// TIA Portal V17 export
// export: Created 2025-03-05T07:59:31.0674442Z, ExportSetting WithDefaults, DisplayName Totally Integrated Automation Portal, DisplayVersion V17 Update 8, DisplayName TIA Portal Openness, DisplayVersion V17 Update 8, DisplayName TIA Portal Version Control Interface, DisplayVersion V17, DisplayName SINAMICS Startdrive Advanced, DisplayVersion V17 SP2, DisplayName SINAMICS Startdrive G110M, G120, G120C, G120D, G120P, G115D, DisplayVersion V17 SP2, DisplayName SINAMICS Startdrive G130, G150, S120, S150, SINAMICS MV, S210, DisplayVersion V17 SP2, DisplayName STEP 7 Professional, DisplayVersion V17 Update 8, DisplayName SINUMERIK ONE STEP 7 Toolbox, DisplayVersion V17 Update 12, DisplayName SINUMERIK 840D sl STEP 7 Toolbox, DisplayVersion V17 Update 12, DisplayName STEP 7 Safety, DisplayVersion V17 Update 6, DisplayName WinCC Advanced, DisplayVersion V17 Update 8
FUNCTION "FC341_NCK_M_CH1_UNIT_1_STA_0" : Void   // FC341, LAD
TITLE = Channel 1 data
{ S7_Optimized_Access := 'FALSE' }
AUTHOR : ETXETAR
VERSION : 1.0
// stored: AutoNumber false, IsIECCheckEnabled false, SetENOAutomatically false, UDAEnableTagReadback false
   VAR_TEMP
      auxm3 : Bool;
      auxm5 : Bool;
      M253_TORQUE_ACTUAL_AUX_1 : Real;
      M253_TORQUE_ACTUAL_AUX_2 : Real;
   END_VAR
   VAR_TEMP   // added for the SCL form of the ladder/FBD networks
      _w1 : Bool;
      _w2 : Bool;
   END_VAR
BEGIN

REGION Network 1: CALL FB331 M CODE EXTENDED CH1 / M CODE EXTENDED CHANNEL 1
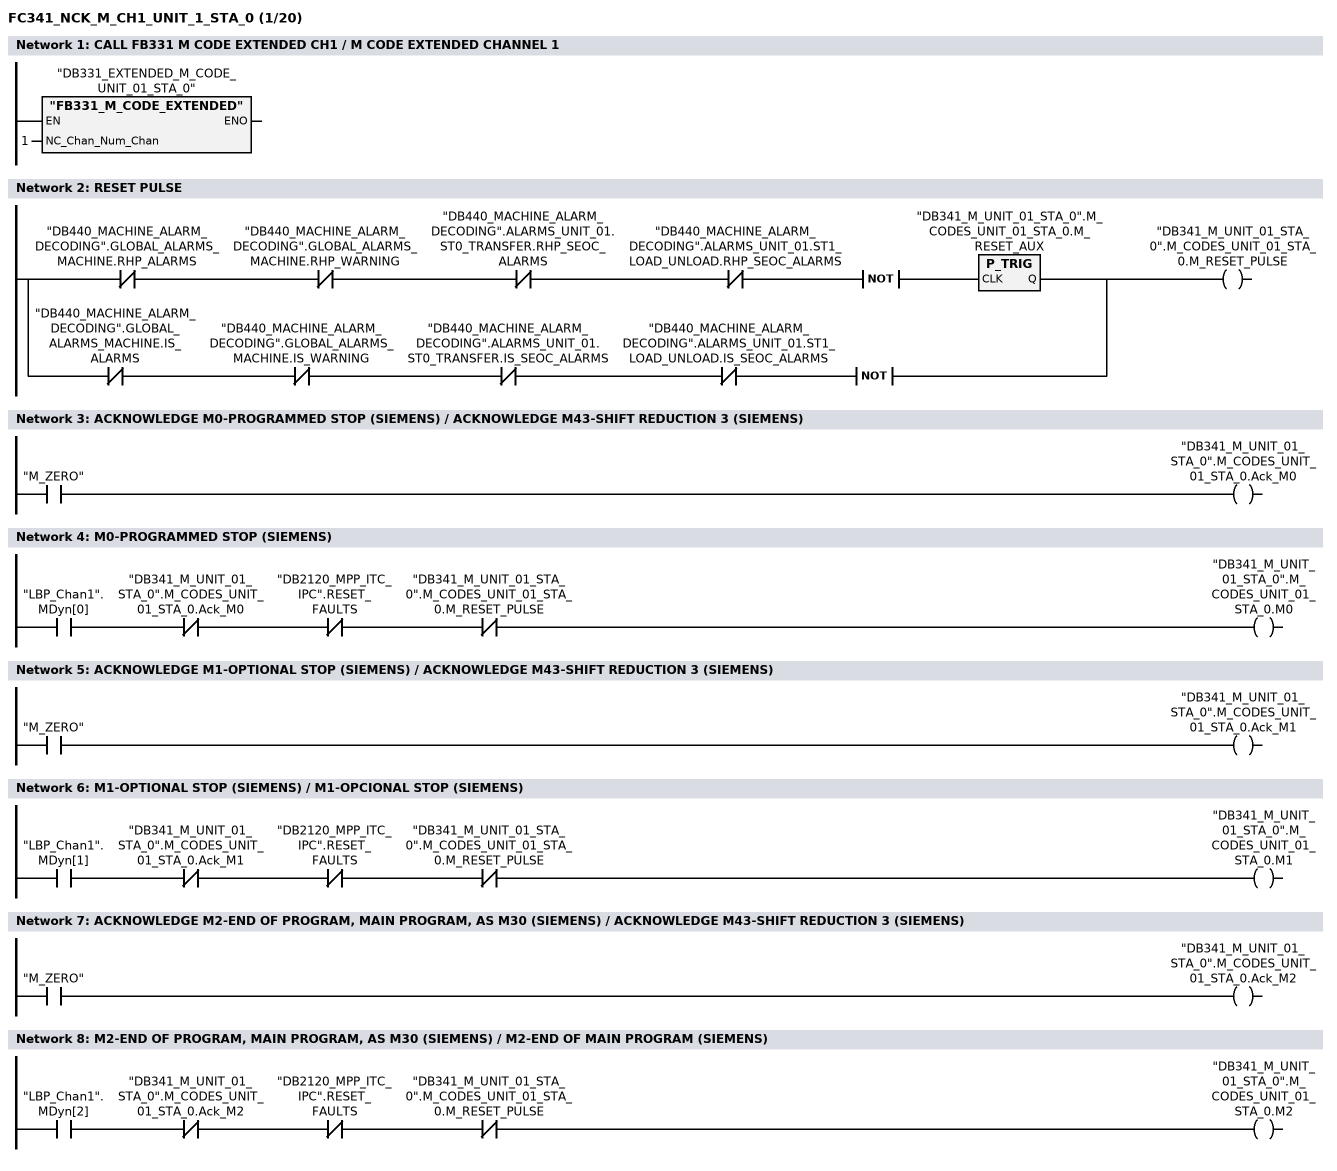
   RUNG wire#powerrail
      "DB331_EXTENDED_M_CODE_UNIT_01_STA_0"(NC_Chan_Num_Chan := 1)
   END_RUNG
   // the same network as SCL:
   "DB331_EXTENDED_M_CODE_UNIT_01_STA_0"(NC_Chan_Num_Chan := 1);   // "FB331_M_CODE_EXTENDED"
END_REGION

REGION Network 2: RESET PULSE
   RUNG wire#powerrail
      I_Contact( "DB440_MACHINE_ALARM_DECODING".GLOBAL_ALARMS_MACHINE.RHP_ALARMS )
      I_Contact( "DB440_MACHINE_ALARM_DECODING".GLOBAL_ALARMS_MACHINE.RHP_WARNING )
      I_Contact( "DB440_MACHINE_ALARM_DECODING".ALARMS_UNIT_01.ST0_TRANSFER.RHP_SEOC_ALARMS )
      I_Contact( "DB440_MACHINE_ALARM_DECODING".ALARMS_UNIT_01.ST1_LOAD_UNLOAD.RHP_SEOC_ALARMS )
      Not()
      P_Trig( "DB341_M_UNIT_01_STA_0".M_CODES_UNIT_01_STA_0.M_RESET_AUX )
      wire#w1
      Coil( "DB341_M_UNIT_01_STA_0".M_CODES_UNIT_01_STA_0.M_RESET_PULSE )
   END_RUNG
   RUNG wire#powerrail
      I_Contact( "DB440_MACHINE_ALARM_DECODING".GLOBAL_ALARMS_MACHINE.IS_ALARMS )
      I_Contact( "DB440_MACHINE_ALARM_DECODING".GLOBAL_ALARMS_MACHINE.IS_WARNING )
      I_Contact( "DB440_MACHINE_ALARM_DECODING".ALARMS_UNIT_01.ST0_TRANSFER.IS_SEOC_ALARMS )
      I_Contact( "DB440_MACHINE_ALARM_DECODING".ALARMS_UNIT_01.ST1_LOAD_UNLOAD.IS_SEOC_ALARMS )
      Not()
   END_RUNG wire#w1
   // the same network as SCL:
   #_w1 := NOT (NOT "DB440_MACHINE_ALARM_DECODING".GLOBAL_ALARMS_MACHINE.RHP_ALARMS AND NOT "DB440_MACHINE_ALARM_DECODING".GLOBAL_ALARMS_MACHINE.RHP_WARNING AND NOT "DB440_MACHINE_ALARM_DECODING".ALARMS_UNIT_01.ST0_TRANSFER.RHP_SEOC_ALARMS AND NOT "DB440_MACHINE_ALARM_DECODING".ALARMS_UNIT_01.ST1_LOAD_UNLOAD.RHP_SEOC_ALARMS);
   #_w2 := #_w1 AND NOT "DB341_M_UNIT_01_STA_0".M_CODES_UNIT_01_STA_0.M_RESET_AUX;   // rising edge
   "DB341_M_UNIT_01_STA_0".M_CODES_UNIT_01_STA_0.M_RESET_AUX := #_w1;
   "DB341_M_UNIT_01_STA_0".M_CODES_UNIT_01_STA_0.M_RESET_PULSE := #_w2 OR NOT (NOT "DB440_MACHINE_ALARM_DECODING".GLOBAL_ALARMS_MACHINE.IS_ALARMS AND NOT "DB440_MACHINE_ALARM_DECODING".GLOBAL_ALARMS_MACHINE.IS_WARNING AND NOT "DB440_MACHINE_ALARM_DECODING".ALARMS_UNIT_01.ST0_TRANSFER.IS_SEOC_ALARMS AND NOT "DB440_MACHINE_ALARM_DECODING".ALARMS_UNIT_01.ST1_LOAD_UNLOAD.IS_SEOC_ALARMS);
END_REGION

REGION Network 3: ACKNOWLEDGE M0-PROGRAMMED STOP (SIEMENS) / ACKNOWLEDGE M43-SHIFT REDUCTION 3 (SIEMENS)
   RUNG wire#powerrail
      Contact( "M_ZERO" )
      Coil( "DB341_M_UNIT_01_STA_0".M_CODES_UNIT_01_STA_0.Ack_M0 )
   END_RUNG
   // the same network as SCL:
   "DB341_M_UNIT_01_STA_0".M_CODES_UNIT_01_STA_0.Ack_M0 := "M_ZERO";
END_REGION

REGION Network 4: M0-PROGRAMMED STOP (SIEMENS)
   RUNG wire#powerrail
      Contact( "LBP_Chan1".MDyn[0] )
      I_Contact( "DB341_M_UNIT_01_STA_0".M_CODES_UNIT_01_STA_0.Ack_M0 )
      I_Contact( "DB2120_MPP_ITC_IPC".RESET_FAULTS )
      I_Contact( "DB341_M_UNIT_01_STA_0".M_CODES_UNIT_01_STA_0.M_RESET_PULSE )
      Coil( "DB341_M_UNIT_01_STA_0".M_CODES_UNIT_01_STA_0.M0 )
   END_RUNG
   // the same network as SCL:
   "DB341_M_UNIT_01_STA_0".M_CODES_UNIT_01_STA_0.M0 := "LBP_Chan1".MDyn[0] AND NOT "DB341_M_UNIT_01_STA_0".M_CODES_UNIT_01_STA_0.Ack_M0 AND NOT "DB2120_MPP_ITC_IPC".RESET_FAULTS AND NOT "DB341_M_UNIT_01_STA_0".M_CODES_UNIT_01_STA_0.M_RESET_PULSE;
END_REGION

REGION Network 5: ACKNOWLEDGE M1-OPTIONAL STOP (SIEMENS) / ACKNOWLEDGE M43-SHIFT REDUCTION 3 (SIEMENS)
   RUNG wire#powerrail
      Contact( "M_ZERO" )
      Coil( "DB341_M_UNIT_01_STA_0".M_CODES_UNIT_01_STA_0.Ack_M1 )
   END_RUNG
   // the same network as SCL:
   "DB341_M_UNIT_01_STA_0".M_CODES_UNIT_01_STA_0.Ack_M1 := "M_ZERO";
END_REGION

REGION Network 6: M1-OPTIONAL STOP (SIEMENS) / M1-OPCIONAL STOP (SIEMENS)
   RUNG wire#powerrail
      Contact( "LBP_Chan1".MDyn[1] )
      I_Contact( "DB341_M_UNIT_01_STA_0".M_CODES_UNIT_01_STA_0.Ack_M1 )
      I_Contact( "DB2120_MPP_ITC_IPC".RESET_FAULTS )
      I_Contact( "DB341_M_UNIT_01_STA_0".M_CODES_UNIT_01_STA_0.M_RESET_PULSE )
      Coil( "DB341_M_UNIT_01_STA_0".M_CODES_UNIT_01_STA_0.M1 )
   END_RUNG
   // the same network as SCL:
   "DB341_M_UNIT_01_STA_0".M_CODES_UNIT_01_STA_0.M1 := "LBP_Chan1".MDyn[1] AND NOT "DB341_M_UNIT_01_STA_0".M_CODES_UNIT_01_STA_0.Ack_M1 AND NOT "DB2120_MPP_ITC_IPC".RESET_FAULTS AND NOT "DB341_M_UNIT_01_STA_0".M_CODES_UNIT_01_STA_0.M_RESET_PULSE;
END_REGION

REGION Network 7: ACKNOWLEDGE M2-END OF PROGRAM, MAIN PROGRAM, AS M30 (SIEMENS) / ACKNOWLEDGE M43-SHIFT REDUCTION 3 (SIEMENS)
   RUNG wire#powerrail
      Contact( "M_ZERO" )
      Coil( "DB341_M_UNIT_01_STA_0".M_CODES_UNIT_01_STA_0.Ack_M2 )
   END_RUNG
   // the same network as SCL:
   "DB341_M_UNIT_01_STA_0".M_CODES_UNIT_01_STA_0.Ack_M2 := "M_ZERO";
END_REGION

REGION Network 8: M2-END OF PROGRAM, MAIN PROGRAM, AS M30 (SIEMENS) / M2-END OF MAIN PROGRAM (SIEMENS)
   RUNG wire#powerrail
      Contact( "LBP_Chan1".MDyn[2] )
      I_Contact( "DB341_M_UNIT_01_STA_0".M_CODES_UNIT_01_STA_0.Ack_M2 )
      I_Contact( "DB2120_MPP_ITC_IPC".RESET_FAULTS )
      I_Contact( "DB341_M_UNIT_01_STA_0".M_CODES_UNIT_01_STA_0.M_RESET_PULSE )
      Coil( "DB341_M_UNIT_01_STA_0".M_CODES_UNIT_01_STA_0.M2 )
   END_RUNG
   // the same network as SCL:
   "DB341_M_UNIT_01_STA_0".M_CODES_UNIT_01_STA_0.M2 := "LBP_Chan1".MDyn[2] AND NOT "DB341_M_UNIT_01_STA_0".M_CODES_UNIT_01_STA_0.Ack_M2 AND NOT "DB2120_MPP_ITC_IPC".RESET_FAULTS AND NOT "DB341_M_UNIT_01_STA_0".M_CODES_UNIT_01_STA_0.M_RESET_PULSE;
END_REGION

REGION Network 9: ACKNOWLEDGE M3-SPINDLE CLOCKWISE (SIEMENS) / ACKNOWLEDGE M3-START SPINDLE CLOCKWISE (SIEMENS)
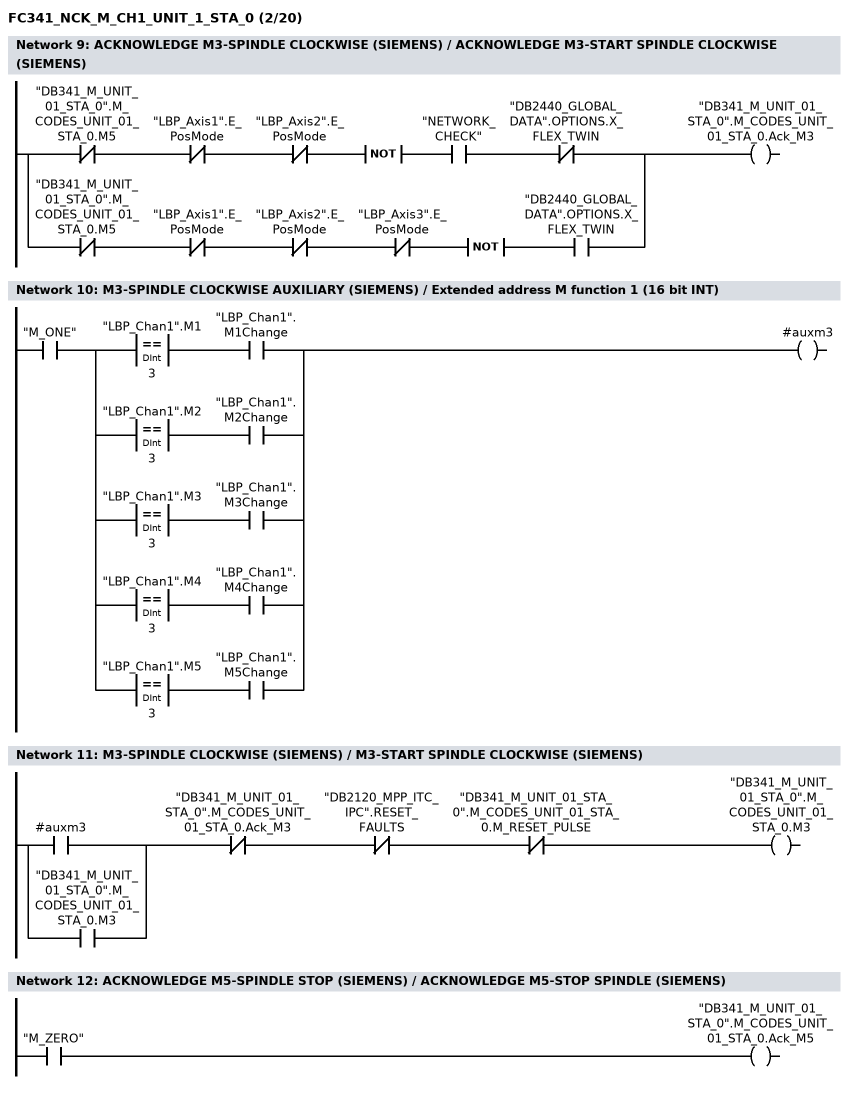
   RUNG wire#powerrail
      I_Contact( "DB341_M_UNIT_01_STA_0".M_CODES_UNIT_01_STA_0.M5 )
      I_Contact( "LBP_Axis1".E_PosMode )
      I_Contact( "LBP_Axis2".E_PosMode )
      Not()
      Contact( "NETWORK_CHECK" )
      I_Contact( "DB2440_GLOBAL_DATA".OPTIONS.X_FLEX_TWIN )
      wire#w1
      Coil( "DB341_M_UNIT_01_STA_0".M_CODES_UNIT_01_STA_0.Ack_M3 )
   END_RUNG
   RUNG wire#powerrail
      I_Contact( "DB341_M_UNIT_01_STA_0".M_CODES_UNIT_01_STA_0.M5 )
      I_Contact( "LBP_Axis1".E_PosMode )
      I_Contact( "LBP_Axis2".E_PosMode )
      I_Contact( "LBP_Axis3".E_PosMode )
      Not()
      Contact( "DB2440_GLOBAL_DATA".OPTIONS.X_FLEX_TWIN )
   END_RUNG wire#w1
   // the same network as SCL:
   "DB341_M_UNIT_01_STA_0".M_CODES_UNIT_01_STA_0.Ack_M3 := (NOT (NOT "DB341_M_UNIT_01_STA_0".M_CODES_UNIT_01_STA_0.M5 AND NOT "LBP_Axis1".E_PosMode AND NOT "LBP_Axis2".E_PosMode) AND "NETWORK_CHECK" AND NOT "DB2440_GLOBAL_DATA".OPTIONS.X_FLEX_TWIN) OR (NOT (NOT "DB341_M_UNIT_01_STA_0".M_CODES_UNIT_01_STA_0.M5 AND NOT "LBP_Axis1".E_PosMode AND NOT "LBP_Axis2".E_PosMode AND NOT "LBP_Axis3".E_PosMode) AND "DB2440_GLOBAL_DATA".OPTIONS.X_FLEX_TWIN);
END_REGION

REGION Network 10: M3-SPINDLE CLOCKWISE AUXILIARY (SIEMENS) / Extended address M function 1 (16 bit INT)
   RUNG wire#powerrail
      Contact( "M_ONE" )
      wire#w1
      { S7_Templates := "SrcType := DInt" } EQ_Contact(in1 := "LBP_Chan1".M1, in2 := 3)
      Contact( "LBP_Chan1".M1Change )
      wire#w2
      Coil( #auxm3 )
   END_RUNG
   RUNG wire#w1
      { S7_Templates := "SrcType := DInt" } EQ_Contact(in1 := "LBP_Chan1".M2, in2 := 3)
      Contact( "LBP_Chan1".M2Change )
   END_RUNG wire#w2
   RUNG wire#w1
      { S7_Templates := "SrcType := DInt" } EQ_Contact(in1 := "LBP_Chan1".M3, in2 := 3)
      Contact( "LBP_Chan1".M3Change )
   END_RUNG wire#w2
   RUNG wire#w1
      { S7_Templates := "SrcType := DInt" } EQ_Contact(in1 := "LBP_Chan1".M4, in2 := 3)
      Contact( "LBP_Chan1".M4Change )
   END_RUNG wire#w2
   RUNG wire#w1
      { S7_Templates := "SrcType := DInt" } EQ_Contact(in1 := "LBP_Chan1".M5, in2 := 3)
      Contact( "LBP_Chan1".M5Change )
   END_RUNG wire#w2
   // the same network as SCL:
   #auxm3 := "M_ONE" AND ((("LBP_Chan1".M1 = 3) AND "LBP_Chan1".M1Change) OR (("LBP_Chan1".M2 = 3) AND "LBP_Chan1".M2Change) OR (("LBP_Chan1".M3 = 3) AND "LBP_Chan1".M3Change) OR (("LBP_Chan1".M4 = 3) AND "LBP_Chan1".M4Change) OR (("LBP_Chan1".M5 = 3) AND "LBP_Chan1".M5Change));
END_REGION

REGION Network 11: M3-SPINDLE CLOCKWISE (SIEMENS) / M3-START SPINDLE CLOCKWISE (SIEMENS)
   RUNG wire#powerrail
      Contact( #auxm3 )
      wire#w1
      I_Contact( "DB341_M_UNIT_01_STA_0".M_CODES_UNIT_01_STA_0.Ack_M3 )
      I_Contact( "DB2120_MPP_ITC_IPC".RESET_FAULTS )
      I_Contact( "DB341_M_UNIT_01_STA_0".M_CODES_UNIT_01_STA_0.M_RESET_PULSE )
      Coil( "DB341_M_UNIT_01_STA_0".M_CODES_UNIT_01_STA_0.M3 )
   END_RUNG
   RUNG wire#powerrail
      Contact( "DB341_M_UNIT_01_STA_0".M_CODES_UNIT_01_STA_0.M3 )
   END_RUNG wire#w1
   // the same network as SCL:
   "DB341_M_UNIT_01_STA_0".M_CODES_UNIT_01_STA_0.M3 := (#auxm3 OR "DB341_M_UNIT_01_STA_0".M_CODES_UNIT_01_STA_0.M3) AND NOT "DB341_M_UNIT_01_STA_0".M_CODES_UNIT_01_STA_0.Ack_M3 AND NOT "DB2120_MPP_ITC_IPC".RESET_FAULTS AND NOT "DB341_M_UNIT_01_STA_0".M_CODES_UNIT_01_STA_0.M_RESET_PULSE;
END_REGION

REGION Network 12: ACKNOWLEDGE M5-SPINDLE STOP (SIEMENS) / ACKNOWLEDGE M5-STOP SPINDLE (SIEMENS)
   RUNG wire#powerrail
      Contact( "M_ZERO" )
      Coil( "DB341_M_UNIT_01_STA_0".M_CODES_UNIT_01_STA_0.Ack_M5 )
   END_RUNG
   // the same network as SCL:
   "DB341_M_UNIT_01_STA_0".M_CODES_UNIT_01_STA_0.Ack_M5 := "M_ZERO";
END_REGION

REGION Network 13: M5-SPINDLE STOP AUXILIARY (SIEMENS) / Auxilir M5
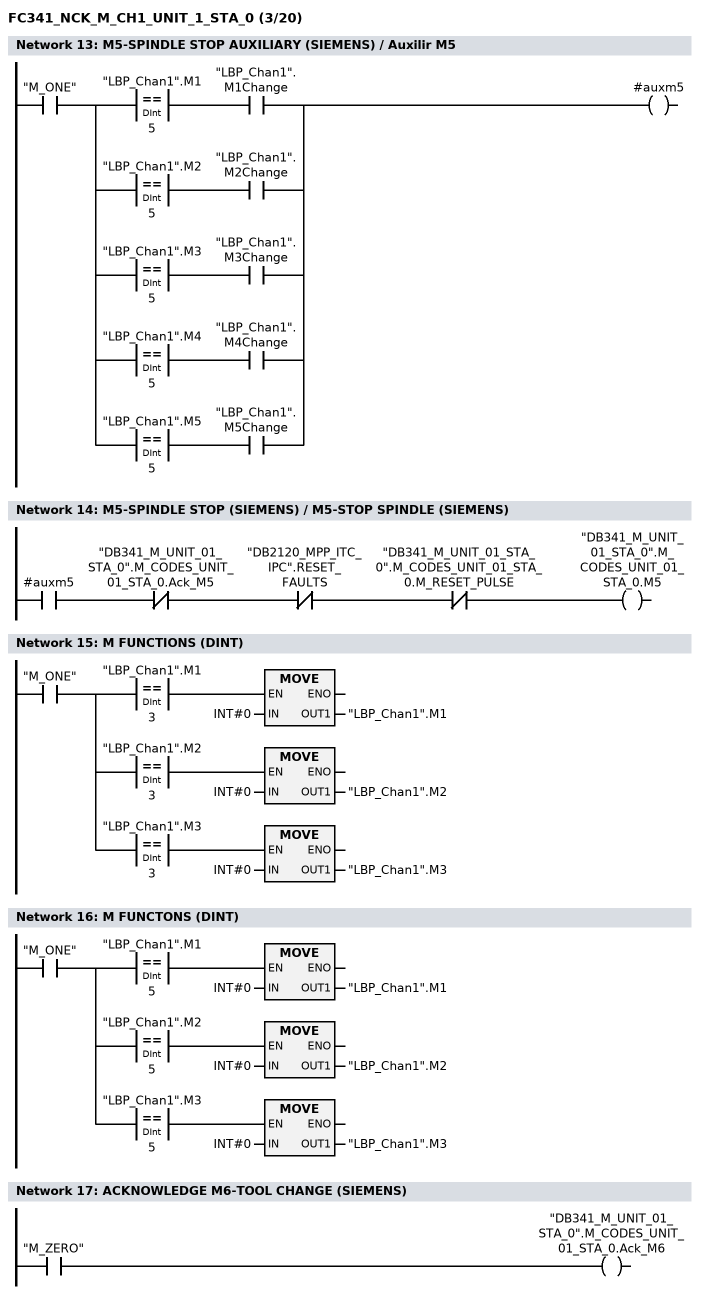
   RUNG wire#powerrail
      Contact( "M_ONE" )
      wire#w1
      { S7_Templates := "SrcType := DInt" } EQ_Contact(in1 := "LBP_Chan1".M1, in2 := 5)
      Contact( "LBP_Chan1".M1Change )
      wire#w2
      Coil( #auxm5 )
   END_RUNG
   RUNG wire#w1
      { S7_Templates := "SrcType := DInt" } EQ_Contact(in1 := "LBP_Chan1".M2, in2 := 5)
      Contact( "LBP_Chan1".M2Change )
   END_RUNG wire#w2
   RUNG wire#w1
      { S7_Templates := "SrcType := DInt" } EQ_Contact(in1 := "LBP_Chan1".M3, in2 := 5)
      Contact( "LBP_Chan1".M3Change )
   END_RUNG wire#w2
   RUNG wire#w1
      { S7_Templates := "SrcType := DInt" } EQ_Contact(in1 := "LBP_Chan1".M4, in2 := 5)
      Contact( "LBP_Chan1".M4Change )
   END_RUNG wire#w2
   RUNG wire#w1
      { S7_Templates := "SrcType := DInt" } EQ_Contact(in1 := "LBP_Chan1".M5, in2 := 5)
      Contact( "LBP_Chan1".M5Change )
   END_RUNG wire#w2
   // the same network as SCL:
   #auxm5 := "M_ONE" AND ((("LBP_Chan1".M1 = 5) AND "LBP_Chan1".M1Change) OR (("LBP_Chan1".M2 = 5) AND "LBP_Chan1".M2Change) OR (("LBP_Chan1".M3 = 5) AND "LBP_Chan1".M3Change) OR (("LBP_Chan1".M4 = 5) AND "LBP_Chan1".M4Change) OR (("LBP_Chan1".M5 = 5) AND "LBP_Chan1".M5Change));
END_REGION

REGION Network 14: M5-SPINDLE STOP (SIEMENS) / M5-STOP SPINDLE (SIEMENS)
   RUNG wire#powerrail
      Contact( #auxm5 )
      I_Contact( "DB341_M_UNIT_01_STA_0".M_CODES_UNIT_01_STA_0.Ack_M5 )
      I_Contact( "DB2120_MPP_ITC_IPC".RESET_FAULTS )
      I_Contact( "DB341_M_UNIT_01_STA_0".M_CODES_UNIT_01_STA_0.M_RESET_PULSE )
      Coil( "DB341_M_UNIT_01_STA_0".M_CODES_UNIT_01_STA_0.M5 )
   END_RUNG
   // the same network as SCL:
   "DB341_M_UNIT_01_STA_0".M_CODES_UNIT_01_STA_0.M5 := #auxm5 AND NOT "DB341_M_UNIT_01_STA_0".M_CODES_UNIT_01_STA_0.Ack_M5 AND NOT "DB2120_MPP_ITC_IPC".RESET_FAULTS AND NOT "DB341_M_UNIT_01_STA_0".M_CODES_UNIT_01_STA_0.M_RESET_PULSE;
END_REGION

REGION Network 15: M FUNCTIONS (DINT)
   RUNG wire#powerrail
      Contact( "M_ONE" )
      wire#w1
      { S7_Templates := "SrcType := DInt" } EQ_Contact(in1 := "LBP_Chan1".M1, in2 := 3)
      { S7_GenerateENO := "TRUE" } Move(in := INT#0, out1 => "LBP_Chan1".M1)
   END_RUNG
   RUNG wire#w1
      { S7_Templates := "SrcType := DInt" } EQ_Contact(in1 := "LBP_Chan1".M2, in2 := 3)
      { S7_GenerateENO := "TRUE" } Move(in := INT#0, out1 => "LBP_Chan1".M2)
   END_RUNG
   RUNG wire#w1
      { S7_Templates := "SrcType := DInt" } EQ_Contact(in1 := "LBP_Chan1".M3, in2 := 3)
      { S7_GenerateENO := "TRUE" } Move(in := INT#0, out1 => "LBP_Chan1".M3)
   END_RUNG
   // the same network as SCL:
   IF "M_ONE" AND ("LBP_Chan1".M1 = 3) THEN "LBP_Chan1".M1 := INT#0; END_IF;
   IF "M_ONE" AND ("LBP_Chan1".M2 = 3) THEN "LBP_Chan1".M2 := INT#0; END_IF;
   IF "M_ONE" AND ("LBP_Chan1".M3 = 3) THEN "LBP_Chan1".M3 := INT#0; END_IF;
END_REGION

REGION Network 16: M FUNCTONS (DINT)
   RUNG wire#powerrail
      Contact( "M_ONE" )
      wire#w1
      { S7_Templates := "SrcType := DInt" } EQ_Contact(in1 := "LBP_Chan1".M1, in2 := 5)
      { S7_GenerateENO := "TRUE" } Move(in := INT#0, out1 => "LBP_Chan1".M1)
   END_RUNG
   RUNG wire#w1
      { S7_Templates := "SrcType := DInt" } EQ_Contact(in1 := "LBP_Chan1".M2, in2 := 5)
      { S7_GenerateENO := "TRUE" } Move(in := INT#0, out1 => "LBP_Chan1".M2)
   END_RUNG
   RUNG wire#w1
      { S7_Templates := "SrcType := DInt" } EQ_Contact(in1 := "LBP_Chan1".M3, in2 := 5)
      { S7_GenerateENO := "TRUE" } Move(in := INT#0, out1 => "LBP_Chan1".M3)
   END_RUNG
   // the same network as SCL:
   IF "M_ONE" AND ("LBP_Chan1".M1 = 5) THEN "LBP_Chan1".M1 := INT#0; END_IF;
   IF "M_ONE" AND ("LBP_Chan1".M2 = 5) THEN "LBP_Chan1".M2 := INT#0; END_IF;
   IF "M_ONE" AND ("LBP_Chan1".M3 = 5) THEN "LBP_Chan1".M3 := INT#0; END_IF;
END_REGION

REGION Network 17: ACKNOWLEDGE M6-TOOL CHANGE (SIEMENS)
   RUNG wire#powerrail
      Contact( "M_ZERO" )
      Coil( "DB341_M_UNIT_01_STA_0".M_CODES_UNIT_01_STA_0.Ack_M6 )
   END_RUNG
   // the same network as SCL:
   "DB341_M_UNIT_01_STA_0".M_CODES_UNIT_01_STA_0.Ack_M6 := "M_ZERO";
END_REGION

REGION Network 18: M6-TOOL CHANGE (SIEMENS)
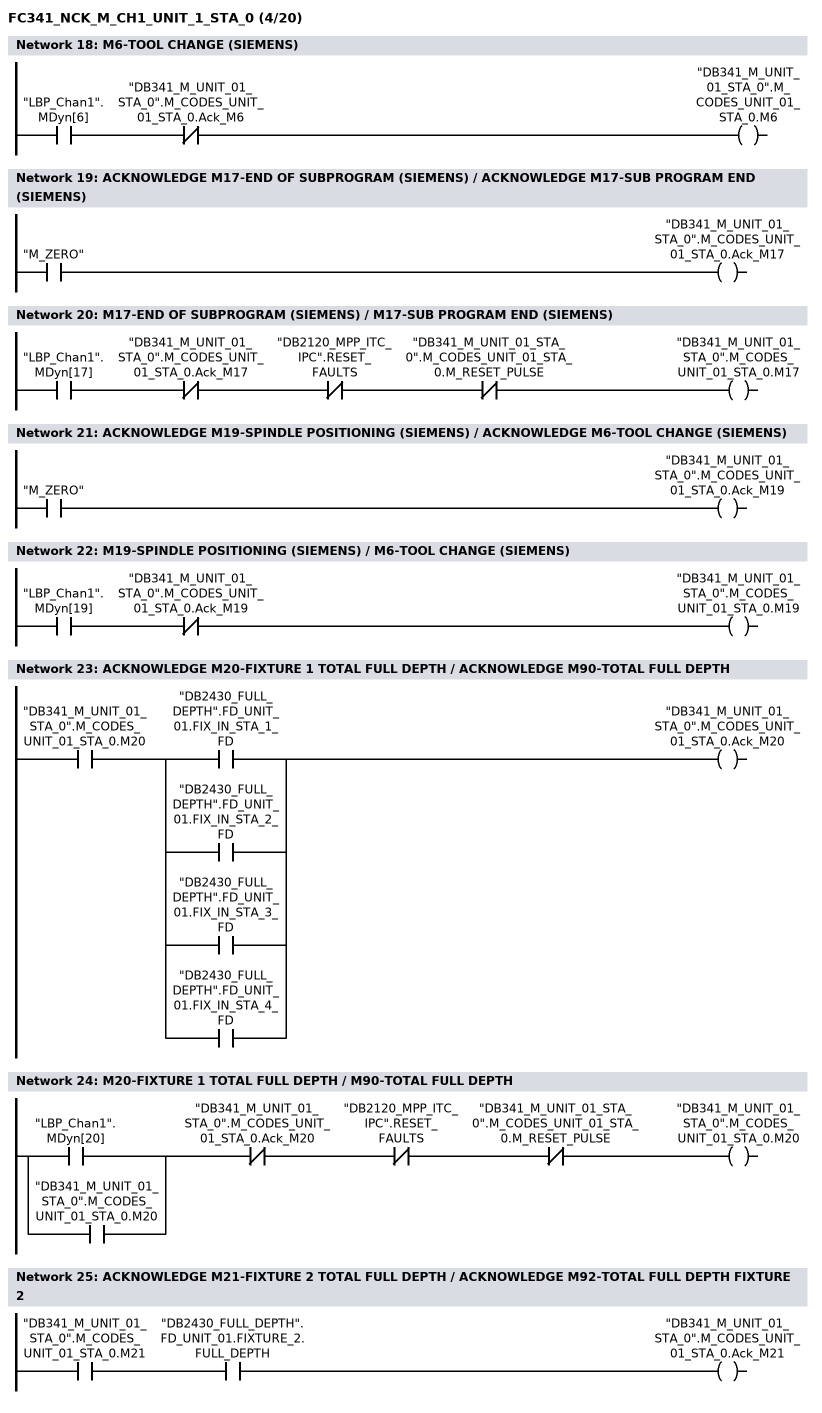
   RUNG wire#powerrail
      Contact( "LBP_Chan1".MDyn[6] )
      I_Contact( "DB341_M_UNIT_01_STA_0".M_CODES_UNIT_01_STA_0.Ack_M6 )
      Coil( "DB341_M_UNIT_01_STA_0".M_CODES_UNIT_01_STA_0.M6 )
   END_RUNG
   // the same network as SCL:
   "DB341_M_UNIT_01_STA_0".M_CODES_UNIT_01_STA_0.M6 := "LBP_Chan1".MDyn[6] AND NOT "DB341_M_UNIT_01_STA_0".M_CODES_UNIT_01_STA_0.Ack_M6;
END_REGION

REGION Network 19: ACKNOWLEDGE M17-END OF SUBPROGRAM (SIEMENS) / ACKNOWLEDGE M17-SUB PROGRAM END (SIEMENS)
   RUNG wire#powerrail
      Contact( "M_ZERO" )
      Coil( "DB341_M_UNIT_01_STA_0".M_CODES_UNIT_01_STA_0.Ack_M17 )
   END_RUNG
   // the same network as SCL:
   "DB341_M_UNIT_01_STA_0".M_CODES_UNIT_01_STA_0.Ack_M17 := "M_ZERO";
END_REGION

REGION Network 20: M17-END OF SUBPROGRAM (SIEMENS) / M17-SUB PROGRAM END (SIEMENS)
   RUNG wire#powerrail
      Contact( "LBP_Chan1".MDyn[17] )
      I_Contact( "DB341_M_UNIT_01_STA_0".M_CODES_UNIT_01_STA_0.Ack_M17 )
      I_Contact( "DB2120_MPP_ITC_IPC".RESET_FAULTS )
      I_Contact( "DB341_M_UNIT_01_STA_0".M_CODES_UNIT_01_STA_0.M_RESET_PULSE )
      Coil( "DB341_M_UNIT_01_STA_0".M_CODES_UNIT_01_STA_0.M17 )
   END_RUNG
   // the same network as SCL:
   "DB341_M_UNIT_01_STA_0".M_CODES_UNIT_01_STA_0.M17 := "LBP_Chan1".MDyn[17] AND NOT "DB341_M_UNIT_01_STA_0".M_CODES_UNIT_01_STA_0.Ack_M17 AND NOT "DB2120_MPP_ITC_IPC".RESET_FAULTS AND NOT "DB341_M_UNIT_01_STA_0".M_CODES_UNIT_01_STA_0.M_RESET_PULSE;
END_REGION

REGION Network 21: ACKNOWLEDGE M19-SPINDLE POSITIONING (SIEMENS) / ACKNOWLEDGE M6-TOOL CHANGE (SIEMENS)
   RUNG wire#powerrail
      Contact( "M_ZERO" )
      Coil( "DB341_M_UNIT_01_STA_0".M_CODES_UNIT_01_STA_0.Ack_M19 )
   END_RUNG
   // the same network as SCL:
   "DB341_M_UNIT_01_STA_0".M_CODES_UNIT_01_STA_0.Ack_M19 := "M_ZERO";
END_REGION

REGION Network 22: M19-SPINDLE POSITIONING (SIEMENS) / M6-TOOL CHANGE (SIEMENS)
   RUNG wire#powerrail
      Contact( "LBP_Chan1".MDyn[19] )
      I_Contact( "DB341_M_UNIT_01_STA_0".M_CODES_UNIT_01_STA_0.Ack_M19 )
      Coil( "DB341_M_UNIT_01_STA_0".M_CODES_UNIT_01_STA_0.M19 )
   END_RUNG
   // the same network as SCL:
   "DB341_M_UNIT_01_STA_0".M_CODES_UNIT_01_STA_0.M19 := "LBP_Chan1".MDyn[19] AND NOT "DB341_M_UNIT_01_STA_0".M_CODES_UNIT_01_STA_0.Ack_M19;
END_REGION

REGION Network 23: ACKNOWLEDGE M20-FIXTURE 1 TOTAL FULL DEPTH / ACKNOWLEDGE M90-TOTAL FULL DEPTH
   RUNG wire#powerrail
      Contact( "DB341_M_UNIT_01_STA_0".M_CODES_UNIT_01_STA_0.M20 )
      wire#w1
      Contact( "DB2430_FULL_DEPTH".FD_UNIT_01.FIX_IN_STA_1_FD )
      wire#w2
      Coil( "DB341_M_UNIT_01_STA_0".M_CODES_UNIT_01_STA_0.Ack_M20 )
   END_RUNG
   RUNG wire#w1
      Contact( "DB2430_FULL_DEPTH".FD_UNIT_01.FIX_IN_STA_2_FD )
   END_RUNG wire#w2
   RUNG wire#w1
      Contact( "DB2430_FULL_DEPTH".FD_UNIT_01.FIX_IN_STA_3_FD )
   END_RUNG wire#w2
   RUNG wire#w1
      Contact( "DB2430_FULL_DEPTH".FD_UNIT_01.FIX_IN_STA_4_FD )
   END_RUNG wire#w2
   // the same network as SCL:
   "DB341_M_UNIT_01_STA_0".M_CODES_UNIT_01_STA_0.Ack_M20 := "DB341_M_UNIT_01_STA_0".M_CODES_UNIT_01_STA_0.M20 AND ("DB2430_FULL_DEPTH".FD_UNIT_01.FIX_IN_STA_1_FD OR "DB2430_FULL_DEPTH".FD_UNIT_01.FIX_IN_STA_2_FD OR "DB2430_FULL_DEPTH".FD_UNIT_01.FIX_IN_STA_3_FD OR "DB2430_FULL_DEPTH".FD_UNIT_01.FIX_IN_STA_4_FD);
END_REGION

REGION Network 24: M20-FIXTURE 1 TOTAL FULL DEPTH / M90-TOTAL FULL DEPTH
   RUNG wire#powerrail
      Contact( "LBP_Chan1".MDyn[20] )
      wire#w1
      I_Contact( "DB341_M_UNIT_01_STA_0".M_CODES_UNIT_01_STA_0.Ack_M20 )
      I_Contact( "DB2120_MPP_ITC_IPC".RESET_FAULTS )
      I_Contact( "DB341_M_UNIT_01_STA_0".M_CODES_UNIT_01_STA_0.M_RESET_PULSE )
      Coil( "DB341_M_UNIT_01_STA_0".M_CODES_UNIT_01_STA_0.M20 )
   END_RUNG
   RUNG wire#powerrail
      Contact( "DB341_M_UNIT_01_STA_0".M_CODES_UNIT_01_STA_0.M20 )
   END_RUNG wire#w1
   // the same network as SCL:
   "DB341_M_UNIT_01_STA_0".M_CODES_UNIT_01_STA_0.M20 := ("LBP_Chan1".MDyn[20] OR "DB341_M_UNIT_01_STA_0".M_CODES_UNIT_01_STA_0.M20) AND NOT "DB341_M_UNIT_01_STA_0".M_CODES_UNIT_01_STA_0.Ack_M20 AND NOT "DB2120_MPP_ITC_IPC".RESET_FAULTS AND NOT "DB341_M_UNIT_01_STA_0".M_CODES_UNIT_01_STA_0.M_RESET_PULSE;
END_REGION

REGION Network 25: ACKNOWLEDGE M21-FIXTURE 2 TOTAL FULL DEPTH / ACKNOWLEDGE M92-TOTAL FULL DEPTH FIXTURE 2
   RUNG wire#powerrail
      Contact( "DB341_M_UNIT_01_STA_0".M_CODES_UNIT_01_STA_0.M21 )
      Contact( "DB2430_FULL_DEPTH".FD_UNIT_01.FIXTURE_2.FULL_DEPTH )
      Coil( "DB341_M_UNIT_01_STA_0".M_CODES_UNIT_01_STA_0.Ack_M21 )
   END_RUNG
   // the same network as SCL:
   "DB341_M_UNIT_01_STA_0".M_CODES_UNIT_01_STA_0.Ack_M21 := "DB341_M_UNIT_01_STA_0".M_CODES_UNIT_01_STA_0.M21 AND "DB2430_FULL_DEPTH".FD_UNIT_01.FIXTURE_2.FULL_DEPTH;
END_REGION

REGION Network 26: M21-FIXTURE 2 TOTAL FULL DEPTH / M92-TOTAL FULL DEPTH FIXTURE 2
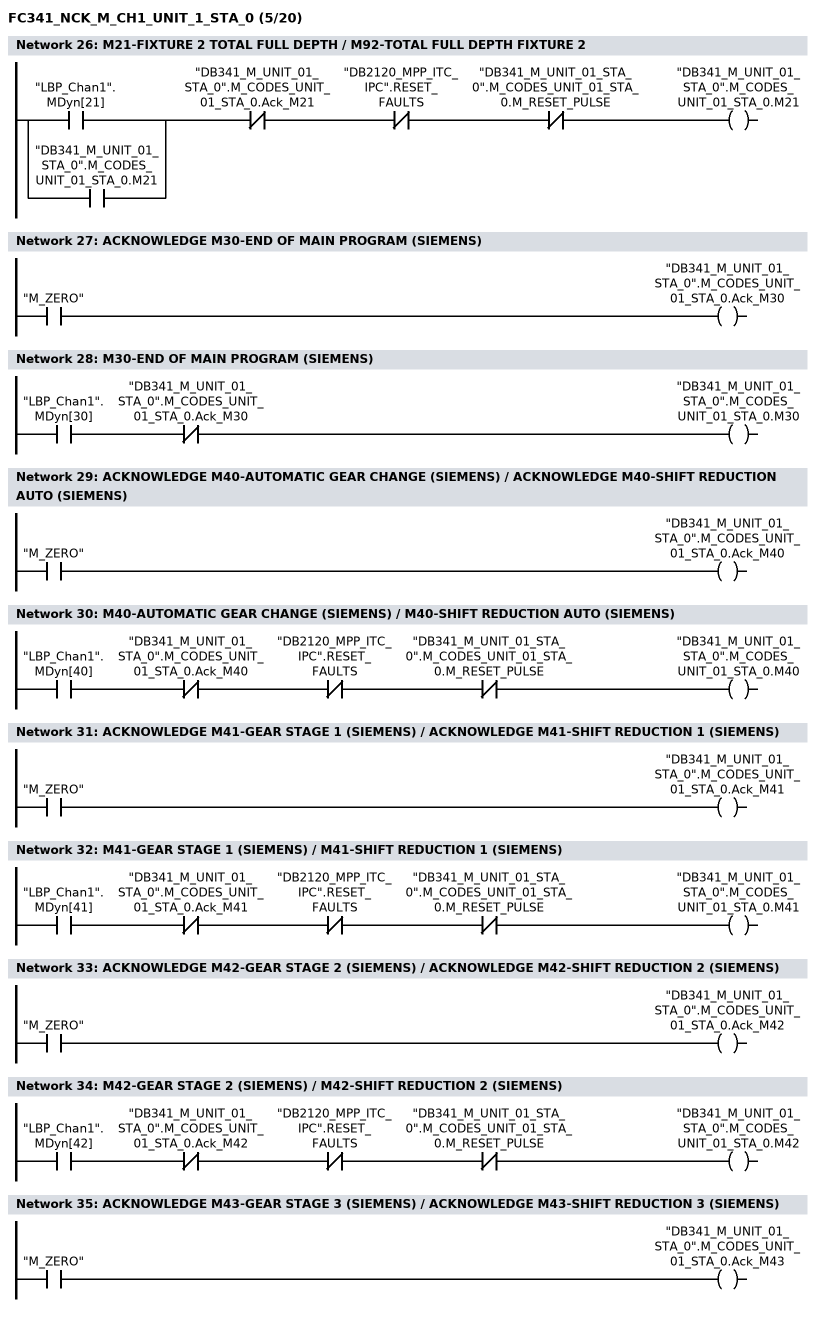
   RUNG wire#powerrail
      Contact( "LBP_Chan1".MDyn[21] )
      wire#w1
      I_Contact( "DB341_M_UNIT_01_STA_0".M_CODES_UNIT_01_STA_0.Ack_M21 )
      I_Contact( "DB2120_MPP_ITC_IPC".RESET_FAULTS )
      I_Contact( "DB341_M_UNIT_01_STA_0".M_CODES_UNIT_01_STA_0.M_RESET_PULSE )
      Coil( "DB341_M_UNIT_01_STA_0".M_CODES_UNIT_01_STA_0.M21 )
   END_RUNG
   RUNG wire#powerrail
      Contact( "DB341_M_UNIT_01_STA_0".M_CODES_UNIT_01_STA_0.M21 )
   END_RUNG wire#w1
   // the same network as SCL:
   "DB341_M_UNIT_01_STA_0".M_CODES_UNIT_01_STA_0.M21 := ("LBP_Chan1".MDyn[21] OR "DB341_M_UNIT_01_STA_0".M_CODES_UNIT_01_STA_0.M21) AND NOT "DB341_M_UNIT_01_STA_0".M_CODES_UNIT_01_STA_0.Ack_M21 AND NOT "DB2120_MPP_ITC_IPC".RESET_FAULTS AND NOT "DB341_M_UNIT_01_STA_0".M_CODES_UNIT_01_STA_0.M_RESET_PULSE;
END_REGION

REGION Network 27: ACKNOWLEDGE M30-END OF MAIN PROGRAM (SIEMENS)
   RUNG wire#powerrail
      Contact( "M_ZERO" )
      Coil( "DB341_M_UNIT_01_STA_0".M_CODES_UNIT_01_STA_0.Ack_M30 )
   END_RUNG
   // the same network as SCL:
   "DB341_M_UNIT_01_STA_0".M_CODES_UNIT_01_STA_0.Ack_M30 := "M_ZERO";
END_REGION

REGION Network 28: M30-END OF MAIN PROGRAM (SIEMENS)
   RUNG wire#powerrail
      Contact( "LBP_Chan1".MDyn[30] )
      I_Contact( "DB341_M_UNIT_01_STA_0".M_CODES_UNIT_01_STA_0.Ack_M30 )
      Coil( "DB341_M_UNIT_01_STA_0".M_CODES_UNIT_01_STA_0.M30 )
   END_RUNG
   // the same network as SCL:
   "DB341_M_UNIT_01_STA_0".M_CODES_UNIT_01_STA_0.M30 := "LBP_Chan1".MDyn[30] AND NOT "DB341_M_UNIT_01_STA_0".M_CODES_UNIT_01_STA_0.Ack_M30;
END_REGION

REGION Network 29: ACKNOWLEDGE M40-AUTOMATIC GEAR CHANGE (SIEMENS) / ACKNOWLEDGE M40-SHIFT REDUCTION AUTO (SIEMENS)
   RUNG wire#powerrail
      Contact( "M_ZERO" )
      Coil( "DB341_M_UNIT_01_STA_0".M_CODES_UNIT_01_STA_0.Ack_M40 )
   END_RUNG
   // the same network as SCL:
   "DB341_M_UNIT_01_STA_0".M_CODES_UNIT_01_STA_0.Ack_M40 := "M_ZERO";
END_REGION

REGION Network 30: M40-AUTOMATIC GEAR CHANGE (SIEMENS) / M40-SHIFT REDUCTION AUTO (SIEMENS)
   RUNG wire#powerrail
      Contact( "LBP_Chan1".MDyn[40] )
      I_Contact( "DB341_M_UNIT_01_STA_0".M_CODES_UNIT_01_STA_0.Ack_M40 )
      I_Contact( "DB2120_MPP_ITC_IPC".RESET_FAULTS )
      I_Contact( "DB341_M_UNIT_01_STA_0".M_CODES_UNIT_01_STA_0.M_RESET_PULSE )
      Coil( "DB341_M_UNIT_01_STA_0".M_CODES_UNIT_01_STA_0.M40 )
   END_RUNG
   // the same network as SCL:
   "DB341_M_UNIT_01_STA_0".M_CODES_UNIT_01_STA_0.M40 := "LBP_Chan1".MDyn[40] AND NOT "DB341_M_UNIT_01_STA_0".M_CODES_UNIT_01_STA_0.Ack_M40 AND NOT "DB2120_MPP_ITC_IPC".RESET_FAULTS AND NOT "DB341_M_UNIT_01_STA_0".M_CODES_UNIT_01_STA_0.M_RESET_PULSE;
END_REGION

REGION Network 31: ACKNOWLEDGE M41-GEAR STAGE 1 (SIEMENS) / ACKNOWLEDGE M41-SHIFT REDUCTION 1 (SIEMENS)
   RUNG wire#powerrail
      Contact( "M_ZERO" )
      Coil( "DB341_M_UNIT_01_STA_0".M_CODES_UNIT_01_STA_0.Ack_M41 )
   END_RUNG
   // the same network as SCL:
   "DB341_M_UNIT_01_STA_0".M_CODES_UNIT_01_STA_0.Ack_M41 := "M_ZERO";
END_REGION

REGION Network 32: M41-GEAR STAGE 1 (SIEMENS) / M41-SHIFT REDUCTION 1 (SIEMENS)
   RUNG wire#powerrail
      Contact( "LBP_Chan1".MDyn[41] )
      I_Contact( "DB341_M_UNIT_01_STA_0".M_CODES_UNIT_01_STA_0.Ack_M41 )
      I_Contact( "DB2120_MPP_ITC_IPC".RESET_FAULTS )
      I_Contact( "DB341_M_UNIT_01_STA_0".M_CODES_UNIT_01_STA_0.M_RESET_PULSE )
      Coil( "DB341_M_UNIT_01_STA_0".M_CODES_UNIT_01_STA_0.M41 )
   END_RUNG
   // the same network as SCL:
   "DB341_M_UNIT_01_STA_0".M_CODES_UNIT_01_STA_0.M41 := "LBP_Chan1".MDyn[41] AND NOT "DB341_M_UNIT_01_STA_0".M_CODES_UNIT_01_STA_0.Ack_M41 AND NOT "DB2120_MPP_ITC_IPC".RESET_FAULTS AND NOT "DB341_M_UNIT_01_STA_0".M_CODES_UNIT_01_STA_0.M_RESET_PULSE;
END_REGION

REGION Network 33: ACKNOWLEDGE M42-GEAR STAGE 2 (SIEMENS) / ACKNOWLEDGE M42-SHIFT REDUCTION 2 (SIEMENS)
   RUNG wire#powerrail
      Contact( "M_ZERO" )
      Coil( "DB341_M_UNIT_01_STA_0".M_CODES_UNIT_01_STA_0.Ack_M42 )
   END_RUNG
   // the same network as SCL:
   "DB341_M_UNIT_01_STA_0".M_CODES_UNIT_01_STA_0.Ack_M42 := "M_ZERO";
END_REGION

REGION Network 34: M42-GEAR STAGE 2 (SIEMENS) / M42-SHIFT REDUCTION 2 (SIEMENS)
   RUNG wire#powerrail
      Contact( "LBP_Chan1".MDyn[42] )
      I_Contact( "DB341_M_UNIT_01_STA_0".M_CODES_UNIT_01_STA_0.Ack_M42 )
      I_Contact( "DB2120_MPP_ITC_IPC".RESET_FAULTS )
      I_Contact( "DB341_M_UNIT_01_STA_0".M_CODES_UNIT_01_STA_0.M_RESET_PULSE )
      Coil( "DB341_M_UNIT_01_STA_0".M_CODES_UNIT_01_STA_0.M42 )
   END_RUNG
   // the same network as SCL:
   "DB341_M_UNIT_01_STA_0".M_CODES_UNIT_01_STA_0.M42 := "LBP_Chan1".MDyn[42] AND NOT "DB341_M_UNIT_01_STA_0".M_CODES_UNIT_01_STA_0.Ack_M42 AND NOT "DB2120_MPP_ITC_IPC".RESET_FAULTS AND NOT "DB341_M_UNIT_01_STA_0".M_CODES_UNIT_01_STA_0.M_RESET_PULSE;
END_REGION

REGION Network 35: ACKNOWLEDGE M43-GEAR STAGE 3 (SIEMENS) / ACKNOWLEDGE M43-SHIFT REDUCTION 3 (SIEMENS)
   RUNG wire#powerrail
      Contact( "M_ZERO" )
      Coil( "DB341_M_UNIT_01_STA_0".M_CODES_UNIT_01_STA_0.Ack_M43 )
   END_RUNG
   // the same network as SCL:
   "DB341_M_UNIT_01_STA_0".M_CODES_UNIT_01_STA_0.Ack_M43 := "M_ZERO";
END_REGION

REGION Network 36: M43-GEAR STAGE 3 (SIEMENS) / M43-SHIFT REDUCTION 3 (SIEMENS)
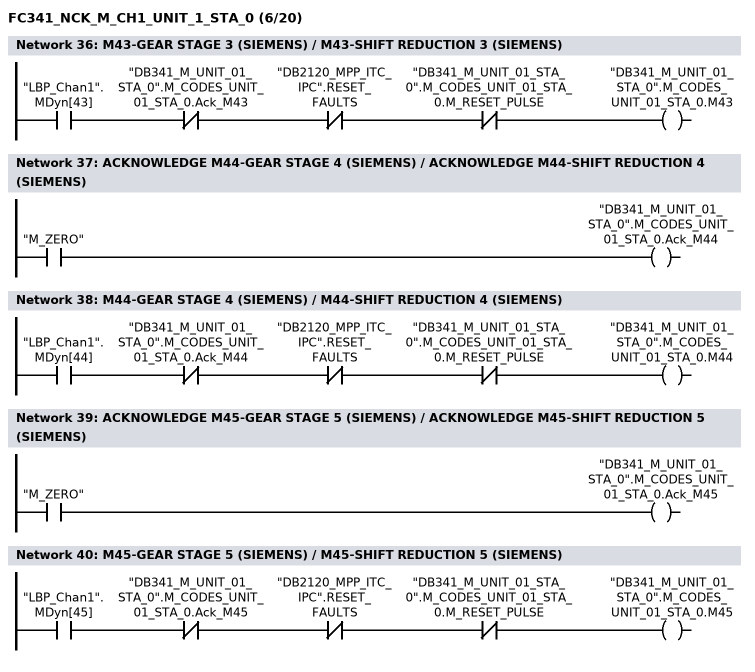
   RUNG wire#powerrail
      Contact( "LBP_Chan1".MDyn[43] )
      I_Contact( "DB341_M_UNIT_01_STA_0".M_CODES_UNIT_01_STA_0.Ack_M43 )
      I_Contact( "DB2120_MPP_ITC_IPC".RESET_FAULTS )
      I_Contact( "DB341_M_UNIT_01_STA_0".M_CODES_UNIT_01_STA_0.M_RESET_PULSE )
      Coil( "DB341_M_UNIT_01_STA_0".M_CODES_UNIT_01_STA_0.M43 )
   END_RUNG
   // the same network as SCL:
   "DB341_M_UNIT_01_STA_0".M_CODES_UNIT_01_STA_0.M43 := "LBP_Chan1".MDyn[43] AND NOT "DB341_M_UNIT_01_STA_0".M_CODES_UNIT_01_STA_0.Ack_M43 AND NOT "DB2120_MPP_ITC_IPC".RESET_FAULTS AND NOT "DB341_M_UNIT_01_STA_0".M_CODES_UNIT_01_STA_0.M_RESET_PULSE;
END_REGION

REGION Network 37: ACKNOWLEDGE M44-GEAR STAGE 4 (SIEMENS) / ACKNOWLEDGE M44-SHIFT REDUCTION 4 (SIEMENS)
   RUNG wire#powerrail
      Contact( "M_ZERO" )
      Coil( "DB341_M_UNIT_01_STA_0".M_CODES_UNIT_01_STA_0.Ack_M44 )
   END_RUNG
   // the same network as SCL:
   "DB341_M_UNIT_01_STA_0".M_CODES_UNIT_01_STA_0.Ack_M44 := "M_ZERO";
END_REGION

REGION Network 38: M44-GEAR STAGE 4 (SIEMENS) / M44-SHIFT REDUCTION 4 (SIEMENS)
   RUNG wire#powerrail
      Contact( "LBP_Chan1".MDyn[44] )
      I_Contact( "DB341_M_UNIT_01_STA_0".M_CODES_UNIT_01_STA_0.Ack_M44 )
      I_Contact( "DB2120_MPP_ITC_IPC".RESET_FAULTS )
      I_Contact( "DB341_M_UNIT_01_STA_0".M_CODES_UNIT_01_STA_0.M_RESET_PULSE )
      Coil( "DB341_M_UNIT_01_STA_0".M_CODES_UNIT_01_STA_0.M44 )
   END_RUNG
   // the same network as SCL:
   "DB341_M_UNIT_01_STA_0".M_CODES_UNIT_01_STA_0.M44 := "LBP_Chan1".MDyn[44] AND NOT "DB341_M_UNIT_01_STA_0".M_CODES_UNIT_01_STA_0.Ack_M44 AND NOT "DB2120_MPP_ITC_IPC".RESET_FAULTS AND NOT "DB341_M_UNIT_01_STA_0".M_CODES_UNIT_01_STA_0.M_RESET_PULSE;
END_REGION

REGION Network 39: ACKNOWLEDGE M45-GEAR STAGE 5 (SIEMENS) / ACKNOWLEDGE M45-SHIFT REDUCTION 5 (SIEMENS)
   RUNG wire#powerrail
      Contact( "M_ZERO" )
      Coil( "DB341_M_UNIT_01_STA_0".M_CODES_UNIT_01_STA_0.Ack_M45 )
   END_RUNG
   // the same network as SCL:
   "DB341_M_UNIT_01_STA_0".M_CODES_UNIT_01_STA_0.Ack_M45 := "M_ZERO";
END_REGION

REGION Network 40: M45-GEAR STAGE 5 (SIEMENS) / M45-SHIFT REDUCTION 5 (SIEMENS)
   RUNG wire#powerrail
      Contact( "LBP_Chan1".MDyn[45] )
      I_Contact( "DB341_M_UNIT_01_STA_0".M_CODES_UNIT_01_STA_0.Ack_M45 )
      I_Contact( "DB2120_MPP_ITC_IPC".RESET_FAULTS )
      I_Contact( "DB341_M_UNIT_01_STA_0".M_CODES_UNIT_01_STA_0.M_RESET_PULSE )
      Coil( "DB341_M_UNIT_01_STA_0".M_CODES_UNIT_01_STA_0.M45 )
   END_RUNG
   // the same network as SCL:
   "DB341_M_UNIT_01_STA_0".M_CODES_UNIT_01_STA_0.M45 := "LBP_Chan1".MDyn[45] AND NOT "DB341_M_UNIT_01_STA_0".M_CODES_UNIT_01_STA_0.Ack_M45 AND NOT "DB2120_MPP_ITC_IPC".RESET_FAULTS AND NOT "DB341_M_UNIT_01_STA_0".M_CODES_UNIT_01_STA_0.M_RESET_PULSE;
END_REGION

REGION Network 41: ACKNOWLEDGE M50-LOAD PART FROM ROBOT (READ IN DISABLE)
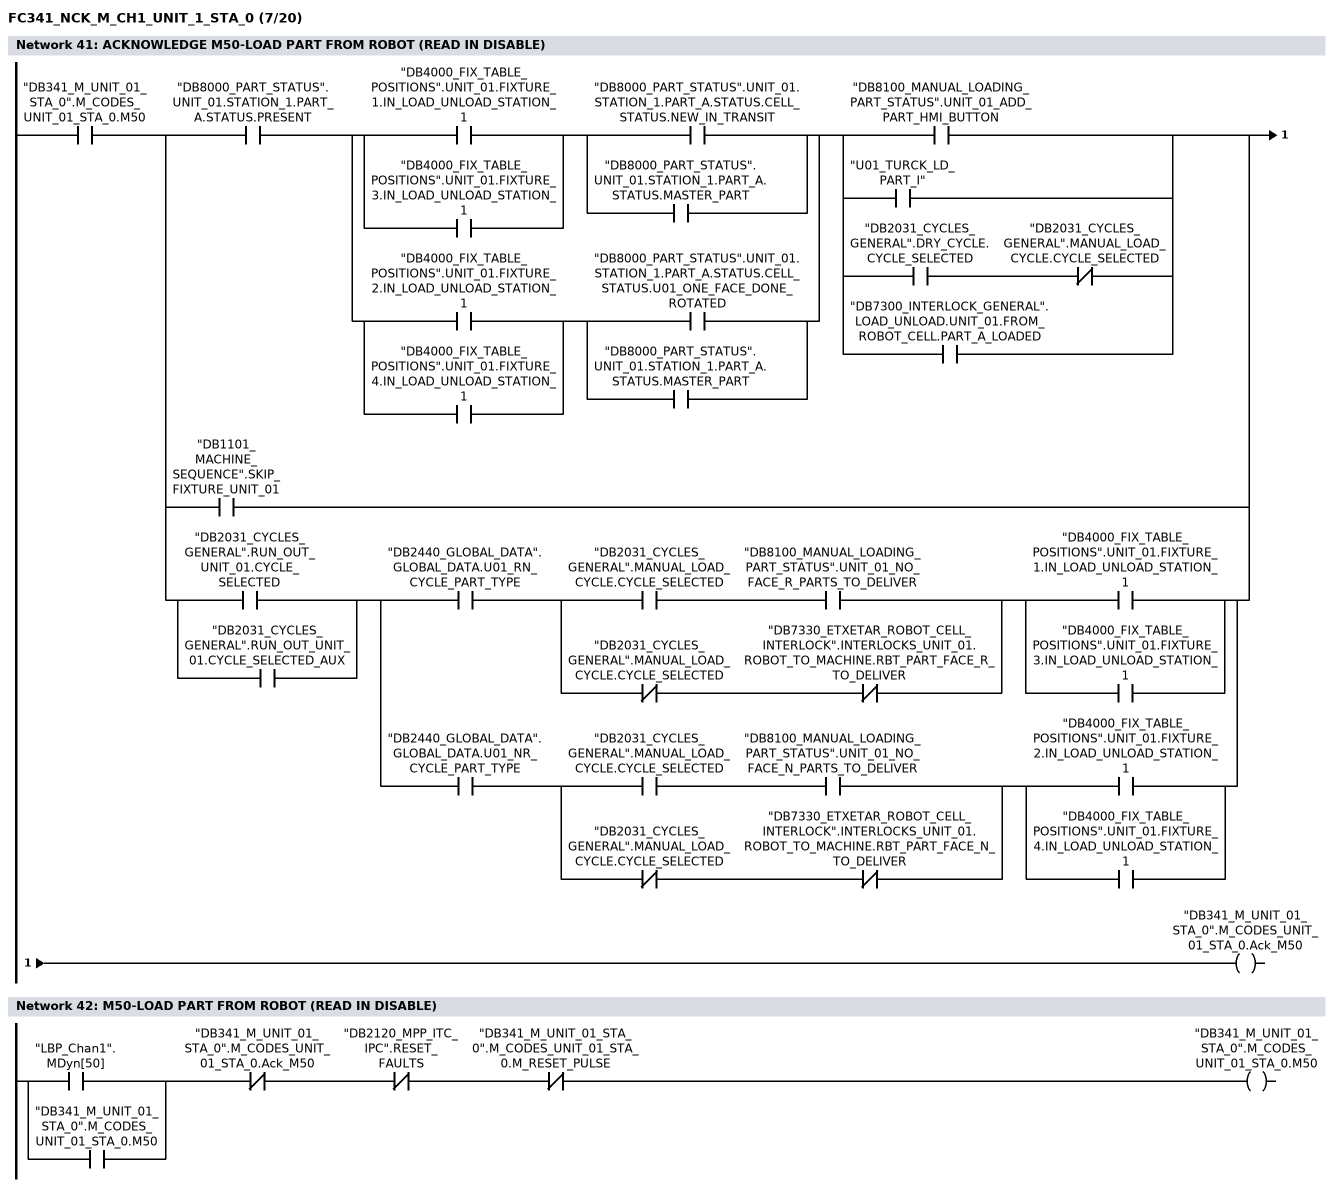
   RUNG wire#powerrail
      Contact( "DB341_M_UNIT_01_STA_0".M_CODES_UNIT_01_STA_0.M50 )
      wire#w1
      Contact( "DB8000_PART_STATUS".UNIT_01.STATION_1.PART_A.STATUS.PRESENT )
      wire#w2
      Contact( "DB4000_FIX_TABLE_POSITIONS".UNIT_01.FIXTURE_1.IN_LOAD_UNLOAD_STATION_1 )
      wire#w3
      Contact( "DB8000_PART_STATUS".UNIT_01.STATION_1.PART_A.STATUS.CELL_STATUS.NEW_IN_TRANSIT )
      wire#w4
      Contact( "DB8100_MANUAL_LOADING_PART_STATUS".UNIT_01_ADD_PART_HMI_BUTTON )
      wire#w6
      Coil( "DB341_M_UNIT_01_STA_0".M_CODES_UNIT_01_STA_0.Ack_M50 )
   END_RUNG
   RUNG wire#w2
      Contact( "DB4000_FIX_TABLE_POSITIONS".UNIT_01.FIXTURE_3.IN_LOAD_UNLOAD_STATION_1 )
   END_RUNG wire#w3
   RUNG wire#w3
      Contact( "DB8000_PART_STATUS".UNIT_01.STATION_1.PART_A.STATUS.MASTER_PART )
   END_RUNG wire#w4
   RUNG wire#w2
      Contact( "DB4000_FIX_TABLE_POSITIONS".UNIT_01.FIXTURE_2.IN_LOAD_UNLOAD_STATION_1 )
      wire#w5
      Contact( "DB8000_PART_STATUS".UNIT_01.STATION_1.PART_A.STATUS.CELL_STATUS.U01_ONE_FACE_DONE_ROTATED )
   END_RUNG wire#w4
   RUNG wire#w2
      Contact( "DB4000_FIX_TABLE_POSITIONS".UNIT_01.FIXTURE_4.IN_LOAD_UNLOAD_STATION_1 )
   END_RUNG wire#w5
   RUNG wire#w5
      Contact( "DB8000_PART_STATUS".UNIT_01.STATION_1.PART_A.STATUS.MASTER_PART )
   END_RUNG wire#w4
   RUNG wire#w4
      Contact( "U01_TURCK_LD_PART_I" )
   END_RUNG wire#w6
   RUNG wire#w4
      Contact( "DB2031_CYCLES_GENERAL".DRY_CYCLE.CYCLE_SELECTED )
      I_Contact( "DB2031_CYCLES_GENERAL".MANUAL_LOAD_CYCLE.CYCLE_SELECTED )
   END_RUNG wire#w6
   RUNG wire#w4
      Contact( "DB7300_INTERLOCK_GENERAL".LOAD_UNLOAD.UNIT_01.FROM_ROBOT_CELL.PART_A_LOADED )
   END_RUNG wire#w6
   RUNG wire#w1
      Contact( "DB1101_MACHINE_SEQUENCE".SKIP_FIXTURE_UNIT_01 )
   END_RUNG wire#w6
   RUNG wire#w1
      Contact( "DB2031_CYCLES_GENERAL".RUN_OUT_UNIT_01.CYCLE_SELECTED )
      wire#w7
      Contact( "DB2440_GLOBAL_DATA".GLOBAL_DATA.U01_RN_CYCLE_PART_TYPE )
      wire#w8
      Contact( "DB2031_CYCLES_GENERAL".MANUAL_LOAD_CYCLE.CYCLE_SELECTED )
      Contact( "DB8100_MANUAL_LOADING_PART_STATUS".UNIT_01_NO_FACE_R_PARTS_TO_DELIVER )
      wire#w9
      Contact( "DB4000_FIX_TABLE_POSITIONS".UNIT_01.FIXTURE_1.IN_LOAD_UNLOAD_STATION_1 )
   END_RUNG wire#w6
   RUNG wire#w1
      Contact( "DB2031_CYCLES_GENERAL".RUN_OUT_UNIT_01.CYCLE_SELECTED_AUX )
   END_RUNG wire#w7
   RUNG wire#w8
      I_Contact( "DB2031_CYCLES_GENERAL".MANUAL_LOAD_CYCLE.CYCLE_SELECTED )
      I_Contact( "DB7330_ETXETAR_ROBOT_CELL_INTERLOCK".INTERLOCKS_UNIT_01.ROBOT_TO_MACHINE.RBT_PART_FACE_R_TO_DELIVER )
   END_RUNG wire#w9
   RUNG wire#w9
      Contact( "DB4000_FIX_TABLE_POSITIONS".UNIT_01.FIXTURE_3.IN_LOAD_UNLOAD_STATION_1 )
   END_RUNG wire#w6
   RUNG wire#w7
      Contact( "DB2440_GLOBAL_DATA".GLOBAL_DATA.U01_NR_CYCLE_PART_TYPE )
      wire#w10
      Contact( "DB2031_CYCLES_GENERAL".MANUAL_LOAD_CYCLE.CYCLE_SELECTED )
      Contact( "DB8100_MANUAL_LOADING_PART_STATUS".UNIT_01_NO_FACE_N_PARTS_TO_DELIVER )
      wire#w11
      Contact( "DB4000_FIX_TABLE_POSITIONS".UNIT_01.FIXTURE_2.IN_LOAD_UNLOAD_STATION_1 )
   END_RUNG wire#w6
   RUNG wire#w10
      I_Contact( "DB2031_CYCLES_GENERAL".MANUAL_LOAD_CYCLE.CYCLE_SELECTED )
      I_Contact( "DB7330_ETXETAR_ROBOT_CELL_INTERLOCK".INTERLOCKS_UNIT_01.ROBOT_TO_MACHINE.RBT_PART_FACE_N_TO_DELIVER )
   END_RUNG wire#w11
   RUNG wire#w11
      Contact( "DB4000_FIX_TABLE_POSITIONS".UNIT_01.FIXTURE_4.IN_LOAD_UNLOAD_STATION_1 )
   END_RUNG wire#w6
   // the same network as SCL:
   "DB341_M_UNIT_01_STA_0".M_CODES_UNIT_01_STA_0.Ack_M50 := "DB341_M_UNIT_01_STA_0".M_CODES_UNIT_01_STA_0.M50 AND (("DB8000_PART_STATUS".UNIT_01.STATION_1.PART_A.STATUS.PRESENT AND ((("DB4000_FIX_TABLE_POSITIONS".UNIT_01.FIXTURE_1.IN_LOAD_UNLOAD_STATION_1 OR "DB4000_FIX_TABLE_POSITIONS".UNIT_01.FIXTURE_3.IN_LOAD_UNLOAD_STATION_1) AND ("DB8000_PART_STATUS".UNIT_01.STATION_1.PART_A.STATUS.CELL_STATUS.NEW_IN_TRANSIT OR "DB8000_PART_STATUS".UNIT_01.STATION_1.PART_A.STATUS.MASTER_PART)) OR (("DB4000_FIX_TABLE_POSITIONS".UNIT_01.FIXTURE_2.IN_LOAD_UNLOAD_STATION_1 OR "DB4000_FIX_TABLE_POSITIONS".UNIT_01.FIXTURE_4.IN_LOAD_UNLOAD_STATION_1) AND ("DB8000_PART_STATUS".UNIT_01.STATION_1.PART_A.STATUS.CELL_STATUS.U01_ONE_FACE_DONE_ROTATED OR "DB8000_PART_STATUS".UNIT_01.STATION_1.PART_A.STATUS.MASTER_PART))) AND ("DB8100_MANUAL_LOADING_PART_STATUS".UNIT_01_ADD_PART_HMI_BUTTON OR "U01_TURCK_LD_PART_I" OR ("DB2031_CYCLES_GENERAL".DRY_CYCLE.CYCLE_SELECTED AND NOT "DB2031_CYCLES_GENERAL".MANUAL_LOAD_CYCLE.CYCLE_SELECTED) OR "DB7300_INTERLOCK_GENERAL".LOAD_UNLOAD.UNIT_01.FROM_ROBOT_CELL.PART_A_LOADED)) OR "DB1101_MACHINE_SEQUENCE".SKIP_FIXTURE_UNIT_01 OR (("DB2031_CYCLES_GENERAL".RUN_OUT_UNIT_01.CYCLE_SELECTED OR "DB2031_CYCLES_GENERAL".RUN_OUT_UNIT_01.CYCLE_SELECTED_AUX) AND (("DB2440_GLOBAL_DATA".GLOBAL_DATA.U01_RN_CYCLE_PART_TYPE AND (("DB2031_CYCLES_GENERAL".MANUAL_LOAD_CYCLE.CYCLE_SELECTED AND "DB8100_MANUAL_LOADING_PART_STATUS".UNIT_01_NO_FACE_R_PARTS_TO_DELIVER) OR (NOT "DB2031_CYCLES_GENERAL".MANUAL_LOAD_CYCLE.CYCLE_SELECTED AND NOT "DB7330_ETXETAR_ROBOT_CELL_INTERLOCK".INTERLOCKS_UNIT_01.ROBOT_TO_MACHINE.RBT_PART_FACE_R_TO_DELIVER)) AND ("DB4000_FIX_TABLE_POSITIONS".UNIT_01.FIXTURE_1.IN_LOAD_UNLOAD_STATION_1 OR "DB4000_FIX_TABLE_POSITIONS".UNIT_01.FIXTURE_3.IN_LOAD_UNLOAD_STATION_1)) OR ("DB2440_GLOBAL_DATA".GLOBAL_DATA.U01_NR_CYCLE_PART_TYPE AND (("DB2031_CYCLES_GENERAL".MANUAL_LOAD_CYCLE.CYCLE_SELECTED AND "DB8100_MANUAL_LOADING_PART_STATUS".UNIT_01_NO_FACE_N_PARTS_TO_DELIVER) OR (NOT "DB2031_CYCLES_GENERAL".MANUAL_LOAD_CYCLE.CYCLE_SELECTED AND NOT "DB7330_ETXETAR_ROBOT_CELL_INTERLOCK".INTERLOCKS_UNIT_01.ROBOT_TO_MACHINE.RBT_PART_FACE_N_TO_DELIVER)) AND ("DB4000_FIX_TABLE_POSITIONS".UNIT_01.FIXTURE_2.IN_LOAD_UNLOAD_STATION_1 OR "DB4000_FIX_TABLE_POSITIONS".UNIT_01.FIXTURE_4.IN_LOAD_UNLOAD_STATION_1)))));
END_REGION

REGION Network 42: M50-LOAD PART FROM ROBOT (READ IN DISABLE)
   RUNG wire#powerrail
      Contact( "LBP_Chan1".MDyn[50] )
      wire#w1
      I_Contact( "DB341_M_UNIT_01_STA_0".M_CODES_UNIT_01_STA_0.Ack_M50 )
      I_Contact( "DB2120_MPP_ITC_IPC".RESET_FAULTS )
      I_Contact( "DB341_M_UNIT_01_STA_0".M_CODES_UNIT_01_STA_0.M_RESET_PULSE )
      Coil( "DB341_M_UNIT_01_STA_0".M_CODES_UNIT_01_STA_0.M50 )
   END_RUNG
   RUNG wire#powerrail
      Contact( "DB341_M_UNIT_01_STA_0".M_CODES_UNIT_01_STA_0.M50 )
   END_RUNG wire#w1
   // the same network as SCL:
   "DB341_M_UNIT_01_STA_0".M_CODES_UNIT_01_STA_0.M50 := ("LBP_Chan1".MDyn[50] OR "DB341_M_UNIT_01_STA_0".M_CODES_UNIT_01_STA_0.M50) AND NOT "DB341_M_UNIT_01_STA_0".M_CODES_UNIT_01_STA_0.Ack_M50 AND NOT "DB2120_MPP_ITC_IPC".RESET_FAULTS AND NOT "DB341_M_UNIT_01_STA_0".M_CODES_UNIT_01_STA_0.M_RESET_PULSE;
END_REGION

REGION Network 43: ACKNOWLEDGE M51-UNLOAD PART FROM ROBOT (READ IN DISABLE)
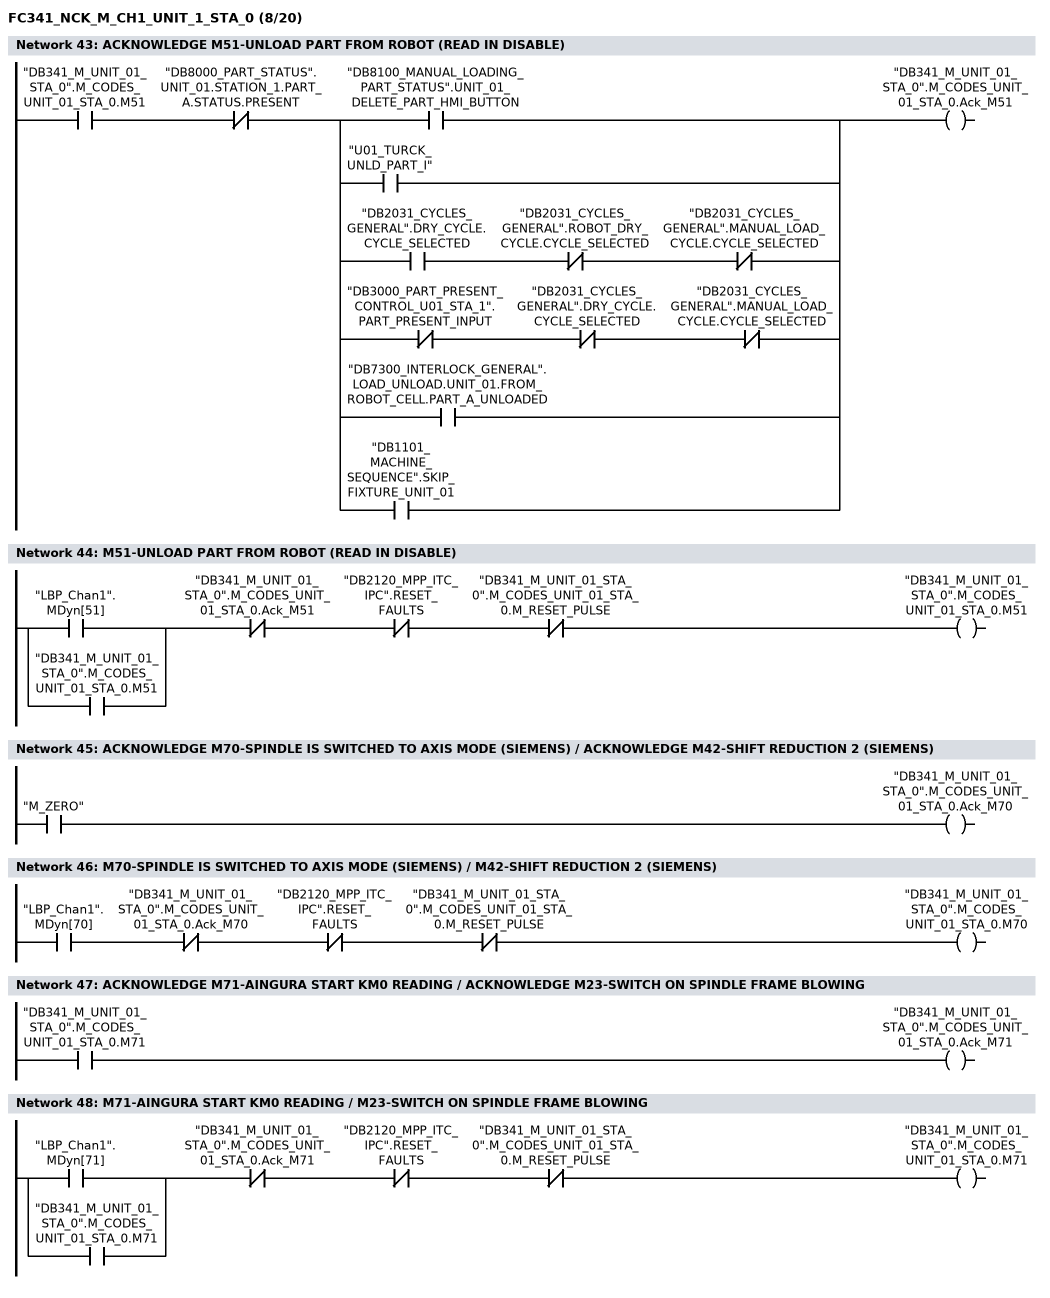
   RUNG wire#powerrail
      Contact( "DB341_M_UNIT_01_STA_0".M_CODES_UNIT_01_STA_0.M51 )
      I_Contact( "DB8000_PART_STATUS".UNIT_01.STATION_1.PART_A.STATUS.PRESENT )
      wire#w1
      Contact( "DB8100_MANUAL_LOADING_PART_STATUS".UNIT_01_DELETE_PART_HMI_BUTTON )
      wire#w2
      Coil( "DB341_M_UNIT_01_STA_0".M_CODES_UNIT_01_STA_0.Ack_M51 )
   END_RUNG
   RUNG wire#w1
      Contact( "U01_TURCK_UNLD_PART_I" )
   END_RUNG wire#w2
   RUNG wire#w1
      Contact( "DB2031_CYCLES_GENERAL".DRY_CYCLE.CYCLE_SELECTED )
      I_Contact( "DB2031_CYCLES_GENERAL".ROBOT_DRY_CYCLE.CYCLE_SELECTED )
      I_Contact( "DB2031_CYCLES_GENERAL".MANUAL_LOAD_CYCLE.CYCLE_SELECTED )
   END_RUNG wire#w2
   RUNG wire#w1
      I_Contact( "DB3000_PART_PRESENT_CONTROL_U01_STA_1".PART_PRESENT_INPUT )
      I_Contact( "DB2031_CYCLES_GENERAL".DRY_CYCLE.CYCLE_SELECTED )
      I_Contact( "DB2031_CYCLES_GENERAL".MANUAL_LOAD_CYCLE.CYCLE_SELECTED )
   END_RUNG wire#w2
   RUNG wire#w1
      Contact( "DB7300_INTERLOCK_GENERAL".LOAD_UNLOAD.UNIT_01.FROM_ROBOT_CELL.PART_A_UNLOADED )
   END_RUNG wire#w2
   RUNG wire#w1
      Contact( "DB1101_MACHINE_SEQUENCE".SKIP_FIXTURE_UNIT_01 )
   END_RUNG wire#w2
   // the same network as SCL:
   "DB341_M_UNIT_01_STA_0".M_CODES_UNIT_01_STA_0.Ack_M51 := "DB341_M_UNIT_01_STA_0".M_CODES_UNIT_01_STA_0.M51 AND NOT "DB8000_PART_STATUS".UNIT_01.STATION_1.PART_A.STATUS.PRESENT AND ("DB8100_MANUAL_LOADING_PART_STATUS".UNIT_01_DELETE_PART_HMI_BUTTON OR "U01_TURCK_UNLD_PART_I" OR ("DB2031_CYCLES_GENERAL".DRY_CYCLE.CYCLE_SELECTED AND NOT "DB2031_CYCLES_GENERAL".ROBOT_DRY_CYCLE.CYCLE_SELECTED AND NOT "DB2031_CYCLES_GENERAL".MANUAL_LOAD_CYCLE.CYCLE_SELECTED) OR (NOT "DB3000_PART_PRESENT_CONTROL_U01_STA_1".PART_PRESENT_INPUT AND NOT "DB2031_CYCLES_GENERAL".DRY_CYCLE.CYCLE_SELECTED AND NOT "DB2031_CYCLES_GENERAL".MANUAL_LOAD_CYCLE.CYCLE_SELECTED) OR "DB7300_INTERLOCK_GENERAL".LOAD_UNLOAD.UNIT_01.FROM_ROBOT_CELL.PART_A_UNLOADED OR "DB1101_MACHINE_SEQUENCE".SKIP_FIXTURE_UNIT_01);
END_REGION

REGION Network 44: M51-UNLOAD PART FROM ROBOT (READ IN DISABLE)
   RUNG wire#powerrail
      Contact( "LBP_Chan1".MDyn[51] )
      wire#w1
      I_Contact( "DB341_M_UNIT_01_STA_0".M_CODES_UNIT_01_STA_0.Ack_M51 )
      I_Contact( "DB2120_MPP_ITC_IPC".RESET_FAULTS )
      I_Contact( "DB341_M_UNIT_01_STA_0".M_CODES_UNIT_01_STA_0.M_RESET_PULSE )
      Coil( "DB341_M_UNIT_01_STA_0".M_CODES_UNIT_01_STA_0.M51 )
   END_RUNG
   RUNG wire#powerrail
      Contact( "DB341_M_UNIT_01_STA_0".M_CODES_UNIT_01_STA_0.M51 )
   END_RUNG wire#w1
   // the same network as SCL:
   "DB341_M_UNIT_01_STA_0".M_CODES_UNIT_01_STA_0.M51 := ("LBP_Chan1".MDyn[51] OR "DB341_M_UNIT_01_STA_0".M_CODES_UNIT_01_STA_0.M51) AND NOT "DB341_M_UNIT_01_STA_0".M_CODES_UNIT_01_STA_0.Ack_M51 AND NOT "DB2120_MPP_ITC_IPC".RESET_FAULTS AND NOT "DB341_M_UNIT_01_STA_0".M_CODES_UNIT_01_STA_0.M_RESET_PULSE;
END_REGION

REGION Network 45: ACKNOWLEDGE M70-SPINDLE IS SWITCHED TO AXIS MODE (SIEMENS) / ACKNOWLEDGE M42-SHIFT REDUCTION 2 (SIEMENS)
   RUNG wire#powerrail
      Contact( "M_ZERO" )
      Coil( "DB341_M_UNIT_01_STA_0".M_CODES_UNIT_01_STA_0.Ack_M70 )
   END_RUNG
   // the same network as SCL:
   "DB341_M_UNIT_01_STA_0".M_CODES_UNIT_01_STA_0.Ack_M70 := "M_ZERO";
END_REGION

REGION Network 46: M70-SPINDLE IS SWITCHED TO AXIS MODE (SIEMENS) / M42-SHIFT REDUCTION 2 (SIEMENS)
   RUNG wire#powerrail
      Contact( "LBP_Chan1".MDyn[70] )
      I_Contact( "DB341_M_UNIT_01_STA_0".M_CODES_UNIT_01_STA_0.Ack_M70 )
      I_Contact( "DB2120_MPP_ITC_IPC".RESET_FAULTS )
      I_Contact( "DB341_M_UNIT_01_STA_0".M_CODES_UNIT_01_STA_0.M_RESET_PULSE )
      Coil( "DB341_M_UNIT_01_STA_0".M_CODES_UNIT_01_STA_0.M70 )
   END_RUNG
   // the same network as SCL:
   "DB341_M_UNIT_01_STA_0".M_CODES_UNIT_01_STA_0.M70 := "LBP_Chan1".MDyn[70] AND NOT "DB341_M_UNIT_01_STA_0".M_CODES_UNIT_01_STA_0.Ack_M70 AND NOT "DB2120_MPP_ITC_IPC".RESET_FAULTS AND NOT "DB341_M_UNIT_01_STA_0".M_CODES_UNIT_01_STA_0.M_RESET_PULSE;
END_REGION

REGION Network 47: ACKNOWLEDGE M71-AINGURA START KM0 READING / ACKNOWLEDGE M23-SWITCH ON SPINDLE FRAME BLOWING
   RUNG wire#powerrail
      Contact( "DB341_M_UNIT_01_STA_0".M_CODES_UNIT_01_STA_0.M71 )
      Coil( "DB341_M_UNIT_01_STA_0".M_CODES_UNIT_01_STA_0.Ack_M71 )
   END_RUNG
   // the same network as SCL:
   "DB341_M_UNIT_01_STA_0".M_CODES_UNIT_01_STA_0.Ack_M71 := "DB341_M_UNIT_01_STA_0".M_CODES_UNIT_01_STA_0.M71;
END_REGION

REGION Network 48: M71-AINGURA START KM0 READING / M23-SWITCH ON SPINDLE FRAME BLOWING
   RUNG wire#powerrail
      Contact( "LBP_Chan1".MDyn[71] )
      wire#w1
      I_Contact( "DB341_M_UNIT_01_STA_0".M_CODES_UNIT_01_STA_0.Ack_M71 )
      I_Contact( "DB2120_MPP_ITC_IPC".RESET_FAULTS )
      I_Contact( "DB341_M_UNIT_01_STA_0".M_CODES_UNIT_01_STA_0.M_RESET_PULSE )
      Coil( "DB341_M_UNIT_01_STA_0".M_CODES_UNIT_01_STA_0.M71 )
   END_RUNG
   RUNG wire#powerrail
      Contact( "DB341_M_UNIT_01_STA_0".M_CODES_UNIT_01_STA_0.M71 )
   END_RUNG wire#w1
   // the same network as SCL:
   "DB341_M_UNIT_01_STA_0".M_CODES_UNIT_01_STA_0.M71 := ("LBP_Chan1".MDyn[71] OR "DB341_M_UNIT_01_STA_0".M_CODES_UNIT_01_STA_0.M71) AND NOT "DB341_M_UNIT_01_STA_0".M_CODES_UNIT_01_STA_0.Ack_M71 AND NOT "DB2120_MPP_ITC_IPC".RESET_FAULTS AND NOT "DB341_M_UNIT_01_STA_0".M_CODES_UNIT_01_STA_0.M_RESET_PULSE;
END_REGION

REGION Network 49: ACKNOWLEDGE M72-AINGURA STOP KM0 READING / ACKNOWLEDGE M23-SWITCH ON SPINDLE FRAME BLOWING
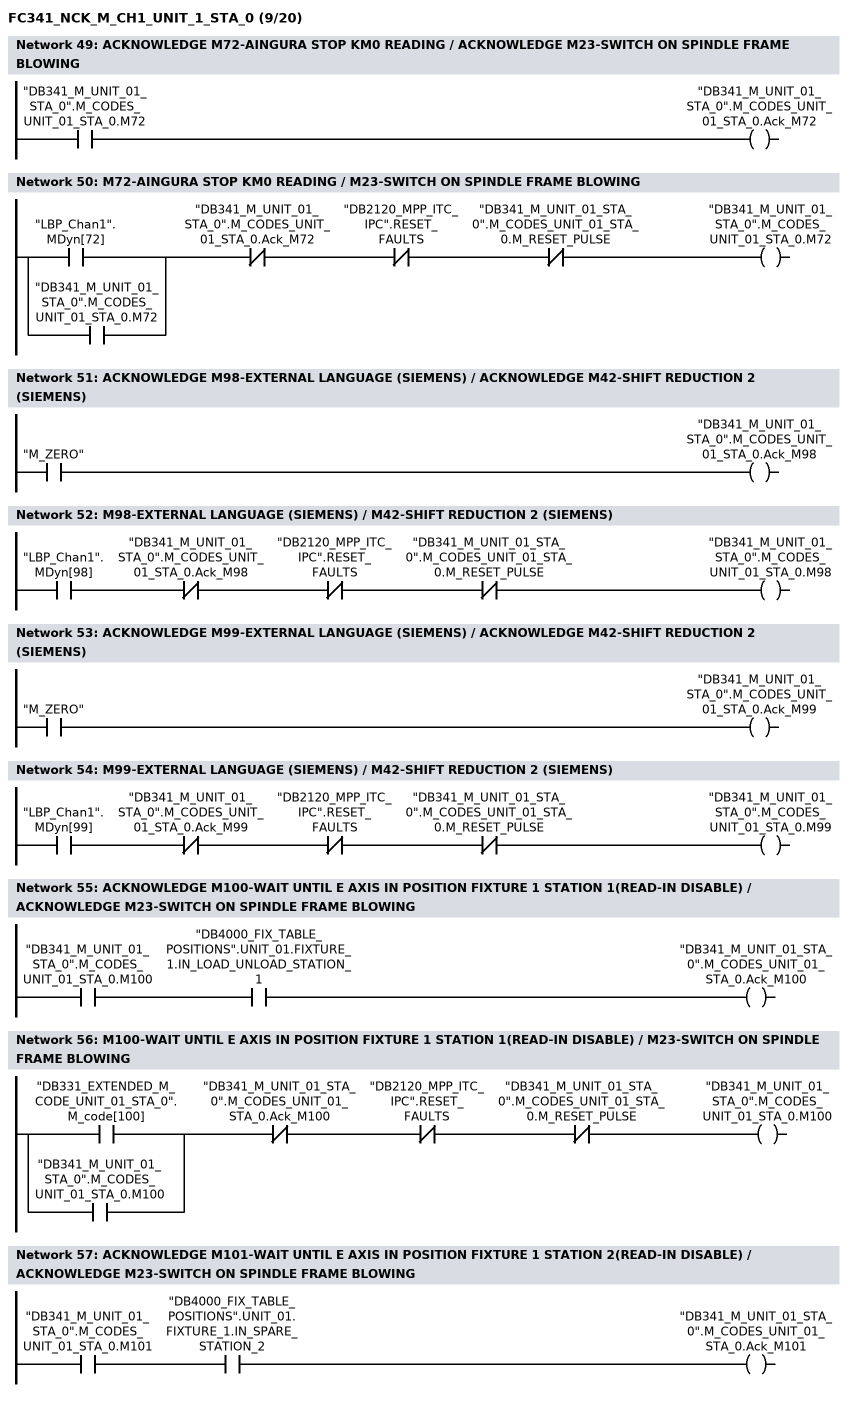
   RUNG wire#powerrail
      Contact( "DB341_M_UNIT_01_STA_0".M_CODES_UNIT_01_STA_0.M72 )
      Coil( "DB341_M_UNIT_01_STA_0".M_CODES_UNIT_01_STA_0.Ack_M72 )
   END_RUNG
   // the same network as SCL:
   "DB341_M_UNIT_01_STA_0".M_CODES_UNIT_01_STA_0.Ack_M72 := "DB341_M_UNIT_01_STA_0".M_CODES_UNIT_01_STA_0.M72;
END_REGION

REGION Network 50: M72-AINGURA STOP KM0 READING / M23-SWITCH ON SPINDLE FRAME BLOWING
   RUNG wire#powerrail
      Contact( "LBP_Chan1".MDyn[72] )
      wire#w1
      I_Contact( "DB341_M_UNIT_01_STA_0".M_CODES_UNIT_01_STA_0.Ack_M72 )
      I_Contact( "DB2120_MPP_ITC_IPC".RESET_FAULTS )
      I_Contact( "DB341_M_UNIT_01_STA_0".M_CODES_UNIT_01_STA_0.M_RESET_PULSE )
      Coil( "DB341_M_UNIT_01_STA_0".M_CODES_UNIT_01_STA_0.M72 )
   END_RUNG
   RUNG wire#powerrail
      Contact( "DB341_M_UNIT_01_STA_0".M_CODES_UNIT_01_STA_0.M72 )
   END_RUNG wire#w1
   // the same network as SCL:
   "DB341_M_UNIT_01_STA_0".M_CODES_UNIT_01_STA_0.M72 := ("LBP_Chan1".MDyn[72] OR "DB341_M_UNIT_01_STA_0".M_CODES_UNIT_01_STA_0.M72) AND NOT "DB341_M_UNIT_01_STA_0".M_CODES_UNIT_01_STA_0.Ack_M72 AND NOT "DB2120_MPP_ITC_IPC".RESET_FAULTS AND NOT "DB341_M_UNIT_01_STA_0".M_CODES_UNIT_01_STA_0.M_RESET_PULSE;
END_REGION

REGION Network 51: ACKNOWLEDGE M98-EXTERNAL LANGUAGE (SIEMENS) / ACKNOWLEDGE M42-SHIFT REDUCTION 2 (SIEMENS)
   RUNG wire#powerrail
      Contact( "M_ZERO" )
      Coil( "DB341_M_UNIT_01_STA_0".M_CODES_UNIT_01_STA_0.Ack_M98 )
   END_RUNG
   // the same network as SCL:
   "DB341_M_UNIT_01_STA_0".M_CODES_UNIT_01_STA_0.Ack_M98 := "M_ZERO";
END_REGION

REGION Network 52: M98-EXTERNAL LANGUAGE (SIEMENS) / M42-SHIFT REDUCTION 2 (SIEMENS)
   RUNG wire#powerrail
      Contact( "LBP_Chan1".MDyn[98] )
      I_Contact( "DB341_M_UNIT_01_STA_0".M_CODES_UNIT_01_STA_0.Ack_M98 )
      I_Contact( "DB2120_MPP_ITC_IPC".RESET_FAULTS )
      I_Contact( "DB341_M_UNIT_01_STA_0".M_CODES_UNIT_01_STA_0.M_RESET_PULSE )
      Coil( "DB341_M_UNIT_01_STA_0".M_CODES_UNIT_01_STA_0.M98 )
   END_RUNG
   // the same network as SCL:
   "DB341_M_UNIT_01_STA_0".M_CODES_UNIT_01_STA_0.M98 := "LBP_Chan1".MDyn[98] AND NOT "DB341_M_UNIT_01_STA_0".M_CODES_UNIT_01_STA_0.Ack_M98 AND NOT "DB2120_MPP_ITC_IPC".RESET_FAULTS AND NOT "DB341_M_UNIT_01_STA_0".M_CODES_UNIT_01_STA_0.M_RESET_PULSE;
END_REGION

REGION Network 53: ACKNOWLEDGE M99-EXTERNAL LANGUAGE (SIEMENS) / ACKNOWLEDGE M42-SHIFT REDUCTION 2 (SIEMENS)
   RUNG wire#powerrail
      Contact( "M_ZERO" )
      Coil( "DB341_M_UNIT_01_STA_0".M_CODES_UNIT_01_STA_0.Ack_M99 )
   END_RUNG
   // the same network as SCL:
   "DB341_M_UNIT_01_STA_0".M_CODES_UNIT_01_STA_0.Ack_M99 := "M_ZERO";
END_REGION

REGION Network 54: M99-EXTERNAL LANGUAGE (SIEMENS) / M42-SHIFT REDUCTION 2 (SIEMENS)
   RUNG wire#powerrail
      Contact( "LBP_Chan1".MDyn[99] )
      I_Contact( "DB341_M_UNIT_01_STA_0".M_CODES_UNIT_01_STA_0.Ack_M99 )
      I_Contact( "DB2120_MPP_ITC_IPC".RESET_FAULTS )
      I_Contact( "DB341_M_UNIT_01_STA_0".M_CODES_UNIT_01_STA_0.M_RESET_PULSE )
      Coil( "DB341_M_UNIT_01_STA_0".M_CODES_UNIT_01_STA_0.M99 )
   END_RUNG
   // the same network as SCL:
   "DB341_M_UNIT_01_STA_0".M_CODES_UNIT_01_STA_0.M99 := "LBP_Chan1".MDyn[99] AND NOT "DB341_M_UNIT_01_STA_0".M_CODES_UNIT_01_STA_0.Ack_M99 AND NOT "DB2120_MPP_ITC_IPC".RESET_FAULTS AND NOT "DB341_M_UNIT_01_STA_0".M_CODES_UNIT_01_STA_0.M_RESET_PULSE;
END_REGION

REGION Network 55: ACKNOWLEDGE M100-WAIT UNTIL E AXIS IN POSITION FIXTURE 1 STATION 1(READ-IN DISABLE) / ACKNOWLEDGE M23-SWITCH ON SPINDLE FRAME BLOWING
   RUNG wire#powerrail
      Contact( "DB341_M_UNIT_01_STA_0".M_CODES_UNIT_01_STA_0.M100 )
      Contact( "DB4000_FIX_TABLE_POSITIONS".UNIT_01.FIXTURE_1.IN_LOAD_UNLOAD_STATION_1 )
      Coil( "DB341_M_UNIT_01_STA_0".M_CODES_UNIT_01_STA_0.Ack_M100 )
   END_RUNG
   // the same network as SCL:
   "DB341_M_UNIT_01_STA_0".M_CODES_UNIT_01_STA_0.Ack_M100 := "DB341_M_UNIT_01_STA_0".M_CODES_UNIT_01_STA_0.M100 AND "DB4000_FIX_TABLE_POSITIONS".UNIT_01.FIXTURE_1.IN_LOAD_UNLOAD_STATION_1;
END_REGION

REGION Network 56: M100-WAIT UNTIL E AXIS IN POSITION FIXTURE 1 STATION 1(READ-IN DISABLE) / M23-SWITCH ON SPINDLE FRAME BLOWING
   RUNG wire#powerrail
      Contact( "DB331_EXTENDED_M_CODE_UNIT_01_STA_0".M_code[100] )
      wire#w1
      I_Contact( "DB341_M_UNIT_01_STA_0".M_CODES_UNIT_01_STA_0.Ack_M100 )
      I_Contact( "DB2120_MPP_ITC_IPC".RESET_FAULTS )
      I_Contact( "DB341_M_UNIT_01_STA_0".M_CODES_UNIT_01_STA_0.M_RESET_PULSE )
      Coil( "DB341_M_UNIT_01_STA_0".M_CODES_UNIT_01_STA_0.M100 )
   END_RUNG
   RUNG wire#powerrail
      Contact( "DB341_M_UNIT_01_STA_0".M_CODES_UNIT_01_STA_0.M100 )
   END_RUNG wire#w1
   // the same network as SCL:
   "DB341_M_UNIT_01_STA_0".M_CODES_UNIT_01_STA_0.M100 := ("DB331_EXTENDED_M_CODE_UNIT_01_STA_0".M_code[100] OR "DB341_M_UNIT_01_STA_0".M_CODES_UNIT_01_STA_0.M100) AND NOT "DB341_M_UNIT_01_STA_0".M_CODES_UNIT_01_STA_0.Ack_M100 AND NOT "DB2120_MPP_ITC_IPC".RESET_FAULTS AND NOT "DB341_M_UNIT_01_STA_0".M_CODES_UNIT_01_STA_0.M_RESET_PULSE;
END_REGION

REGION Network 57: ACKNOWLEDGE M101-WAIT UNTIL E AXIS IN POSITION FIXTURE 1 STATION 2(READ-IN DISABLE) / ACKNOWLEDGE M23-SWITCH ON SPINDLE FRAME BLOWING
   RUNG wire#powerrail
      Contact( "DB341_M_UNIT_01_STA_0".M_CODES_UNIT_01_STA_0.M101 )
      Contact( "DB4000_FIX_TABLE_POSITIONS".UNIT_01.FIXTURE_1.IN_SPARE_STATION_2 )
      Coil( "DB341_M_UNIT_01_STA_0".M_CODES_UNIT_01_STA_0.Ack_M101 )
   END_RUNG
   // the same network as SCL:
   "DB341_M_UNIT_01_STA_0".M_CODES_UNIT_01_STA_0.Ack_M101 := "DB341_M_UNIT_01_STA_0".M_CODES_UNIT_01_STA_0.M101 AND "DB4000_FIX_TABLE_POSITIONS".UNIT_01.FIXTURE_1.IN_SPARE_STATION_2;
END_REGION

REGION Network 58: M101-WAIT UNTIL E AXIS IN POSITION FIXTURE 1 STATION 2(READ-IN DISABLE) / M23-SWITCH ON SPINDLE FRAME BLOWING
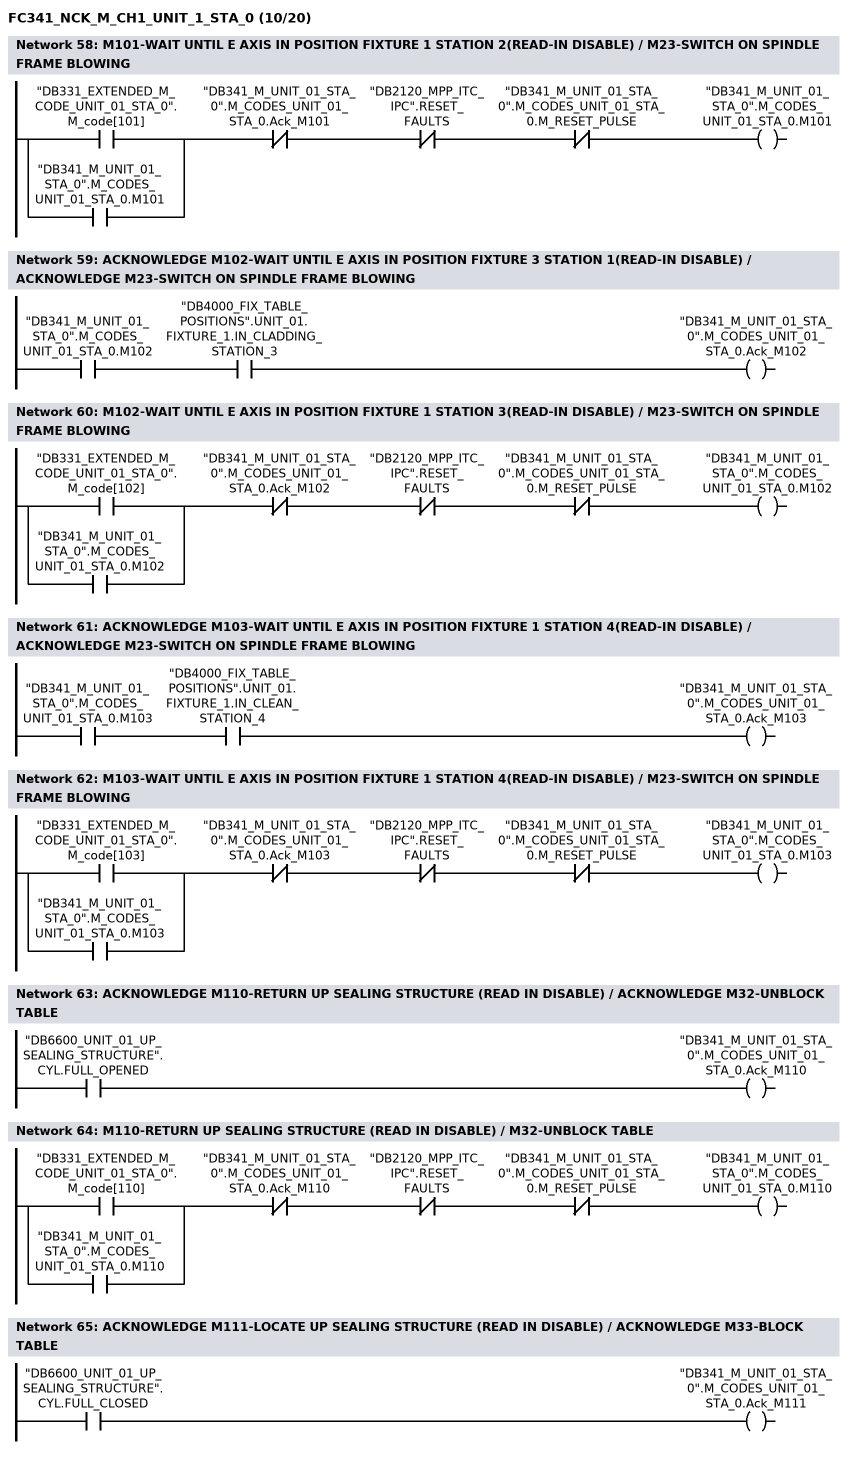
   RUNG wire#powerrail
      Contact( "DB331_EXTENDED_M_CODE_UNIT_01_STA_0".M_code[101] )
      wire#w1
      I_Contact( "DB341_M_UNIT_01_STA_0".M_CODES_UNIT_01_STA_0.Ack_M101 )
      I_Contact( "DB2120_MPP_ITC_IPC".RESET_FAULTS )
      I_Contact( "DB341_M_UNIT_01_STA_0".M_CODES_UNIT_01_STA_0.M_RESET_PULSE )
      Coil( "DB341_M_UNIT_01_STA_0".M_CODES_UNIT_01_STA_0.M101 )
   END_RUNG
   RUNG wire#powerrail
      Contact( "DB341_M_UNIT_01_STA_0".M_CODES_UNIT_01_STA_0.M101 )
   END_RUNG wire#w1
   // the same network as SCL:
   "DB341_M_UNIT_01_STA_0".M_CODES_UNIT_01_STA_0.M101 := ("DB331_EXTENDED_M_CODE_UNIT_01_STA_0".M_code[101] OR "DB341_M_UNIT_01_STA_0".M_CODES_UNIT_01_STA_0.M101) AND NOT "DB341_M_UNIT_01_STA_0".M_CODES_UNIT_01_STA_0.Ack_M101 AND NOT "DB2120_MPP_ITC_IPC".RESET_FAULTS AND NOT "DB341_M_UNIT_01_STA_0".M_CODES_UNIT_01_STA_0.M_RESET_PULSE;
END_REGION

REGION Network 59: ACKNOWLEDGE M102-WAIT UNTIL E AXIS IN POSITION FIXTURE 3 STATION 1(READ-IN DISABLE) / ACKNOWLEDGE M23-SWITCH ON SPINDLE FRAME BLOWING
   RUNG wire#powerrail
      Contact( "DB341_M_UNIT_01_STA_0".M_CODES_UNIT_01_STA_0.M102 )
      Contact( "DB4000_FIX_TABLE_POSITIONS".UNIT_01.FIXTURE_1.IN_CLADDING_STATION_3 )
      Coil( "DB341_M_UNIT_01_STA_0".M_CODES_UNIT_01_STA_0.Ack_M102 )
   END_RUNG
   // the same network as SCL:
   "DB341_M_UNIT_01_STA_0".M_CODES_UNIT_01_STA_0.Ack_M102 := "DB341_M_UNIT_01_STA_0".M_CODES_UNIT_01_STA_0.M102 AND "DB4000_FIX_TABLE_POSITIONS".UNIT_01.FIXTURE_1.IN_CLADDING_STATION_3;
END_REGION

REGION Network 60: M102-WAIT UNTIL E AXIS IN POSITION FIXTURE 1 STATION 3(READ-IN DISABLE) / M23-SWITCH ON SPINDLE FRAME BLOWING
   RUNG wire#powerrail
      Contact( "DB331_EXTENDED_M_CODE_UNIT_01_STA_0".M_code[102] )
      wire#w1
      I_Contact( "DB341_M_UNIT_01_STA_0".M_CODES_UNIT_01_STA_0.Ack_M102 )
      I_Contact( "DB2120_MPP_ITC_IPC".RESET_FAULTS )
      I_Contact( "DB341_M_UNIT_01_STA_0".M_CODES_UNIT_01_STA_0.M_RESET_PULSE )
      Coil( "DB341_M_UNIT_01_STA_0".M_CODES_UNIT_01_STA_0.M102 )
   END_RUNG
   RUNG wire#powerrail
      Contact( "DB341_M_UNIT_01_STA_0".M_CODES_UNIT_01_STA_0.M102 )
   END_RUNG wire#w1
   // the same network as SCL:
   "DB341_M_UNIT_01_STA_0".M_CODES_UNIT_01_STA_0.M102 := ("DB331_EXTENDED_M_CODE_UNIT_01_STA_0".M_code[102] OR "DB341_M_UNIT_01_STA_0".M_CODES_UNIT_01_STA_0.M102) AND NOT "DB341_M_UNIT_01_STA_0".M_CODES_UNIT_01_STA_0.Ack_M102 AND NOT "DB2120_MPP_ITC_IPC".RESET_FAULTS AND NOT "DB341_M_UNIT_01_STA_0".M_CODES_UNIT_01_STA_0.M_RESET_PULSE;
END_REGION

REGION Network 61: ACKNOWLEDGE M103-WAIT UNTIL E AXIS IN POSITION FIXTURE 1 STATION 4(READ-IN DISABLE) / ACKNOWLEDGE M23-SWITCH ON SPINDLE FRAME BLOWING
   RUNG wire#powerrail
      Contact( "DB341_M_UNIT_01_STA_0".M_CODES_UNIT_01_STA_0.M103 )
      Contact( "DB4000_FIX_TABLE_POSITIONS".UNIT_01.FIXTURE_1.IN_CLEAN_STATION_4 )
      Coil( "DB341_M_UNIT_01_STA_0".M_CODES_UNIT_01_STA_0.Ack_M103 )
   END_RUNG
   // the same network as SCL:
   "DB341_M_UNIT_01_STA_0".M_CODES_UNIT_01_STA_0.Ack_M103 := "DB341_M_UNIT_01_STA_0".M_CODES_UNIT_01_STA_0.M103 AND "DB4000_FIX_TABLE_POSITIONS".UNIT_01.FIXTURE_1.IN_CLEAN_STATION_4;
END_REGION

REGION Network 62: M103-WAIT UNTIL E AXIS IN POSITION FIXTURE 1 STATION 4(READ-IN DISABLE) / M23-SWITCH ON SPINDLE FRAME BLOWING
   RUNG wire#powerrail
      Contact( "DB331_EXTENDED_M_CODE_UNIT_01_STA_0".M_code[103] )
      wire#w1
      I_Contact( "DB341_M_UNIT_01_STA_0".M_CODES_UNIT_01_STA_0.Ack_M103 )
      I_Contact( "DB2120_MPP_ITC_IPC".RESET_FAULTS )
      I_Contact( "DB341_M_UNIT_01_STA_0".M_CODES_UNIT_01_STA_0.M_RESET_PULSE )
      Coil( "DB341_M_UNIT_01_STA_0".M_CODES_UNIT_01_STA_0.M103 )
   END_RUNG
   RUNG wire#powerrail
      Contact( "DB341_M_UNIT_01_STA_0".M_CODES_UNIT_01_STA_0.M103 )
   END_RUNG wire#w1
   // the same network as SCL:
   "DB341_M_UNIT_01_STA_0".M_CODES_UNIT_01_STA_0.M103 := ("DB331_EXTENDED_M_CODE_UNIT_01_STA_0".M_code[103] OR "DB341_M_UNIT_01_STA_0".M_CODES_UNIT_01_STA_0.M103) AND NOT "DB341_M_UNIT_01_STA_0".M_CODES_UNIT_01_STA_0.Ack_M103 AND NOT "DB2120_MPP_ITC_IPC".RESET_FAULTS AND NOT "DB341_M_UNIT_01_STA_0".M_CODES_UNIT_01_STA_0.M_RESET_PULSE;
END_REGION

REGION Network 63: ACKNOWLEDGE M110-RETURN UP SEALING STRUCTURE (READ IN DISABLE) / ACKNOWLEDGE M32-UNBLOCK TABLE
   RUNG wire#powerrail
      Contact( "DB6600_UNIT_01_UP_SEALING_STRUCTURE".CYL.FULL_OPENED )
      Coil( "DB341_M_UNIT_01_STA_0".M_CODES_UNIT_01_STA_0.Ack_M110 )
   END_RUNG
   // the same network as SCL:
   "DB341_M_UNIT_01_STA_0".M_CODES_UNIT_01_STA_0.Ack_M110 := "DB6600_UNIT_01_UP_SEALING_STRUCTURE".CYL.FULL_OPENED;
END_REGION

REGION Network 64: M110-RETURN UP SEALING STRUCTURE (READ IN DISABLE) / M32-UNBLOCK TABLE
   RUNG wire#powerrail
      Contact( "DB331_EXTENDED_M_CODE_UNIT_01_STA_0".M_code[110] )
      wire#w1
      I_Contact( "DB341_M_UNIT_01_STA_0".M_CODES_UNIT_01_STA_0.Ack_M110 )
      I_Contact( "DB2120_MPP_ITC_IPC".RESET_FAULTS )
      I_Contact( "DB341_M_UNIT_01_STA_0".M_CODES_UNIT_01_STA_0.M_RESET_PULSE )
      Coil( "DB341_M_UNIT_01_STA_0".M_CODES_UNIT_01_STA_0.M110 )
   END_RUNG
   RUNG wire#powerrail
      Contact( "DB341_M_UNIT_01_STA_0".M_CODES_UNIT_01_STA_0.M110 )
   END_RUNG wire#w1
   // the same network as SCL:
   "DB341_M_UNIT_01_STA_0".M_CODES_UNIT_01_STA_0.M110 := ("DB331_EXTENDED_M_CODE_UNIT_01_STA_0".M_code[110] OR "DB341_M_UNIT_01_STA_0".M_CODES_UNIT_01_STA_0.M110) AND NOT "DB341_M_UNIT_01_STA_0".M_CODES_UNIT_01_STA_0.Ack_M110 AND NOT "DB2120_MPP_ITC_IPC".RESET_FAULTS AND NOT "DB341_M_UNIT_01_STA_0".M_CODES_UNIT_01_STA_0.M_RESET_PULSE;
END_REGION

REGION Network 65: ACKNOWLEDGE M111-LOCATE UP SEALING STRUCTURE (READ IN DISABLE) / ACKNOWLEDGE M33-BLOCK TABLE
   RUNG wire#powerrail
      Contact( "DB6600_UNIT_01_UP_SEALING_STRUCTURE".CYL.FULL_CLOSED )
      Coil( "DB341_M_UNIT_01_STA_0".M_CODES_UNIT_01_STA_0.Ack_M111 )
   END_RUNG
   // the same network as SCL:
   "DB341_M_UNIT_01_STA_0".M_CODES_UNIT_01_STA_0.Ack_M111 := "DB6600_UNIT_01_UP_SEALING_STRUCTURE".CYL.FULL_CLOSED;
END_REGION

REGION Network 66: M111-LOCATE UP SEALING STRUCTURE (READ IN DISABLE) / M33-BLOCK TABLE
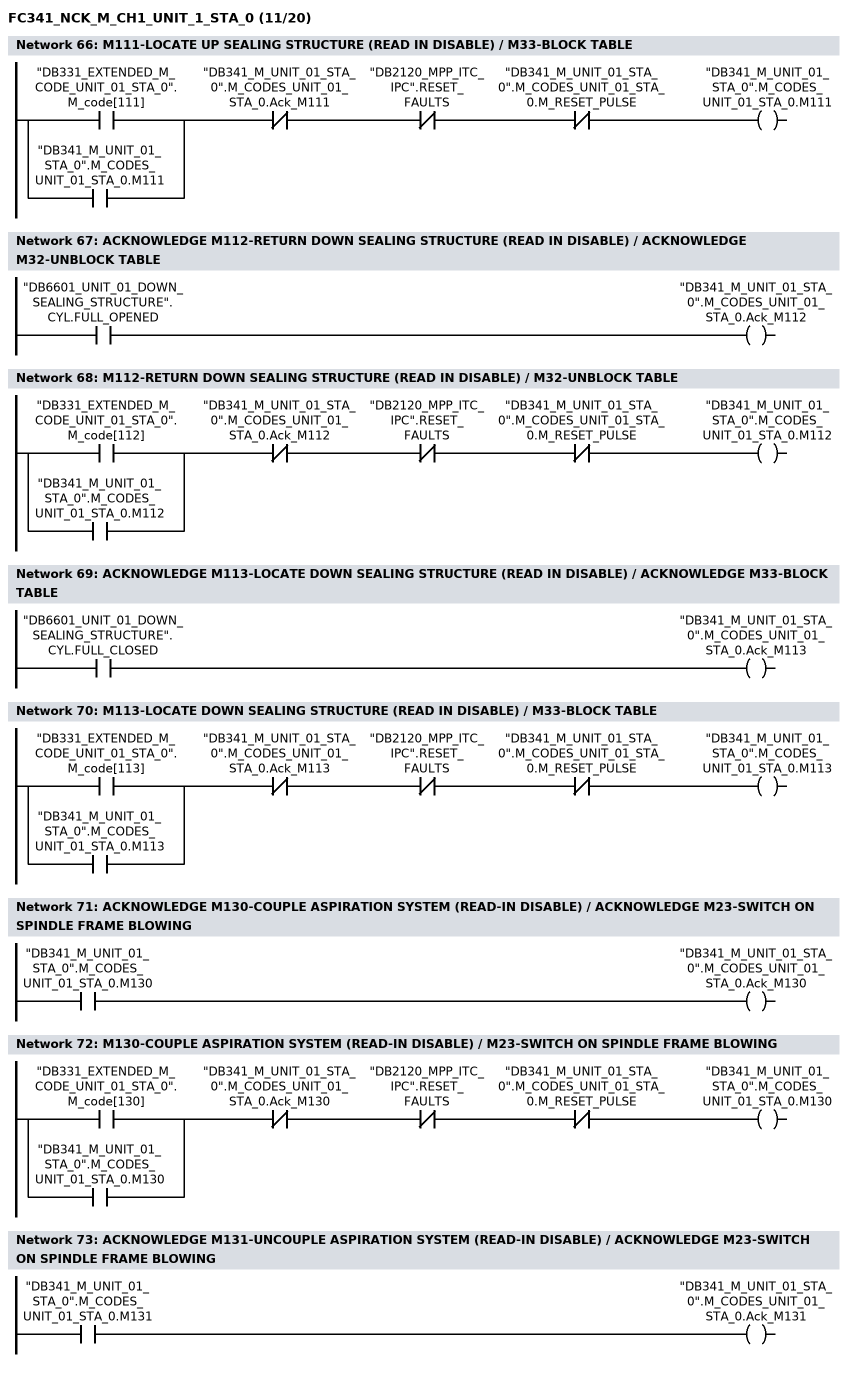
   RUNG wire#powerrail
      Contact( "DB331_EXTENDED_M_CODE_UNIT_01_STA_0".M_code[111] )
      wire#w1
      I_Contact( "DB341_M_UNIT_01_STA_0".M_CODES_UNIT_01_STA_0.Ack_M111 )
      I_Contact( "DB2120_MPP_ITC_IPC".RESET_FAULTS )
      I_Contact( "DB341_M_UNIT_01_STA_0".M_CODES_UNIT_01_STA_0.M_RESET_PULSE )
      Coil( "DB341_M_UNIT_01_STA_0".M_CODES_UNIT_01_STA_0.M111 )
   END_RUNG
   RUNG wire#powerrail
      Contact( "DB341_M_UNIT_01_STA_0".M_CODES_UNIT_01_STA_0.M111 )
   END_RUNG wire#w1
   // the same network as SCL:
   "DB341_M_UNIT_01_STA_0".M_CODES_UNIT_01_STA_0.M111 := ("DB331_EXTENDED_M_CODE_UNIT_01_STA_0".M_code[111] OR "DB341_M_UNIT_01_STA_0".M_CODES_UNIT_01_STA_0.M111) AND NOT "DB341_M_UNIT_01_STA_0".M_CODES_UNIT_01_STA_0.Ack_M111 AND NOT "DB2120_MPP_ITC_IPC".RESET_FAULTS AND NOT "DB341_M_UNIT_01_STA_0".M_CODES_UNIT_01_STA_0.M_RESET_PULSE;
END_REGION

REGION Network 67: ACKNOWLEDGE M112-RETURN DOWN SEALING STRUCTURE (READ IN DISABLE) / ACKNOWLEDGE M32-UNBLOCK TABLE
   RUNG wire#powerrail
      Contact( "DB6601_UNIT_01_DOWN_SEALING_STRUCTURE".CYL.FULL_OPENED )
      Coil( "DB341_M_UNIT_01_STA_0".M_CODES_UNIT_01_STA_0.Ack_M112 )
   END_RUNG
   // the same network as SCL:
   "DB341_M_UNIT_01_STA_0".M_CODES_UNIT_01_STA_0.Ack_M112 := "DB6601_UNIT_01_DOWN_SEALING_STRUCTURE".CYL.FULL_OPENED;
END_REGION

REGION Network 68: M112-RETURN DOWN SEALING STRUCTURE (READ IN DISABLE) / M32-UNBLOCK TABLE
   RUNG wire#powerrail
      Contact( "DB331_EXTENDED_M_CODE_UNIT_01_STA_0".M_code[112] )
      wire#w1
      I_Contact( "DB341_M_UNIT_01_STA_0".M_CODES_UNIT_01_STA_0.Ack_M112 )
      I_Contact( "DB2120_MPP_ITC_IPC".RESET_FAULTS )
      I_Contact( "DB341_M_UNIT_01_STA_0".M_CODES_UNIT_01_STA_0.M_RESET_PULSE )
      Coil( "DB341_M_UNIT_01_STA_0".M_CODES_UNIT_01_STA_0.M112 )
   END_RUNG
   RUNG wire#powerrail
      Contact( "DB341_M_UNIT_01_STA_0".M_CODES_UNIT_01_STA_0.M112 )
   END_RUNG wire#w1
   // the same network as SCL:
   "DB341_M_UNIT_01_STA_0".M_CODES_UNIT_01_STA_0.M112 := ("DB331_EXTENDED_M_CODE_UNIT_01_STA_0".M_code[112] OR "DB341_M_UNIT_01_STA_0".M_CODES_UNIT_01_STA_0.M112) AND NOT "DB341_M_UNIT_01_STA_0".M_CODES_UNIT_01_STA_0.Ack_M112 AND NOT "DB2120_MPP_ITC_IPC".RESET_FAULTS AND NOT "DB341_M_UNIT_01_STA_0".M_CODES_UNIT_01_STA_0.M_RESET_PULSE;
END_REGION

REGION Network 69: ACKNOWLEDGE M113-LOCATE DOWN SEALING STRUCTURE (READ IN DISABLE) / ACKNOWLEDGE M33-BLOCK TABLE
   RUNG wire#powerrail
      Contact( "DB6601_UNIT_01_DOWN_SEALING_STRUCTURE".CYL.FULL_CLOSED )
      Coil( "DB341_M_UNIT_01_STA_0".M_CODES_UNIT_01_STA_0.Ack_M113 )
   END_RUNG
   // the same network as SCL:
   "DB341_M_UNIT_01_STA_0".M_CODES_UNIT_01_STA_0.Ack_M113 := "DB6601_UNIT_01_DOWN_SEALING_STRUCTURE".CYL.FULL_CLOSED;
END_REGION

REGION Network 70: M113-LOCATE DOWN SEALING STRUCTURE (READ IN DISABLE) / M33-BLOCK TABLE
   RUNG wire#powerrail
      Contact( "DB331_EXTENDED_M_CODE_UNIT_01_STA_0".M_code[113] )
      wire#w1
      I_Contact( "DB341_M_UNIT_01_STA_0".M_CODES_UNIT_01_STA_0.Ack_M113 )
      I_Contact( "DB2120_MPP_ITC_IPC".RESET_FAULTS )
      I_Contact( "DB341_M_UNIT_01_STA_0".M_CODES_UNIT_01_STA_0.M_RESET_PULSE )
      Coil( "DB341_M_UNIT_01_STA_0".M_CODES_UNIT_01_STA_0.M113 )
   END_RUNG
   RUNG wire#powerrail
      Contact( "DB341_M_UNIT_01_STA_0".M_CODES_UNIT_01_STA_0.M113 )
   END_RUNG wire#w1
   // the same network as SCL:
   "DB341_M_UNIT_01_STA_0".M_CODES_UNIT_01_STA_0.M113 := ("DB331_EXTENDED_M_CODE_UNIT_01_STA_0".M_code[113] OR "DB341_M_UNIT_01_STA_0".M_CODES_UNIT_01_STA_0.M113) AND NOT "DB341_M_UNIT_01_STA_0".M_CODES_UNIT_01_STA_0.Ack_M113 AND NOT "DB2120_MPP_ITC_IPC".RESET_FAULTS AND NOT "DB341_M_UNIT_01_STA_0".M_CODES_UNIT_01_STA_0.M_RESET_PULSE;
END_REGION

REGION Network 71: ACKNOWLEDGE M130-COUPLE ASPIRATION SYSTEM (READ-IN DISABLE) / ACKNOWLEDGE M23-SWITCH ON SPINDLE FRAME BLOWING
   RUNG wire#powerrail
      Contact( "DB341_M_UNIT_01_STA_0".M_CODES_UNIT_01_STA_0.M130 )
      Coil( "DB341_M_UNIT_01_STA_0".M_CODES_UNIT_01_STA_0.Ack_M130 )
   END_RUNG
   // the same network as SCL:
   "DB341_M_UNIT_01_STA_0".M_CODES_UNIT_01_STA_0.Ack_M130 := "DB341_M_UNIT_01_STA_0".M_CODES_UNIT_01_STA_0.M130;
END_REGION

REGION Network 72: M130-COUPLE ASPIRATION SYSTEM (READ-IN DISABLE) / M23-SWITCH ON SPINDLE FRAME BLOWING
   RUNG wire#powerrail
      Contact( "DB331_EXTENDED_M_CODE_UNIT_01_STA_0".M_code[130] )
      wire#w1
      I_Contact( "DB341_M_UNIT_01_STA_0".M_CODES_UNIT_01_STA_0.Ack_M130 )
      I_Contact( "DB2120_MPP_ITC_IPC".RESET_FAULTS )
      I_Contact( "DB341_M_UNIT_01_STA_0".M_CODES_UNIT_01_STA_0.M_RESET_PULSE )
      Coil( "DB341_M_UNIT_01_STA_0".M_CODES_UNIT_01_STA_0.M130 )
   END_RUNG
   RUNG wire#powerrail
      Contact( "DB341_M_UNIT_01_STA_0".M_CODES_UNIT_01_STA_0.M130 )
   END_RUNG wire#w1
   // the same network as SCL:
   "DB341_M_UNIT_01_STA_0".M_CODES_UNIT_01_STA_0.M130 := ("DB331_EXTENDED_M_CODE_UNIT_01_STA_0".M_code[130] OR "DB341_M_UNIT_01_STA_0".M_CODES_UNIT_01_STA_0.M130) AND NOT "DB341_M_UNIT_01_STA_0".M_CODES_UNIT_01_STA_0.Ack_M130 AND NOT "DB2120_MPP_ITC_IPC".RESET_FAULTS AND NOT "DB341_M_UNIT_01_STA_0".M_CODES_UNIT_01_STA_0.M_RESET_PULSE;
END_REGION

REGION Network 73: ACKNOWLEDGE M131-UNCOUPLE ASPIRATION SYSTEM (READ-IN DISABLE) / ACKNOWLEDGE M23-SWITCH ON SPINDLE FRAME BLOWING
   RUNG wire#powerrail
      Contact( "DB341_M_UNIT_01_STA_0".M_CODES_UNIT_01_STA_0.M131 )
      Coil( "DB341_M_UNIT_01_STA_0".M_CODES_UNIT_01_STA_0.Ack_M131 )
   END_RUNG
   // the same network as SCL:
   "DB341_M_UNIT_01_STA_0".M_CODES_UNIT_01_STA_0.Ack_M131 := "DB341_M_UNIT_01_STA_0".M_CODES_UNIT_01_STA_0.M131;
END_REGION

REGION Network 74: M131-UNCOUPLE ASPIRATION SYSTEM (READ-IN DISABLE) / M23-SWITCH ON SPINDLE FRAME BLOWING
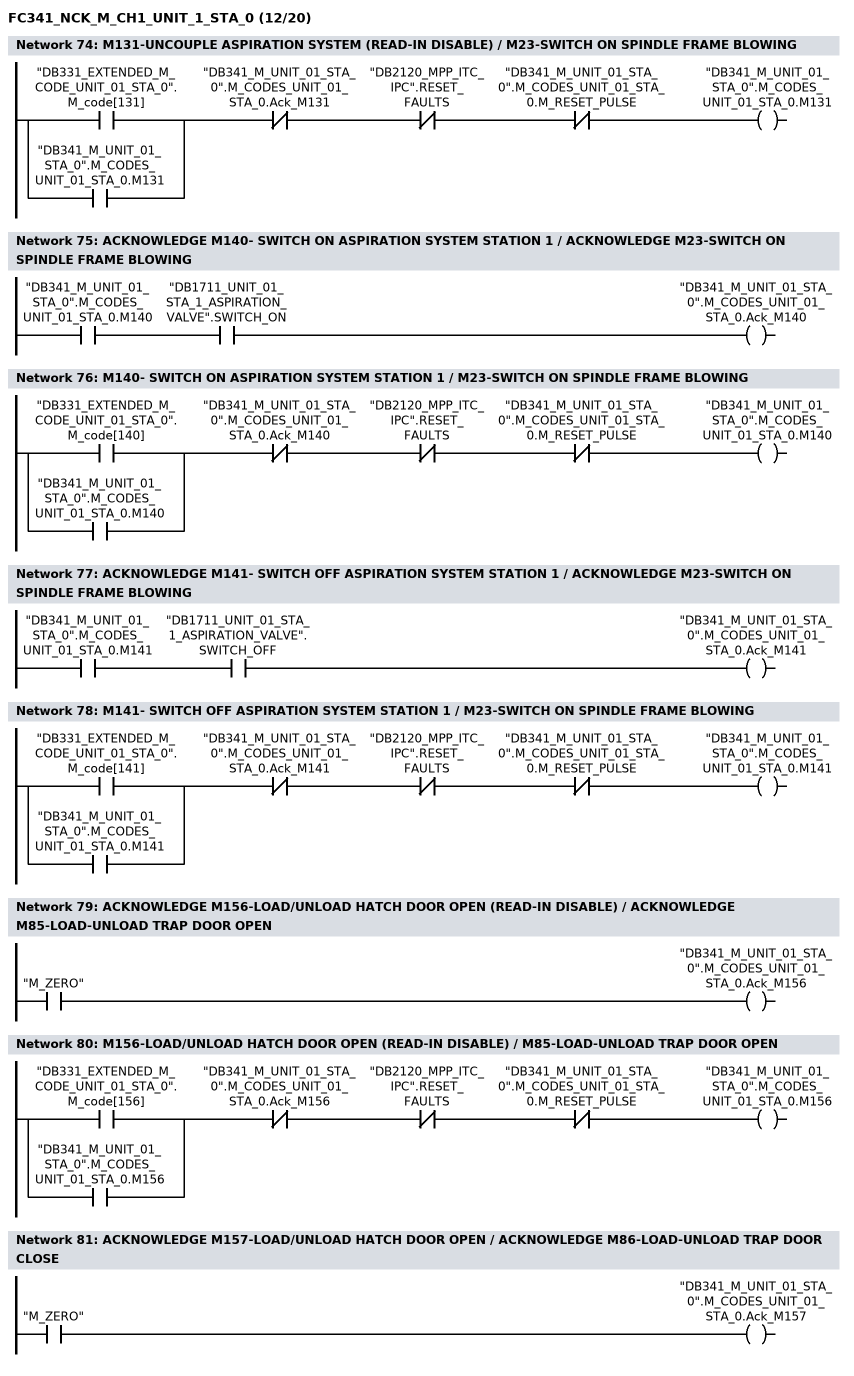
   RUNG wire#powerrail
      Contact( "DB331_EXTENDED_M_CODE_UNIT_01_STA_0".M_code[131] )
      wire#w1
      I_Contact( "DB341_M_UNIT_01_STA_0".M_CODES_UNIT_01_STA_0.Ack_M131 )
      I_Contact( "DB2120_MPP_ITC_IPC".RESET_FAULTS )
      I_Contact( "DB341_M_UNIT_01_STA_0".M_CODES_UNIT_01_STA_0.M_RESET_PULSE )
      Coil( "DB341_M_UNIT_01_STA_0".M_CODES_UNIT_01_STA_0.M131 )
   END_RUNG
   RUNG wire#powerrail
      Contact( "DB341_M_UNIT_01_STA_0".M_CODES_UNIT_01_STA_0.M131 )
   END_RUNG wire#w1
   // the same network as SCL:
   "DB341_M_UNIT_01_STA_0".M_CODES_UNIT_01_STA_0.M131 := ("DB331_EXTENDED_M_CODE_UNIT_01_STA_0".M_code[131] OR "DB341_M_UNIT_01_STA_0".M_CODES_UNIT_01_STA_0.M131) AND NOT "DB341_M_UNIT_01_STA_0".M_CODES_UNIT_01_STA_0.Ack_M131 AND NOT "DB2120_MPP_ITC_IPC".RESET_FAULTS AND NOT "DB341_M_UNIT_01_STA_0".M_CODES_UNIT_01_STA_0.M_RESET_PULSE;
END_REGION

REGION Network 75: ACKNOWLEDGE M140- SWITCH ON ASPIRATION SYSTEM STATION 1 / ACKNOWLEDGE M23-SWITCH ON SPINDLE FRAME BLOWING
   RUNG wire#powerrail
      Contact( "DB341_M_UNIT_01_STA_0".M_CODES_UNIT_01_STA_0.M140 )
      Contact( "DB1711_UNIT_01_STA_1_ASPIRATION_VALVE".SWITCH_ON )
      Coil( "DB341_M_UNIT_01_STA_0".M_CODES_UNIT_01_STA_0.Ack_M140 )
   END_RUNG
   // the same network as SCL:
   "DB341_M_UNIT_01_STA_0".M_CODES_UNIT_01_STA_0.Ack_M140 := "DB341_M_UNIT_01_STA_0".M_CODES_UNIT_01_STA_0.M140 AND "DB1711_UNIT_01_STA_1_ASPIRATION_VALVE".SWITCH_ON;
END_REGION

REGION Network 76: M140- SWITCH ON ASPIRATION SYSTEM STATION 1 / M23-SWITCH ON SPINDLE FRAME BLOWING
   RUNG wire#powerrail
      Contact( "DB331_EXTENDED_M_CODE_UNIT_01_STA_0".M_code[140] )
      wire#w1
      I_Contact( "DB341_M_UNIT_01_STA_0".M_CODES_UNIT_01_STA_0.Ack_M140 )
      I_Contact( "DB2120_MPP_ITC_IPC".RESET_FAULTS )
      I_Contact( "DB341_M_UNIT_01_STA_0".M_CODES_UNIT_01_STA_0.M_RESET_PULSE )
      Coil( "DB341_M_UNIT_01_STA_0".M_CODES_UNIT_01_STA_0.M140 )
   END_RUNG
   RUNG wire#powerrail
      Contact( "DB341_M_UNIT_01_STA_0".M_CODES_UNIT_01_STA_0.M140 )
   END_RUNG wire#w1
   // the same network as SCL:
   "DB341_M_UNIT_01_STA_0".M_CODES_UNIT_01_STA_0.M140 := ("DB331_EXTENDED_M_CODE_UNIT_01_STA_0".M_code[140] OR "DB341_M_UNIT_01_STA_0".M_CODES_UNIT_01_STA_0.M140) AND NOT "DB341_M_UNIT_01_STA_0".M_CODES_UNIT_01_STA_0.Ack_M140 AND NOT "DB2120_MPP_ITC_IPC".RESET_FAULTS AND NOT "DB341_M_UNIT_01_STA_0".M_CODES_UNIT_01_STA_0.M_RESET_PULSE;
END_REGION

REGION Network 77: ACKNOWLEDGE M141- SWITCH OFF ASPIRATION SYSTEM STATION 1 / ACKNOWLEDGE M23-SWITCH ON SPINDLE FRAME BLOWING
   RUNG wire#powerrail
      Contact( "DB341_M_UNIT_01_STA_0".M_CODES_UNIT_01_STA_0.M141 )
      Contact( "DB1711_UNIT_01_STA_1_ASPIRATION_VALVE".SWITCH_OFF )
      Coil( "DB341_M_UNIT_01_STA_0".M_CODES_UNIT_01_STA_0.Ack_M141 )
   END_RUNG
   // the same network as SCL:
   "DB341_M_UNIT_01_STA_0".M_CODES_UNIT_01_STA_0.Ack_M141 := "DB341_M_UNIT_01_STA_0".M_CODES_UNIT_01_STA_0.M141 AND "DB1711_UNIT_01_STA_1_ASPIRATION_VALVE".SWITCH_OFF;
END_REGION

REGION Network 78: M141- SWITCH OFF ASPIRATION SYSTEM STATION 1 / M23-SWITCH ON SPINDLE FRAME BLOWING
   RUNG wire#powerrail
      Contact( "DB331_EXTENDED_M_CODE_UNIT_01_STA_0".M_code[141] )
      wire#w1
      I_Contact( "DB341_M_UNIT_01_STA_0".M_CODES_UNIT_01_STA_0.Ack_M141 )
      I_Contact( "DB2120_MPP_ITC_IPC".RESET_FAULTS )
      I_Contact( "DB341_M_UNIT_01_STA_0".M_CODES_UNIT_01_STA_0.M_RESET_PULSE )
      Coil( "DB341_M_UNIT_01_STA_0".M_CODES_UNIT_01_STA_0.M141 )
   END_RUNG
   RUNG wire#powerrail
      Contact( "DB341_M_UNIT_01_STA_0".M_CODES_UNIT_01_STA_0.M141 )
   END_RUNG wire#w1
   // the same network as SCL:
   "DB341_M_UNIT_01_STA_0".M_CODES_UNIT_01_STA_0.M141 := ("DB331_EXTENDED_M_CODE_UNIT_01_STA_0".M_code[141] OR "DB341_M_UNIT_01_STA_0".M_CODES_UNIT_01_STA_0.M141) AND NOT "DB341_M_UNIT_01_STA_0".M_CODES_UNIT_01_STA_0.Ack_M141 AND NOT "DB2120_MPP_ITC_IPC".RESET_FAULTS AND NOT "DB341_M_UNIT_01_STA_0".M_CODES_UNIT_01_STA_0.M_RESET_PULSE;
END_REGION

REGION Network 79: ACKNOWLEDGE M156-LOAD/UNLOAD HATCH DOOR OPEN (READ-IN DISABLE) / ACKNOWLEDGE M85-LOAD-UNLOAD TRAP DOOR OPEN
   RUNG wire#powerrail
      Contact( "M_ZERO" )
      Coil( "DB341_M_UNIT_01_STA_0".M_CODES_UNIT_01_STA_0.Ack_M156 )
   END_RUNG
   // the same network as SCL:
   "DB341_M_UNIT_01_STA_0".M_CODES_UNIT_01_STA_0.Ack_M156 := "M_ZERO";
END_REGION

REGION Network 80: M156-LOAD/UNLOAD HATCH DOOR OPEN (READ-IN DISABLE) / M85-LOAD-UNLOAD TRAP DOOR OPEN
   RUNG wire#powerrail
      Contact( "DB331_EXTENDED_M_CODE_UNIT_01_STA_0".M_code[156] )
      wire#w1
      I_Contact( "DB341_M_UNIT_01_STA_0".M_CODES_UNIT_01_STA_0.Ack_M156 )
      I_Contact( "DB2120_MPP_ITC_IPC".RESET_FAULTS )
      I_Contact( "DB341_M_UNIT_01_STA_0".M_CODES_UNIT_01_STA_0.M_RESET_PULSE )
      Coil( "DB341_M_UNIT_01_STA_0".M_CODES_UNIT_01_STA_0.M156 )
   END_RUNG
   RUNG wire#powerrail
      Contact( "DB341_M_UNIT_01_STA_0".M_CODES_UNIT_01_STA_0.M156 )
   END_RUNG wire#w1
   // the same network as SCL:
   "DB341_M_UNIT_01_STA_0".M_CODES_UNIT_01_STA_0.M156 := ("DB331_EXTENDED_M_CODE_UNIT_01_STA_0".M_code[156] OR "DB341_M_UNIT_01_STA_0".M_CODES_UNIT_01_STA_0.M156) AND NOT "DB341_M_UNIT_01_STA_0".M_CODES_UNIT_01_STA_0.Ack_M156 AND NOT "DB2120_MPP_ITC_IPC".RESET_FAULTS AND NOT "DB341_M_UNIT_01_STA_0".M_CODES_UNIT_01_STA_0.M_RESET_PULSE;
END_REGION

REGION Network 81: ACKNOWLEDGE M157-LOAD/UNLOAD HATCH DOOR OPEN / ACKNOWLEDGE M86-LOAD-UNLOAD TRAP DOOR CLOSE
   RUNG wire#powerrail
      Contact( "M_ZERO" )
      Coil( "DB341_M_UNIT_01_STA_0".M_CODES_UNIT_01_STA_0.Ack_M157 )
   END_RUNG
   // the same network as SCL:
   "DB341_M_UNIT_01_STA_0".M_CODES_UNIT_01_STA_0.Ack_M157 := "M_ZERO";
END_REGION

REGION Network 82: M157-LOAD/UNLOAD HATCH DOOR OPEN / M86-LOAD-UNLOAD TRAP DOOR CLOSE
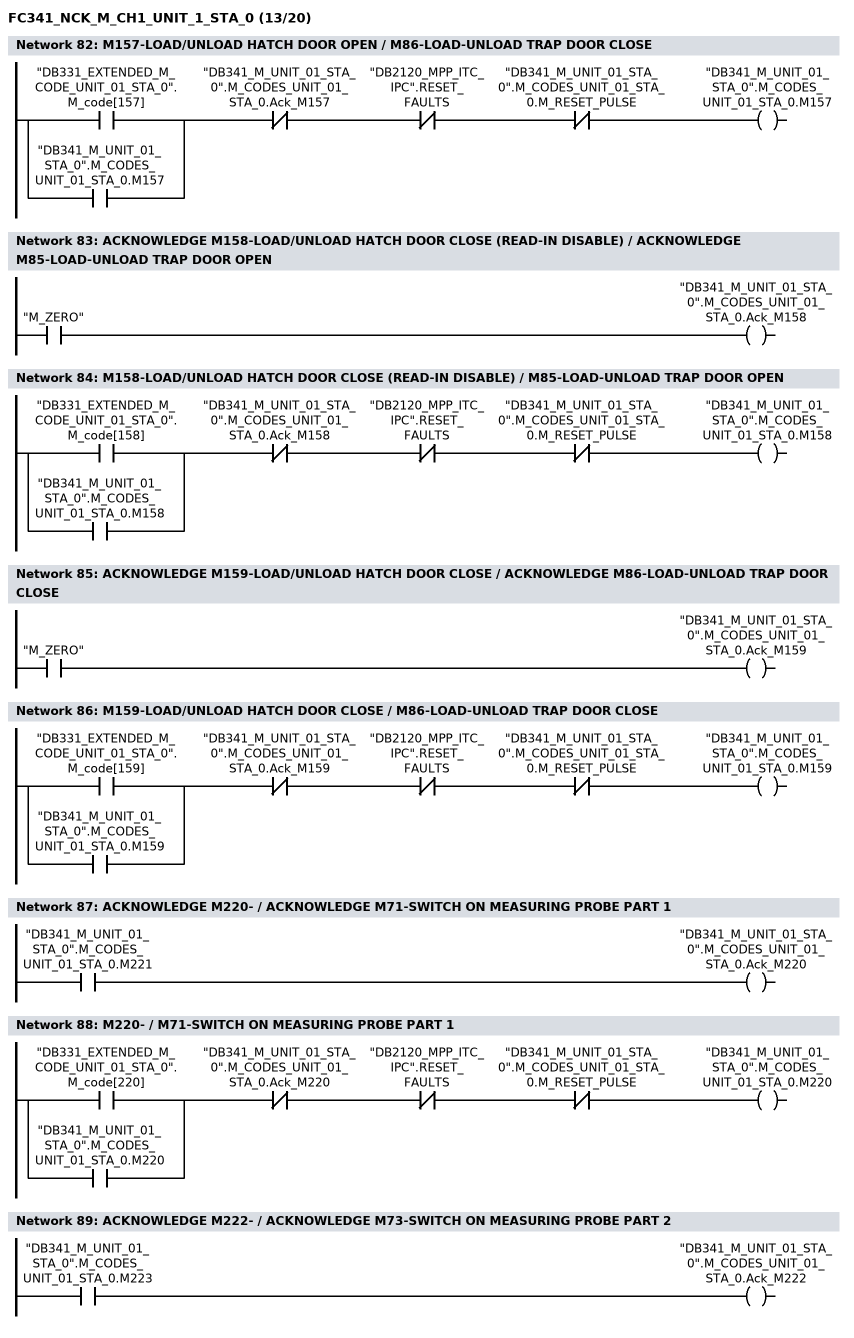
   RUNG wire#powerrail
      Contact( "DB331_EXTENDED_M_CODE_UNIT_01_STA_0".M_code[157] )
      wire#w1
      I_Contact( "DB341_M_UNIT_01_STA_0".M_CODES_UNIT_01_STA_0.Ack_M157 )
      I_Contact( "DB2120_MPP_ITC_IPC".RESET_FAULTS )
      I_Contact( "DB341_M_UNIT_01_STA_0".M_CODES_UNIT_01_STA_0.M_RESET_PULSE )
      Coil( "DB341_M_UNIT_01_STA_0".M_CODES_UNIT_01_STA_0.M157 )
   END_RUNG
   RUNG wire#powerrail
      Contact( "DB341_M_UNIT_01_STA_0".M_CODES_UNIT_01_STA_0.M157 )
   END_RUNG wire#w1
   // the same network as SCL:
   "DB341_M_UNIT_01_STA_0".M_CODES_UNIT_01_STA_0.M157 := ("DB331_EXTENDED_M_CODE_UNIT_01_STA_0".M_code[157] OR "DB341_M_UNIT_01_STA_0".M_CODES_UNIT_01_STA_0.M157) AND NOT "DB341_M_UNIT_01_STA_0".M_CODES_UNIT_01_STA_0.Ack_M157 AND NOT "DB2120_MPP_ITC_IPC".RESET_FAULTS AND NOT "DB341_M_UNIT_01_STA_0".M_CODES_UNIT_01_STA_0.M_RESET_PULSE;
END_REGION

REGION Network 83: ACKNOWLEDGE M158-LOAD/UNLOAD HATCH DOOR CLOSE (READ-IN DISABLE) / ACKNOWLEDGE M85-LOAD-UNLOAD TRAP DOOR OPEN
   RUNG wire#powerrail
      Contact( "M_ZERO" )
      Coil( "DB341_M_UNIT_01_STA_0".M_CODES_UNIT_01_STA_0.Ack_M158 )
   END_RUNG
   // the same network as SCL:
   "DB341_M_UNIT_01_STA_0".M_CODES_UNIT_01_STA_0.Ack_M158 := "M_ZERO";
END_REGION

REGION Network 84: M158-LOAD/UNLOAD HATCH DOOR CLOSE (READ-IN DISABLE) / M85-LOAD-UNLOAD TRAP DOOR OPEN
   RUNG wire#powerrail
      Contact( "DB331_EXTENDED_M_CODE_UNIT_01_STA_0".M_code[158] )
      wire#w1
      I_Contact( "DB341_M_UNIT_01_STA_0".M_CODES_UNIT_01_STA_0.Ack_M158 )
      I_Contact( "DB2120_MPP_ITC_IPC".RESET_FAULTS )
      I_Contact( "DB341_M_UNIT_01_STA_0".M_CODES_UNIT_01_STA_0.M_RESET_PULSE )
      Coil( "DB341_M_UNIT_01_STA_0".M_CODES_UNIT_01_STA_0.M158 )
   END_RUNG
   RUNG wire#powerrail
      Contact( "DB341_M_UNIT_01_STA_0".M_CODES_UNIT_01_STA_0.M158 )
   END_RUNG wire#w1
   // the same network as SCL:
   "DB341_M_UNIT_01_STA_0".M_CODES_UNIT_01_STA_0.M158 := ("DB331_EXTENDED_M_CODE_UNIT_01_STA_0".M_code[158] OR "DB341_M_UNIT_01_STA_0".M_CODES_UNIT_01_STA_0.M158) AND NOT "DB341_M_UNIT_01_STA_0".M_CODES_UNIT_01_STA_0.Ack_M158 AND NOT "DB2120_MPP_ITC_IPC".RESET_FAULTS AND NOT "DB341_M_UNIT_01_STA_0".M_CODES_UNIT_01_STA_0.M_RESET_PULSE;
END_REGION

REGION Network 85: ACKNOWLEDGE M159-LOAD/UNLOAD HATCH DOOR CLOSE / ACKNOWLEDGE M86-LOAD-UNLOAD TRAP DOOR CLOSE
   RUNG wire#powerrail
      Contact( "M_ZERO" )
      Coil( "DB341_M_UNIT_01_STA_0".M_CODES_UNIT_01_STA_0.Ack_M159 )
   END_RUNG
   // the same network as SCL:
   "DB341_M_UNIT_01_STA_0".M_CODES_UNIT_01_STA_0.Ack_M159 := "M_ZERO";
END_REGION

REGION Network 86: M159-LOAD/UNLOAD HATCH DOOR CLOSE / M86-LOAD-UNLOAD TRAP DOOR CLOSE
   RUNG wire#powerrail
      Contact( "DB331_EXTENDED_M_CODE_UNIT_01_STA_0".M_code[159] )
      wire#w1
      I_Contact( "DB341_M_UNIT_01_STA_0".M_CODES_UNIT_01_STA_0.Ack_M159 )
      I_Contact( "DB2120_MPP_ITC_IPC".RESET_FAULTS )
      I_Contact( "DB341_M_UNIT_01_STA_0".M_CODES_UNIT_01_STA_0.M_RESET_PULSE )
      Coil( "DB341_M_UNIT_01_STA_0".M_CODES_UNIT_01_STA_0.M159 )
   END_RUNG
   RUNG wire#powerrail
      Contact( "DB341_M_UNIT_01_STA_0".M_CODES_UNIT_01_STA_0.M159 )
   END_RUNG wire#w1
   // the same network as SCL:
   "DB341_M_UNIT_01_STA_0".M_CODES_UNIT_01_STA_0.M159 := ("DB331_EXTENDED_M_CODE_UNIT_01_STA_0".M_code[159] OR "DB341_M_UNIT_01_STA_0".M_CODES_UNIT_01_STA_0.M159) AND NOT "DB341_M_UNIT_01_STA_0".M_CODES_UNIT_01_STA_0.Ack_M159 AND NOT "DB2120_MPP_ITC_IPC".RESET_FAULTS AND NOT "DB341_M_UNIT_01_STA_0".M_CODES_UNIT_01_STA_0.M_RESET_PULSE;
END_REGION

REGION Network 87: ACKNOWLEDGE M220- / ACKNOWLEDGE M71-SWITCH ON MEASURING PROBE PART 1
   RUNG wire#powerrail
      Contact( "DB341_M_UNIT_01_STA_0".M_CODES_UNIT_01_STA_0.M221 )
      Coil( "DB341_M_UNIT_01_STA_0".M_CODES_UNIT_01_STA_0.Ack_M220 )
   END_RUNG
   // the same network as SCL:
   "DB341_M_UNIT_01_STA_0".M_CODES_UNIT_01_STA_0.Ack_M220 := "DB341_M_UNIT_01_STA_0".M_CODES_UNIT_01_STA_0.M221;
END_REGION

REGION Network 88: M220- / M71-SWITCH ON MEASURING PROBE PART 1
   RUNG wire#powerrail
      Contact( "DB331_EXTENDED_M_CODE_UNIT_01_STA_0".M_code[220] )
      wire#w1
      I_Contact( "DB341_M_UNIT_01_STA_0".M_CODES_UNIT_01_STA_0.Ack_M220 )
      I_Contact( "DB2120_MPP_ITC_IPC".RESET_FAULTS )
      I_Contact( "DB341_M_UNIT_01_STA_0".M_CODES_UNIT_01_STA_0.M_RESET_PULSE )
      Coil( "DB341_M_UNIT_01_STA_0".M_CODES_UNIT_01_STA_0.M220 )
   END_RUNG
   RUNG wire#powerrail
      Contact( "DB341_M_UNIT_01_STA_0".M_CODES_UNIT_01_STA_0.M220 )
   END_RUNG wire#w1
   // the same network as SCL:
   "DB341_M_UNIT_01_STA_0".M_CODES_UNIT_01_STA_0.M220 := ("DB331_EXTENDED_M_CODE_UNIT_01_STA_0".M_code[220] OR "DB341_M_UNIT_01_STA_0".M_CODES_UNIT_01_STA_0.M220) AND NOT "DB341_M_UNIT_01_STA_0".M_CODES_UNIT_01_STA_0.Ack_M220 AND NOT "DB2120_MPP_ITC_IPC".RESET_FAULTS AND NOT "DB341_M_UNIT_01_STA_0".M_CODES_UNIT_01_STA_0.M_RESET_PULSE;
END_REGION

REGION Network 89: ACKNOWLEDGE M222- / ACKNOWLEDGE M73-SWITCH ON MEASURING PROBE PART 2
   RUNG wire#powerrail
      Contact( "DB341_M_UNIT_01_STA_0".M_CODES_UNIT_01_STA_0.M223 )
      Coil( "DB341_M_UNIT_01_STA_0".M_CODES_UNIT_01_STA_0.Ack_M222 )
   END_RUNG
   // the same network as SCL:
   "DB341_M_UNIT_01_STA_0".M_CODES_UNIT_01_STA_0.Ack_M222 := "DB341_M_UNIT_01_STA_0".M_CODES_UNIT_01_STA_0.M223;
END_REGION

REGION Network 90: M222- / M73-SWITCH ON MEASURING PROBE PART 2
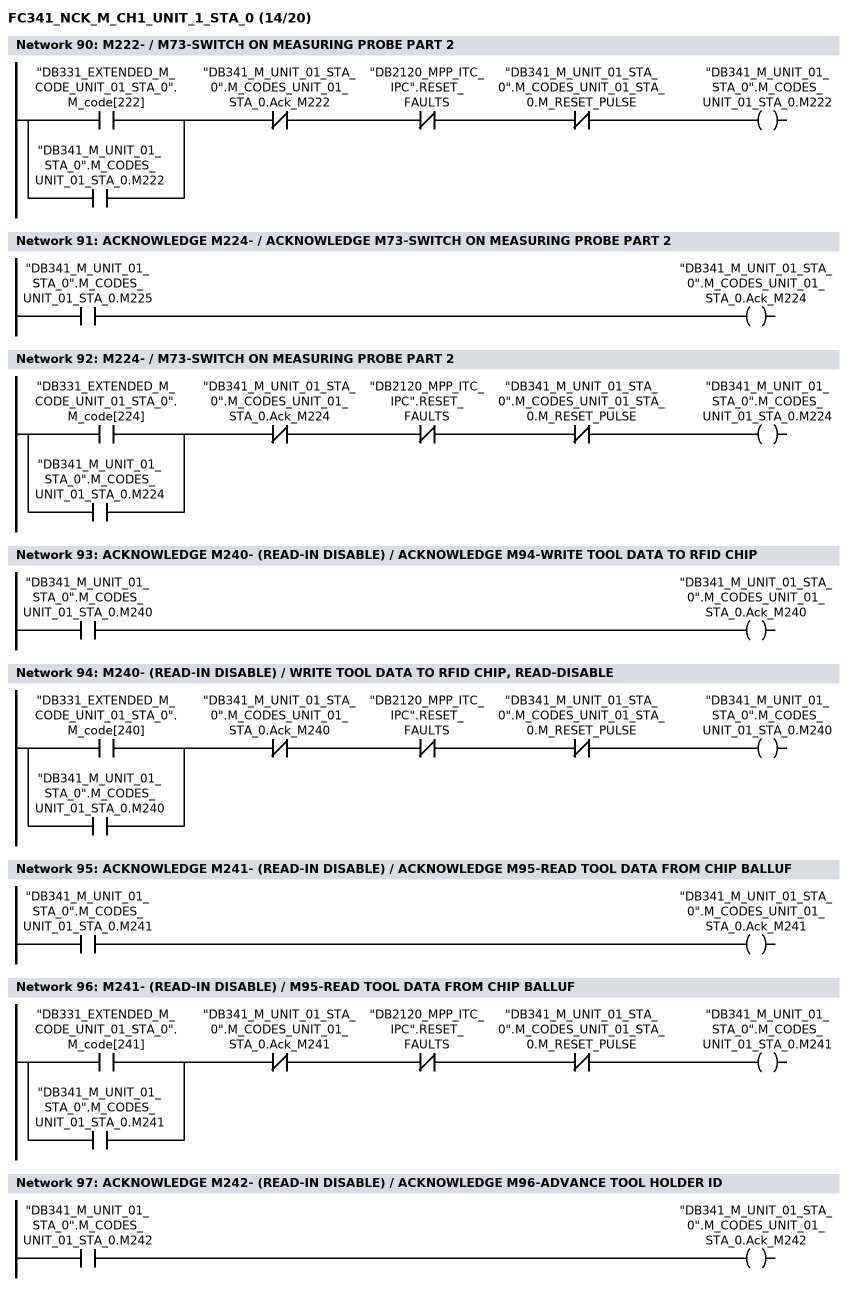
   RUNG wire#powerrail
      Contact( "DB331_EXTENDED_M_CODE_UNIT_01_STA_0".M_code[222] )
      wire#w1
      I_Contact( "DB341_M_UNIT_01_STA_0".M_CODES_UNIT_01_STA_0.Ack_M222 )
      I_Contact( "DB2120_MPP_ITC_IPC".RESET_FAULTS )
      I_Contact( "DB341_M_UNIT_01_STA_0".M_CODES_UNIT_01_STA_0.M_RESET_PULSE )
      Coil( "DB341_M_UNIT_01_STA_0".M_CODES_UNIT_01_STA_0.M222 )
   END_RUNG
   RUNG wire#powerrail
      Contact( "DB341_M_UNIT_01_STA_0".M_CODES_UNIT_01_STA_0.M222 )
   END_RUNG wire#w1
   // the same network as SCL:
   "DB341_M_UNIT_01_STA_0".M_CODES_UNIT_01_STA_0.M222 := ("DB331_EXTENDED_M_CODE_UNIT_01_STA_0".M_code[222] OR "DB341_M_UNIT_01_STA_0".M_CODES_UNIT_01_STA_0.M222) AND NOT "DB341_M_UNIT_01_STA_0".M_CODES_UNIT_01_STA_0.Ack_M222 AND NOT "DB2120_MPP_ITC_IPC".RESET_FAULTS AND NOT "DB341_M_UNIT_01_STA_0".M_CODES_UNIT_01_STA_0.M_RESET_PULSE;
END_REGION

REGION Network 91: ACKNOWLEDGE M224- / ACKNOWLEDGE M73-SWITCH ON MEASURING PROBE PART 2
   RUNG wire#powerrail
      Contact( "DB341_M_UNIT_01_STA_0".M_CODES_UNIT_01_STA_0.M225 )
      Coil( "DB341_M_UNIT_01_STA_0".M_CODES_UNIT_01_STA_0.Ack_M224 )
   END_RUNG
   // the same network as SCL:
   "DB341_M_UNIT_01_STA_0".M_CODES_UNIT_01_STA_0.Ack_M224 := "DB341_M_UNIT_01_STA_0".M_CODES_UNIT_01_STA_0.M225;
END_REGION

REGION Network 92: M224- / M73-SWITCH ON MEASURING PROBE PART 2
   RUNG wire#powerrail
      Contact( "DB331_EXTENDED_M_CODE_UNIT_01_STA_0".M_code[224] )
      wire#w1
      I_Contact( "DB341_M_UNIT_01_STA_0".M_CODES_UNIT_01_STA_0.Ack_M224 )
      I_Contact( "DB2120_MPP_ITC_IPC".RESET_FAULTS )
      I_Contact( "DB341_M_UNIT_01_STA_0".M_CODES_UNIT_01_STA_0.M_RESET_PULSE )
      Coil( "DB341_M_UNIT_01_STA_0".M_CODES_UNIT_01_STA_0.M224 )
   END_RUNG
   RUNG wire#powerrail
      Contact( "DB341_M_UNIT_01_STA_0".M_CODES_UNIT_01_STA_0.M224 )
   END_RUNG wire#w1
   // the same network as SCL:
   "DB341_M_UNIT_01_STA_0".M_CODES_UNIT_01_STA_0.M224 := ("DB331_EXTENDED_M_CODE_UNIT_01_STA_0".M_code[224] OR "DB341_M_UNIT_01_STA_0".M_CODES_UNIT_01_STA_0.M224) AND NOT "DB341_M_UNIT_01_STA_0".M_CODES_UNIT_01_STA_0.Ack_M224 AND NOT "DB2120_MPP_ITC_IPC".RESET_FAULTS AND NOT "DB341_M_UNIT_01_STA_0".M_CODES_UNIT_01_STA_0.M_RESET_PULSE;
END_REGION

REGION Network 93: ACKNOWLEDGE M240- (READ-IN DISABLE) / ACKNOWLEDGE M94-WRITE TOOL DATA TO RFID CHIP
   RUNG wire#powerrail
      Contact( "DB341_M_UNIT_01_STA_0".M_CODES_UNIT_01_STA_0.M240 )
      Coil( "DB341_M_UNIT_01_STA_0".M_CODES_UNIT_01_STA_0.Ack_M240 )
   END_RUNG
   // the same network as SCL:
   "DB341_M_UNIT_01_STA_0".M_CODES_UNIT_01_STA_0.Ack_M240 := "DB341_M_UNIT_01_STA_0".M_CODES_UNIT_01_STA_0.M240;
END_REGION

REGION Network 94: M240- (READ-IN DISABLE) / WRITE TOOL DATA TO RFID CHIP, READ-DISABLE
   RUNG wire#powerrail
      Contact( "DB331_EXTENDED_M_CODE_UNIT_01_STA_0".M_code[240] )
      wire#w1
      I_Contact( "DB341_M_UNIT_01_STA_0".M_CODES_UNIT_01_STA_0.Ack_M240 )
      I_Contact( "DB2120_MPP_ITC_IPC".RESET_FAULTS )
      I_Contact( "DB341_M_UNIT_01_STA_0".M_CODES_UNIT_01_STA_0.M_RESET_PULSE )
      Coil( "DB341_M_UNIT_01_STA_0".M_CODES_UNIT_01_STA_0.M240 )
   END_RUNG
   RUNG wire#powerrail
      Contact( "DB341_M_UNIT_01_STA_0".M_CODES_UNIT_01_STA_0.M240 )
   END_RUNG wire#w1
   // the same network as SCL:
   "DB341_M_UNIT_01_STA_0".M_CODES_UNIT_01_STA_0.M240 := ("DB331_EXTENDED_M_CODE_UNIT_01_STA_0".M_code[240] OR "DB341_M_UNIT_01_STA_0".M_CODES_UNIT_01_STA_0.M240) AND NOT "DB341_M_UNIT_01_STA_0".M_CODES_UNIT_01_STA_0.Ack_M240 AND NOT "DB2120_MPP_ITC_IPC".RESET_FAULTS AND NOT "DB341_M_UNIT_01_STA_0".M_CODES_UNIT_01_STA_0.M_RESET_PULSE;
END_REGION

REGION Network 95: ACKNOWLEDGE M241- (READ-IN DISABLE) / ACKNOWLEDGE M95-READ TOOL DATA FROM CHIP BALLUF
   RUNG wire#powerrail
      Contact( "DB341_M_UNIT_01_STA_0".M_CODES_UNIT_01_STA_0.M241 )
      Coil( "DB341_M_UNIT_01_STA_0".M_CODES_UNIT_01_STA_0.Ack_M241 )
   END_RUNG
   // the same network as SCL:
   "DB341_M_UNIT_01_STA_0".M_CODES_UNIT_01_STA_0.Ack_M241 := "DB341_M_UNIT_01_STA_0".M_CODES_UNIT_01_STA_0.M241;
END_REGION

REGION Network 96: M241- (READ-IN DISABLE) / M95-READ TOOL DATA FROM CHIP BALLUF
   RUNG wire#powerrail
      Contact( "DB331_EXTENDED_M_CODE_UNIT_01_STA_0".M_code[241] )
      wire#w1
      I_Contact( "DB341_M_UNIT_01_STA_0".M_CODES_UNIT_01_STA_0.Ack_M241 )
      I_Contact( "DB2120_MPP_ITC_IPC".RESET_FAULTS )
      I_Contact( "DB341_M_UNIT_01_STA_0".M_CODES_UNIT_01_STA_0.M_RESET_PULSE )
      Coil( "DB341_M_UNIT_01_STA_0".M_CODES_UNIT_01_STA_0.M241 )
   END_RUNG
   RUNG wire#powerrail
      Contact( "DB341_M_UNIT_01_STA_0".M_CODES_UNIT_01_STA_0.M241 )
   END_RUNG wire#w1
   // the same network as SCL:
   "DB341_M_UNIT_01_STA_0".M_CODES_UNIT_01_STA_0.M241 := ("DB331_EXTENDED_M_CODE_UNIT_01_STA_0".M_code[241] OR "DB341_M_UNIT_01_STA_0".M_CODES_UNIT_01_STA_0.M241) AND NOT "DB341_M_UNIT_01_STA_0".M_CODES_UNIT_01_STA_0.Ack_M241 AND NOT "DB2120_MPP_ITC_IPC".RESET_FAULTS AND NOT "DB341_M_UNIT_01_STA_0".M_CODES_UNIT_01_STA_0.M_RESET_PULSE;
END_REGION

REGION Network 97: ACKNOWLEDGE M242- (READ-IN DISABLE) / ACKNOWLEDGE M96-ADVANCE TOOL HOLDER ID
   RUNG wire#powerrail
      Contact( "DB341_M_UNIT_01_STA_0".M_CODES_UNIT_01_STA_0.M242 )
      Coil( "DB341_M_UNIT_01_STA_0".M_CODES_UNIT_01_STA_0.Ack_M242 )
   END_RUNG
   // the same network as SCL:
   "DB341_M_UNIT_01_STA_0".M_CODES_UNIT_01_STA_0.Ack_M242 := "DB341_M_UNIT_01_STA_0".M_CODES_UNIT_01_STA_0.M242;
END_REGION

REGION Network 98: M242- (READ-IN DISABLE) / M96-ADVANCE TOOL HOLDER ID
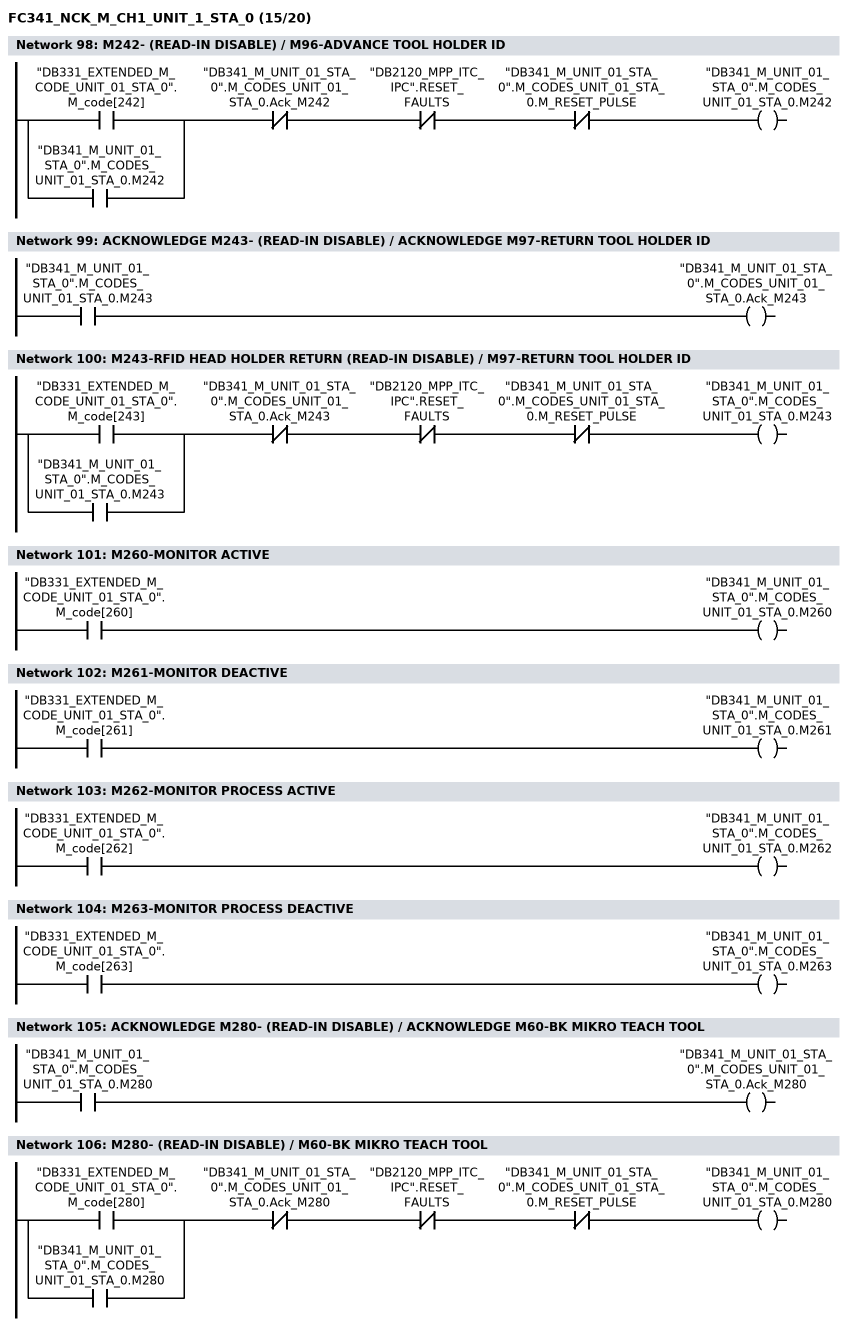
   RUNG wire#powerrail
      Contact( "DB331_EXTENDED_M_CODE_UNIT_01_STA_0".M_code[242] )
      wire#w1
      I_Contact( "DB341_M_UNIT_01_STA_0".M_CODES_UNIT_01_STA_0.Ack_M242 )
      I_Contact( "DB2120_MPP_ITC_IPC".RESET_FAULTS )
      I_Contact( "DB341_M_UNIT_01_STA_0".M_CODES_UNIT_01_STA_0.M_RESET_PULSE )
      Coil( "DB341_M_UNIT_01_STA_0".M_CODES_UNIT_01_STA_0.M242 )
   END_RUNG
   RUNG wire#powerrail
      Contact( "DB341_M_UNIT_01_STA_0".M_CODES_UNIT_01_STA_0.M242 )
   END_RUNG wire#w1
   // the same network as SCL:
   "DB341_M_UNIT_01_STA_0".M_CODES_UNIT_01_STA_0.M242 := ("DB331_EXTENDED_M_CODE_UNIT_01_STA_0".M_code[242] OR "DB341_M_UNIT_01_STA_0".M_CODES_UNIT_01_STA_0.M242) AND NOT "DB341_M_UNIT_01_STA_0".M_CODES_UNIT_01_STA_0.Ack_M242 AND NOT "DB2120_MPP_ITC_IPC".RESET_FAULTS AND NOT "DB341_M_UNIT_01_STA_0".M_CODES_UNIT_01_STA_0.M_RESET_PULSE;
END_REGION

REGION Network 99: ACKNOWLEDGE M243- (READ-IN DISABLE) / ACKNOWLEDGE M97-RETURN TOOL HOLDER ID
   RUNG wire#powerrail
      Contact( "DB341_M_UNIT_01_STA_0".M_CODES_UNIT_01_STA_0.M243 )
      Coil( "DB341_M_UNIT_01_STA_0".M_CODES_UNIT_01_STA_0.Ack_M243 )
   END_RUNG
   // the same network as SCL:
   "DB341_M_UNIT_01_STA_0".M_CODES_UNIT_01_STA_0.Ack_M243 := "DB341_M_UNIT_01_STA_0".M_CODES_UNIT_01_STA_0.M243;
END_REGION

REGION Network 100: M243-RFID HEAD HOLDER RETURN (READ-IN DISABLE) / M97-RETURN TOOL HOLDER ID
   RUNG wire#powerrail
      Contact( "DB331_EXTENDED_M_CODE_UNIT_01_STA_0".M_code[243] )
      wire#w1
      I_Contact( "DB341_M_UNIT_01_STA_0".M_CODES_UNIT_01_STA_0.Ack_M243 )
      I_Contact( "DB2120_MPP_ITC_IPC".RESET_FAULTS )
      I_Contact( "DB341_M_UNIT_01_STA_0".M_CODES_UNIT_01_STA_0.M_RESET_PULSE )
      Coil( "DB341_M_UNIT_01_STA_0".M_CODES_UNIT_01_STA_0.M243 )
   END_RUNG
   RUNG wire#powerrail
      Contact( "DB341_M_UNIT_01_STA_0".M_CODES_UNIT_01_STA_0.M243 )
   END_RUNG wire#w1
   // the same network as SCL:
   "DB341_M_UNIT_01_STA_0".M_CODES_UNIT_01_STA_0.M243 := ("DB331_EXTENDED_M_CODE_UNIT_01_STA_0".M_code[243] OR "DB341_M_UNIT_01_STA_0".M_CODES_UNIT_01_STA_0.M243) AND NOT "DB341_M_UNIT_01_STA_0".M_CODES_UNIT_01_STA_0.Ack_M243 AND NOT "DB2120_MPP_ITC_IPC".RESET_FAULTS AND NOT "DB341_M_UNIT_01_STA_0".M_CODES_UNIT_01_STA_0.M_RESET_PULSE;
END_REGION

REGION Network 101: M260-MONITOR ACTIVE
   RUNG wire#powerrail
      Contact( "DB331_EXTENDED_M_CODE_UNIT_01_STA_0".M_code[260] )
      Coil( "DB341_M_UNIT_01_STA_0".M_CODES_UNIT_01_STA_0.M260 )
   END_RUNG
   // the same network as SCL:
   "DB341_M_UNIT_01_STA_0".M_CODES_UNIT_01_STA_0.M260 := "DB331_EXTENDED_M_CODE_UNIT_01_STA_0".M_code[260];
END_REGION

REGION Network 102: M261-MONITOR DEACTIVE
   RUNG wire#powerrail
      Contact( "DB331_EXTENDED_M_CODE_UNIT_01_STA_0".M_code[261] )
      Coil( "DB341_M_UNIT_01_STA_0".M_CODES_UNIT_01_STA_0.M261 )
   END_RUNG
   // the same network as SCL:
   "DB341_M_UNIT_01_STA_0".M_CODES_UNIT_01_STA_0.M261 := "DB331_EXTENDED_M_CODE_UNIT_01_STA_0".M_code[261];
END_REGION

REGION Network 103: M262-MONITOR PROCESS ACTIVE
   RUNG wire#powerrail
      Contact( "DB331_EXTENDED_M_CODE_UNIT_01_STA_0".M_code[262] )
      Coil( "DB341_M_UNIT_01_STA_0".M_CODES_UNIT_01_STA_0.M262 )
   END_RUNG
   // the same network as SCL:
   "DB341_M_UNIT_01_STA_0".M_CODES_UNIT_01_STA_0.M262 := "DB331_EXTENDED_M_CODE_UNIT_01_STA_0".M_code[262];
END_REGION

REGION Network 104: M263-MONITOR PROCESS DEACTIVE
   RUNG wire#powerrail
      Contact( "DB331_EXTENDED_M_CODE_UNIT_01_STA_0".M_code[263] )
      Coil( "DB341_M_UNIT_01_STA_0".M_CODES_UNIT_01_STA_0.M263 )
   END_RUNG
   // the same network as SCL:
   "DB341_M_UNIT_01_STA_0".M_CODES_UNIT_01_STA_0.M263 := "DB331_EXTENDED_M_CODE_UNIT_01_STA_0".M_code[263];
END_REGION

REGION Network 105: ACKNOWLEDGE M280- (READ-IN DISABLE) / ACKNOWLEDGE M60-BK MIKRO TEACH TOOL
   RUNG wire#powerrail
      Contact( "DB341_M_UNIT_01_STA_0".M_CODES_UNIT_01_STA_0.M280 )
      Coil( "DB341_M_UNIT_01_STA_0".M_CODES_UNIT_01_STA_0.Ack_M280 )
   END_RUNG
   // the same network as SCL:
   "DB341_M_UNIT_01_STA_0".M_CODES_UNIT_01_STA_0.Ack_M280 := "DB341_M_UNIT_01_STA_0".M_CODES_UNIT_01_STA_0.M280;
END_REGION

REGION Network 106: M280- (READ-IN DISABLE) / M60-BK MIKRO TEACH TOOL
   RUNG wire#powerrail
      Contact( "DB331_EXTENDED_M_CODE_UNIT_01_STA_0".M_code[280] )
      wire#w1
      I_Contact( "DB341_M_UNIT_01_STA_0".M_CODES_UNIT_01_STA_0.Ack_M280 )
      I_Contact( "DB2120_MPP_ITC_IPC".RESET_FAULTS )
      I_Contact( "DB341_M_UNIT_01_STA_0".M_CODES_UNIT_01_STA_0.M_RESET_PULSE )
      Coil( "DB341_M_UNIT_01_STA_0".M_CODES_UNIT_01_STA_0.M280 )
   END_RUNG
   RUNG wire#powerrail
      Contact( "DB341_M_UNIT_01_STA_0".M_CODES_UNIT_01_STA_0.M280 )
   END_RUNG wire#w1
   // the same network as SCL:
   "DB341_M_UNIT_01_STA_0".M_CODES_UNIT_01_STA_0.M280 := ("DB331_EXTENDED_M_CODE_UNIT_01_STA_0".M_code[280] OR "DB341_M_UNIT_01_STA_0".M_CODES_UNIT_01_STA_0.M280) AND NOT "DB341_M_UNIT_01_STA_0".M_CODES_UNIT_01_STA_0.Ack_M280 AND NOT "DB2120_MPP_ITC_IPC".RESET_FAULTS AND NOT "DB341_M_UNIT_01_STA_0".M_CODES_UNIT_01_STA_0.M_RESET_PULSE;
END_REGION

REGION Network 107: ACKNOWLEDGE M290- / ACKNOWLEDGE M11-CLAMP GRIPPERS TOOLS
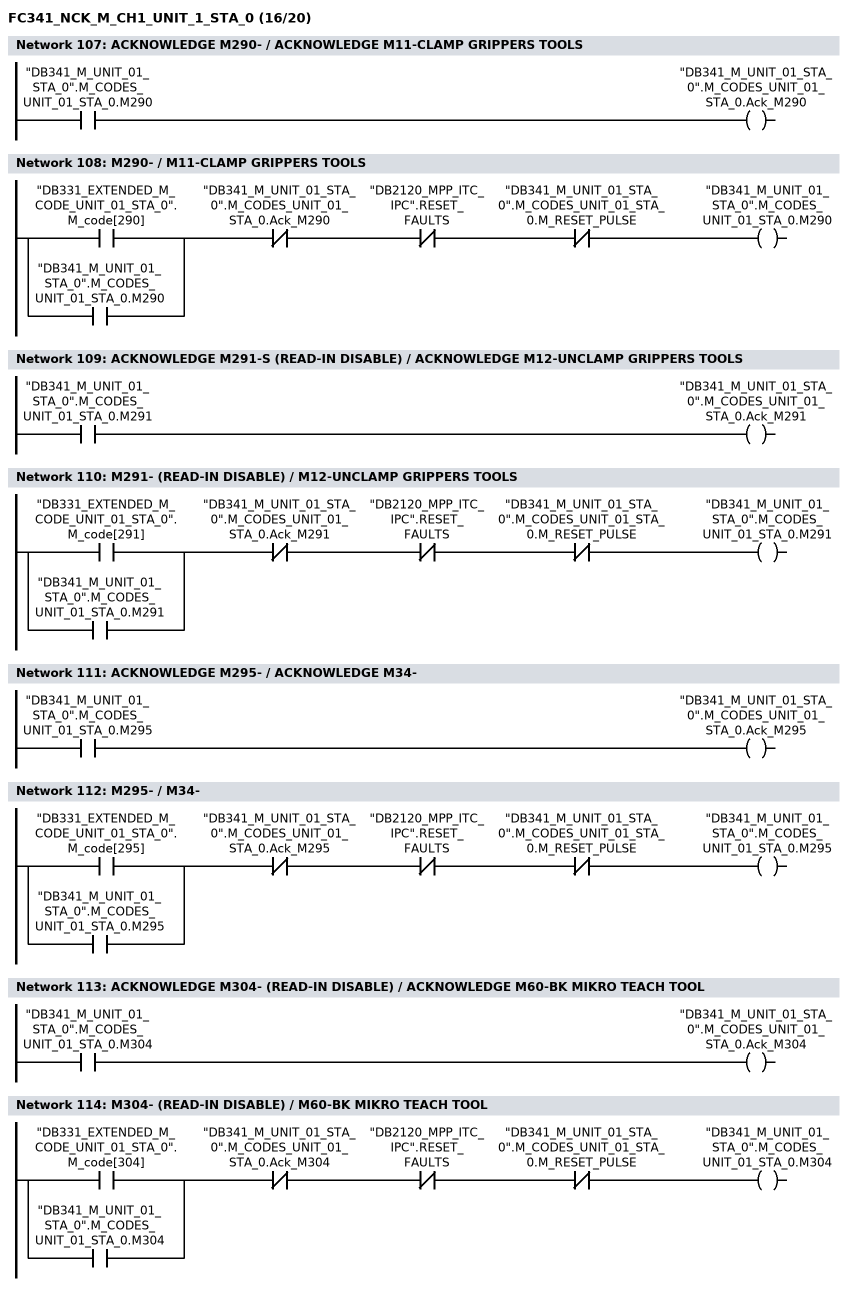
   RUNG wire#powerrail
      Contact( "DB341_M_UNIT_01_STA_0".M_CODES_UNIT_01_STA_0.M290 )
      Coil( "DB341_M_UNIT_01_STA_0".M_CODES_UNIT_01_STA_0.Ack_M290 )
   END_RUNG
   // the same network as SCL:
   "DB341_M_UNIT_01_STA_0".M_CODES_UNIT_01_STA_0.Ack_M290 := "DB341_M_UNIT_01_STA_0".M_CODES_UNIT_01_STA_0.M290;
END_REGION

REGION Network 108: M290- / M11-CLAMP GRIPPERS TOOLS
   RUNG wire#powerrail
      Contact( "DB331_EXTENDED_M_CODE_UNIT_01_STA_0".M_code[290] )
      wire#w1
      I_Contact( "DB341_M_UNIT_01_STA_0".M_CODES_UNIT_01_STA_0.Ack_M290 )
      I_Contact( "DB2120_MPP_ITC_IPC".RESET_FAULTS )
      I_Contact( "DB341_M_UNIT_01_STA_0".M_CODES_UNIT_01_STA_0.M_RESET_PULSE )
      Coil( "DB341_M_UNIT_01_STA_0".M_CODES_UNIT_01_STA_0.M290 )
   END_RUNG
   RUNG wire#powerrail
      Contact( "DB341_M_UNIT_01_STA_0".M_CODES_UNIT_01_STA_0.M290 )
   END_RUNG wire#w1
   // the same network as SCL:
   "DB341_M_UNIT_01_STA_0".M_CODES_UNIT_01_STA_0.M290 := ("DB331_EXTENDED_M_CODE_UNIT_01_STA_0".M_code[290] OR "DB341_M_UNIT_01_STA_0".M_CODES_UNIT_01_STA_0.M290) AND NOT "DB341_M_UNIT_01_STA_0".M_CODES_UNIT_01_STA_0.Ack_M290 AND NOT "DB2120_MPP_ITC_IPC".RESET_FAULTS AND NOT "DB341_M_UNIT_01_STA_0".M_CODES_UNIT_01_STA_0.M_RESET_PULSE;
END_REGION

REGION Network 109: ACKNOWLEDGE M291-S (READ-IN DISABLE) / ACKNOWLEDGE M12-UNCLAMP GRIPPERS TOOLS
   RUNG wire#powerrail
      Contact( "DB341_M_UNIT_01_STA_0".M_CODES_UNIT_01_STA_0.M291 )
      Coil( "DB341_M_UNIT_01_STA_0".M_CODES_UNIT_01_STA_0.Ack_M291 )
   END_RUNG
   // the same network as SCL:
   "DB341_M_UNIT_01_STA_0".M_CODES_UNIT_01_STA_0.Ack_M291 := "DB341_M_UNIT_01_STA_0".M_CODES_UNIT_01_STA_0.M291;
END_REGION

REGION Network 110: M291- (READ-IN DISABLE) / M12-UNCLAMP GRIPPERS TOOLS
   RUNG wire#powerrail
      Contact( "DB331_EXTENDED_M_CODE_UNIT_01_STA_0".M_code[291] )
      wire#w1
      I_Contact( "DB341_M_UNIT_01_STA_0".M_CODES_UNIT_01_STA_0.Ack_M291 )
      I_Contact( "DB2120_MPP_ITC_IPC".RESET_FAULTS )
      I_Contact( "DB341_M_UNIT_01_STA_0".M_CODES_UNIT_01_STA_0.M_RESET_PULSE )
      Coil( "DB341_M_UNIT_01_STA_0".M_CODES_UNIT_01_STA_0.M291 )
   END_RUNG
   RUNG wire#powerrail
      Contact( "DB341_M_UNIT_01_STA_0".M_CODES_UNIT_01_STA_0.M291 )
   END_RUNG wire#w1
   // the same network as SCL:
   "DB341_M_UNIT_01_STA_0".M_CODES_UNIT_01_STA_0.M291 := ("DB331_EXTENDED_M_CODE_UNIT_01_STA_0".M_code[291] OR "DB341_M_UNIT_01_STA_0".M_CODES_UNIT_01_STA_0.M291) AND NOT "DB341_M_UNIT_01_STA_0".M_CODES_UNIT_01_STA_0.Ack_M291 AND NOT "DB2120_MPP_ITC_IPC".RESET_FAULTS AND NOT "DB341_M_UNIT_01_STA_0".M_CODES_UNIT_01_STA_0.M_RESET_PULSE;
END_REGION

REGION Network 111: ACKNOWLEDGE M295- / ACKNOWLEDGE M34-
   RUNG wire#powerrail
      Contact( "DB341_M_UNIT_01_STA_0".M_CODES_UNIT_01_STA_0.M295 )
      Coil( "DB341_M_UNIT_01_STA_0".M_CODES_UNIT_01_STA_0.Ack_M295 )
   END_RUNG
   // the same network as SCL:
   "DB341_M_UNIT_01_STA_0".M_CODES_UNIT_01_STA_0.Ack_M295 := "DB341_M_UNIT_01_STA_0".M_CODES_UNIT_01_STA_0.M295;
END_REGION

REGION Network 112: M295- / M34-
   RUNG wire#powerrail
      Contact( "DB331_EXTENDED_M_CODE_UNIT_01_STA_0".M_code[295] )
      wire#w1
      I_Contact( "DB341_M_UNIT_01_STA_0".M_CODES_UNIT_01_STA_0.Ack_M295 )
      I_Contact( "DB2120_MPP_ITC_IPC".RESET_FAULTS )
      I_Contact( "DB341_M_UNIT_01_STA_0".M_CODES_UNIT_01_STA_0.M_RESET_PULSE )
      Coil( "DB341_M_UNIT_01_STA_0".M_CODES_UNIT_01_STA_0.M295 )
   END_RUNG
   RUNG wire#powerrail
      Contact( "DB341_M_UNIT_01_STA_0".M_CODES_UNIT_01_STA_0.M295 )
   END_RUNG wire#w1
   // the same network as SCL:
   "DB341_M_UNIT_01_STA_0".M_CODES_UNIT_01_STA_0.M295 := ("DB331_EXTENDED_M_CODE_UNIT_01_STA_0".M_code[295] OR "DB341_M_UNIT_01_STA_0".M_CODES_UNIT_01_STA_0.M295) AND NOT "DB341_M_UNIT_01_STA_0".M_CODES_UNIT_01_STA_0.Ack_M295 AND NOT "DB2120_MPP_ITC_IPC".RESET_FAULTS AND NOT "DB341_M_UNIT_01_STA_0".M_CODES_UNIT_01_STA_0.M_RESET_PULSE;
END_REGION

REGION Network 113: ACKNOWLEDGE M304- (READ-IN DISABLE) / ACKNOWLEDGE M60-BK MIKRO TEACH TOOL
   RUNG wire#powerrail
      Contact( "DB341_M_UNIT_01_STA_0".M_CODES_UNIT_01_STA_0.M304 )
      Coil( "DB341_M_UNIT_01_STA_0".M_CODES_UNIT_01_STA_0.Ack_M304 )
   END_RUNG
   // the same network as SCL:
   "DB341_M_UNIT_01_STA_0".M_CODES_UNIT_01_STA_0.Ack_M304 := "DB341_M_UNIT_01_STA_0".M_CODES_UNIT_01_STA_0.M304;
END_REGION

REGION Network 114: M304- (READ-IN DISABLE) / M60-BK MIKRO TEACH TOOL
   RUNG wire#powerrail
      Contact( "DB331_EXTENDED_M_CODE_UNIT_01_STA_0".M_code[304] )
      wire#w1
      I_Contact( "DB341_M_UNIT_01_STA_0".M_CODES_UNIT_01_STA_0.Ack_M304 )
      I_Contact( "DB2120_MPP_ITC_IPC".RESET_FAULTS )
      I_Contact( "DB341_M_UNIT_01_STA_0".M_CODES_UNIT_01_STA_0.M_RESET_PULSE )
      Coil( "DB341_M_UNIT_01_STA_0".M_CODES_UNIT_01_STA_0.M304 )
   END_RUNG
   RUNG wire#powerrail
      Contact( "DB341_M_UNIT_01_STA_0".M_CODES_UNIT_01_STA_0.M304 )
   END_RUNG wire#w1
   // the same network as SCL:
   "DB341_M_UNIT_01_STA_0".M_CODES_UNIT_01_STA_0.M304 := ("DB331_EXTENDED_M_CODE_UNIT_01_STA_0".M_code[304] OR "DB341_M_UNIT_01_STA_0".M_CODES_UNIT_01_STA_0.M304) AND NOT "DB341_M_UNIT_01_STA_0".M_CODES_UNIT_01_STA_0.Ack_M304 AND NOT "DB2120_MPP_ITC_IPC".RESET_FAULTS AND NOT "DB341_M_UNIT_01_STA_0".M_CODES_UNIT_01_STA_0.M_RESET_PULSE;
END_REGION

REGION Network 115: ACKNOWLEDGE M305- (READ-IN DISABLE) / ACKNOWLEDGE M61-BK MIKRO PREPOS TOOL
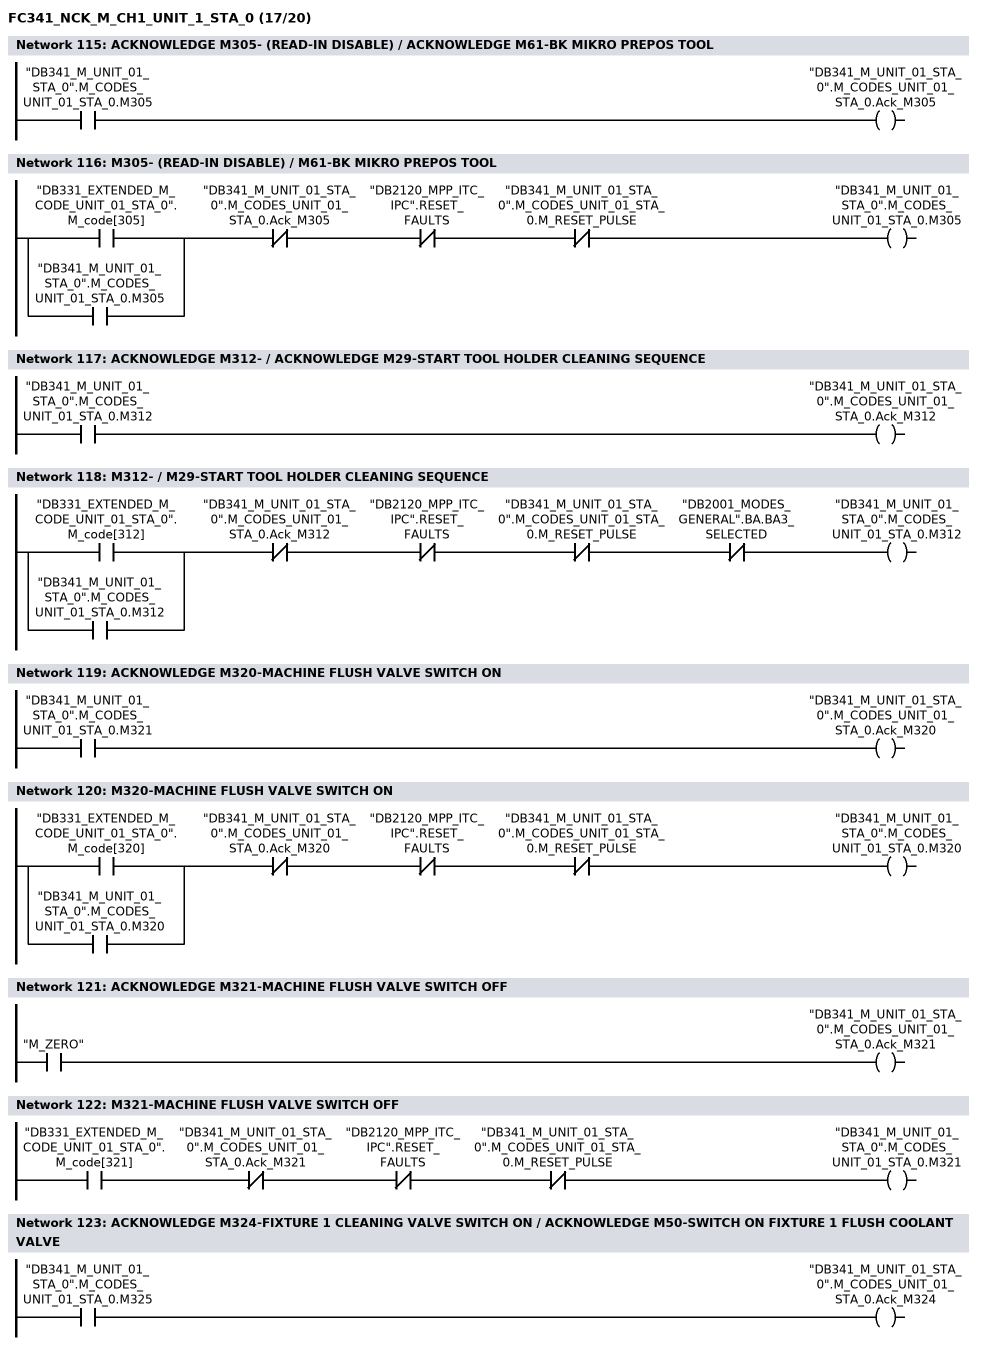
   RUNG wire#powerrail
      Contact( "DB341_M_UNIT_01_STA_0".M_CODES_UNIT_01_STA_0.M305 )
      Coil( "DB341_M_UNIT_01_STA_0".M_CODES_UNIT_01_STA_0.Ack_M305 )
   END_RUNG
   // the same network as SCL:
   "DB341_M_UNIT_01_STA_0".M_CODES_UNIT_01_STA_0.Ack_M305 := "DB341_M_UNIT_01_STA_0".M_CODES_UNIT_01_STA_0.M305;
END_REGION

REGION Network 116: M305- (READ-IN DISABLE) / M61-BK MIKRO PREPOS TOOL
   RUNG wire#powerrail
      Contact( "DB331_EXTENDED_M_CODE_UNIT_01_STA_0".M_code[305] )
      wire#w1
      I_Contact( "DB341_M_UNIT_01_STA_0".M_CODES_UNIT_01_STA_0.Ack_M305 )
      I_Contact( "DB2120_MPP_ITC_IPC".RESET_FAULTS )
      I_Contact( "DB341_M_UNIT_01_STA_0".M_CODES_UNIT_01_STA_0.M_RESET_PULSE )
      Coil( "DB341_M_UNIT_01_STA_0".M_CODES_UNIT_01_STA_0.M305 )
   END_RUNG
   RUNG wire#powerrail
      Contact( "DB341_M_UNIT_01_STA_0".M_CODES_UNIT_01_STA_0.M305 )
   END_RUNG wire#w1
   // the same network as SCL:
   "DB341_M_UNIT_01_STA_0".M_CODES_UNIT_01_STA_0.M305 := ("DB331_EXTENDED_M_CODE_UNIT_01_STA_0".M_code[305] OR "DB341_M_UNIT_01_STA_0".M_CODES_UNIT_01_STA_0.M305) AND NOT "DB341_M_UNIT_01_STA_0".M_CODES_UNIT_01_STA_0.Ack_M305 AND NOT "DB2120_MPP_ITC_IPC".RESET_FAULTS AND NOT "DB341_M_UNIT_01_STA_0".M_CODES_UNIT_01_STA_0.M_RESET_PULSE;
END_REGION

REGION Network 117: ACKNOWLEDGE M312- / ACKNOWLEDGE M29-START TOOL HOLDER CLEANING SEQUENCE
   RUNG wire#powerrail
      Contact( "DB341_M_UNIT_01_STA_0".M_CODES_UNIT_01_STA_0.M312 )
      Coil( "DB341_M_UNIT_01_STA_0".M_CODES_UNIT_01_STA_0.Ack_M312 )
   END_RUNG
   // the same network as SCL:
   "DB341_M_UNIT_01_STA_0".M_CODES_UNIT_01_STA_0.Ack_M312 := "DB341_M_UNIT_01_STA_0".M_CODES_UNIT_01_STA_0.M312;
END_REGION

REGION Network 118: M312- / M29-START TOOL HOLDER CLEANING SEQUENCE
   RUNG wire#powerrail
      Contact( "DB331_EXTENDED_M_CODE_UNIT_01_STA_0".M_code[312] )
      wire#w1
      I_Contact( "DB341_M_UNIT_01_STA_0".M_CODES_UNIT_01_STA_0.Ack_M312 )
      I_Contact( "DB2120_MPP_ITC_IPC".RESET_FAULTS )
      I_Contact( "DB341_M_UNIT_01_STA_0".M_CODES_UNIT_01_STA_0.M_RESET_PULSE )
      I_Contact( "DB2001_MODES_GENERAL".BA.BA3_SELECTED )
      Coil( "DB341_M_UNIT_01_STA_0".M_CODES_UNIT_01_STA_0.M312 )
   END_RUNG
   RUNG wire#powerrail
      Contact( "DB341_M_UNIT_01_STA_0".M_CODES_UNIT_01_STA_0.M312 )
   END_RUNG wire#w1
   // the same network as SCL:
   "DB341_M_UNIT_01_STA_0".M_CODES_UNIT_01_STA_0.M312 := ("DB331_EXTENDED_M_CODE_UNIT_01_STA_0".M_code[312] OR "DB341_M_UNIT_01_STA_0".M_CODES_UNIT_01_STA_0.M312) AND NOT "DB341_M_UNIT_01_STA_0".M_CODES_UNIT_01_STA_0.Ack_M312 AND NOT "DB2120_MPP_ITC_IPC".RESET_FAULTS AND NOT "DB341_M_UNIT_01_STA_0".M_CODES_UNIT_01_STA_0.M_RESET_PULSE AND NOT "DB2001_MODES_GENERAL".BA.BA3_SELECTED;
END_REGION

REGION Network 119: ACKNOWLEDGE M320-MACHINE FLUSH VALVE SWITCH ON
   RUNG wire#powerrail
      Contact( "DB341_M_UNIT_01_STA_0".M_CODES_UNIT_01_STA_0.M321 )
      Coil( "DB341_M_UNIT_01_STA_0".M_CODES_UNIT_01_STA_0.Ack_M320 )
   END_RUNG
   // the same network as SCL:
   "DB341_M_UNIT_01_STA_0".M_CODES_UNIT_01_STA_0.Ack_M320 := "DB341_M_UNIT_01_STA_0".M_CODES_UNIT_01_STA_0.M321;
END_REGION

REGION Network 120: M320-MACHINE FLUSH VALVE SWITCH ON
   RUNG wire#powerrail
      Contact( "DB331_EXTENDED_M_CODE_UNIT_01_STA_0".M_code[320] )
      wire#w1
      I_Contact( "DB341_M_UNIT_01_STA_0".M_CODES_UNIT_01_STA_0.Ack_M320 )
      I_Contact( "DB2120_MPP_ITC_IPC".RESET_FAULTS )
      I_Contact( "DB341_M_UNIT_01_STA_0".M_CODES_UNIT_01_STA_0.M_RESET_PULSE )
      Coil( "DB341_M_UNIT_01_STA_0".M_CODES_UNIT_01_STA_0.M320 )
   END_RUNG
   RUNG wire#powerrail
      Contact( "DB341_M_UNIT_01_STA_0".M_CODES_UNIT_01_STA_0.M320 )
   END_RUNG wire#w1
   // the same network as SCL:
   "DB341_M_UNIT_01_STA_0".M_CODES_UNIT_01_STA_0.M320 := ("DB331_EXTENDED_M_CODE_UNIT_01_STA_0".M_code[320] OR "DB341_M_UNIT_01_STA_0".M_CODES_UNIT_01_STA_0.M320) AND NOT "DB341_M_UNIT_01_STA_0".M_CODES_UNIT_01_STA_0.Ack_M320 AND NOT "DB2120_MPP_ITC_IPC".RESET_FAULTS AND NOT "DB341_M_UNIT_01_STA_0".M_CODES_UNIT_01_STA_0.M_RESET_PULSE;
END_REGION

REGION Network 121: ACKNOWLEDGE M321-MACHINE FLUSH VALVE SWITCH OFF
   RUNG wire#powerrail
      Contact( "M_ZERO" )
      Coil( "DB341_M_UNIT_01_STA_0".M_CODES_UNIT_01_STA_0.Ack_M321 )
   END_RUNG
   // the same network as SCL:
   "DB341_M_UNIT_01_STA_0".M_CODES_UNIT_01_STA_0.Ack_M321 := "M_ZERO";
END_REGION

REGION Network 122: M321-MACHINE FLUSH VALVE SWITCH OFF
   RUNG wire#powerrail
      Contact( "DB331_EXTENDED_M_CODE_UNIT_01_STA_0".M_code[321] )
      I_Contact( "DB341_M_UNIT_01_STA_0".M_CODES_UNIT_01_STA_0.Ack_M321 )
      I_Contact( "DB2120_MPP_ITC_IPC".RESET_FAULTS )
      I_Contact( "DB341_M_UNIT_01_STA_0".M_CODES_UNIT_01_STA_0.M_RESET_PULSE )
      Coil( "DB341_M_UNIT_01_STA_0".M_CODES_UNIT_01_STA_0.M321 )
   END_RUNG
   // the same network as SCL:
   "DB341_M_UNIT_01_STA_0".M_CODES_UNIT_01_STA_0.M321 := "DB331_EXTENDED_M_CODE_UNIT_01_STA_0".M_code[321] AND NOT "DB341_M_UNIT_01_STA_0".M_CODES_UNIT_01_STA_0.Ack_M321 AND NOT "DB2120_MPP_ITC_IPC".RESET_FAULTS AND NOT "DB341_M_UNIT_01_STA_0".M_CODES_UNIT_01_STA_0.M_RESET_PULSE;
END_REGION

REGION Network 123: ACKNOWLEDGE M324-FIXTURE 1 CLEANING VALVE SWITCH ON / ACKNOWLEDGE M50-SWITCH ON FIXTURE 1 FLUSH COOLANT VALVE
   RUNG wire#powerrail
      Contact( "DB341_M_UNIT_01_STA_0".M_CODES_UNIT_01_STA_0.M325 )
      Coil( "DB341_M_UNIT_01_STA_0".M_CODES_UNIT_01_STA_0.Ack_M324 )
   END_RUNG
   // the same network as SCL:
   "DB341_M_UNIT_01_STA_0".M_CODES_UNIT_01_STA_0.Ack_M324 := "DB341_M_UNIT_01_STA_0".M_CODES_UNIT_01_STA_0.M325;
END_REGION

REGION Network 124: M324-FIXTURE 1 CLEANING VALVE SWITCH ON / M50-SWITCH ON FIXTURE 1 FLUSH COOLANT VALVE
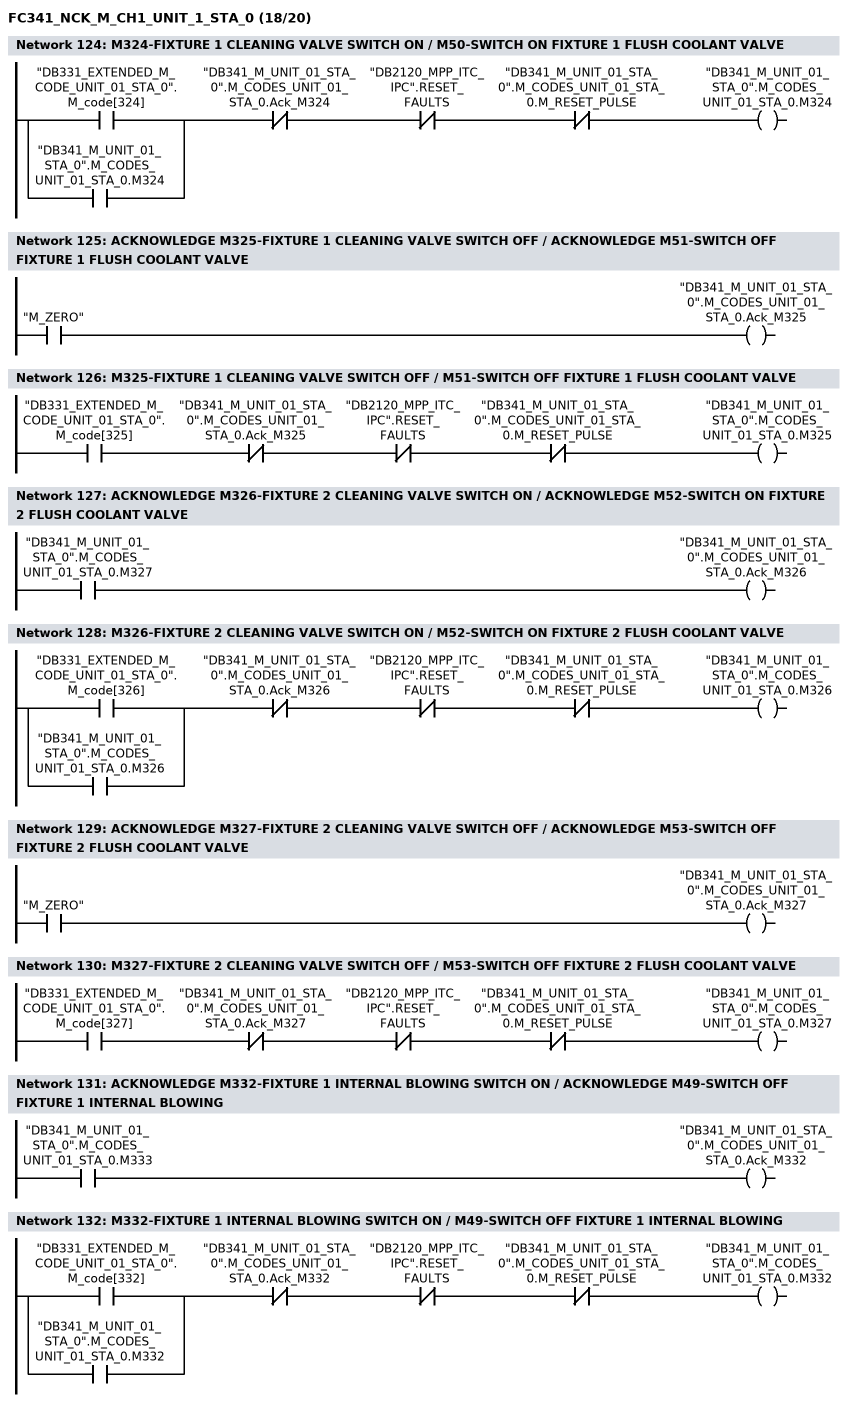
   RUNG wire#powerrail
      Contact( "DB331_EXTENDED_M_CODE_UNIT_01_STA_0".M_code[324] )
      wire#w1
      I_Contact( "DB341_M_UNIT_01_STA_0".M_CODES_UNIT_01_STA_0.Ack_M324 )
      I_Contact( "DB2120_MPP_ITC_IPC".RESET_FAULTS )
      I_Contact( "DB341_M_UNIT_01_STA_0".M_CODES_UNIT_01_STA_0.M_RESET_PULSE )
      Coil( "DB341_M_UNIT_01_STA_0".M_CODES_UNIT_01_STA_0.M324 )
   END_RUNG
   RUNG wire#powerrail
      Contact( "DB341_M_UNIT_01_STA_0".M_CODES_UNIT_01_STA_0.M324 )
   END_RUNG wire#w1
   // the same network as SCL:
   "DB341_M_UNIT_01_STA_0".M_CODES_UNIT_01_STA_0.M324 := ("DB331_EXTENDED_M_CODE_UNIT_01_STA_0".M_code[324] OR "DB341_M_UNIT_01_STA_0".M_CODES_UNIT_01_STA_0.M324) AND NOT "DB341_M_UNIT_01_STA_0".M_CODES_UNIT_01_STA_0.Ack_M324 AND NOT "DB2120_MPP_ITC_IPC".RESET_FAULTS AND NOT "DB341_M_UNIT_01_STA_0".M_CODES_UNIT_01_STA_0.M_RESET_PULSE;
END_REGION

REGION Network 125: ACKNOWLEDGE M325-FIXTURE 1 CLEANING VALVE SWITCH OFF / ACKNOWLEDGE M51-SWITCH OFF FIXTURE 1 FLUSH COOLANT VALVE
   RUNG wire#powerrail
      Contact( "M_ZERO" )
      Coil( "DB341_M_UNIT_01_STA_0".M_CODES_UNIT_01_STA_0.Ack_M325 )
   END_RUNG
   // the same network as SCL:
   "DB341_M_UNIT_01_STA_0".M_CODES_UNIT_01_STA_0.Ack_M325 := "M_ZERO";
END_REGION

REGION Network 126: M325-FIXTURE 1 CLEANING VALVE SWITCH OFF / M51-SWITCH OFF FIXTURE 1 FLUSH COOLANT VALVE
   RUNG wire#powerrail
      Contact( "DB331_EXTENDED_M_CODE_UNIT_01_STA_0".M_code[325] )
      I_Contact( "DB341_M_UNIT_01_STA_0".M_CODES_UNIT_01_STA_0.Ack_M325 )
      I_Contact( "DB2120_MPP_ITC_IPC".RESET_FAULTS )
      I_Contact( "DB341_M_UNIT_01_STA_0".M_CODES_UNIT_01_STA_0.M_RESET_PULSE )
      Coil( "DB341_M_UNIT_01_STA_0".M_CODES_UNIT_01_STA_0.M325 )
   END_RUNG
   // the same network as SCL:
   "DB341_M_UNIT_01_STA_0".M_CODES_UNIT_01_STA_0.M325 := "DB331_EXTENDED_M_CODE_UNIT_01_STA_0".M_code[325] AND NOT "DB341_M_UNIT_01_STA_0".M_CODES_UNIT_01_STA_0.Ack_M325 AND NOT "DB2120_MPP_ITC_IPC".RESET_FAULTS AND NOT "DB341_M_UNIT_01_STA_0".M_CODES_UNIT_01_STA_0.M_RESET_PULSE;
END_REGION

REGION Network 127: ACKNOWLEDGE M326-FIXTURE 2 CLEANING VALVE SWITCH ON / ACKNOWLEDGE M52-SWITCH ON FIXTURE 2 FLUSH COOLANT VALVE
   RUNG wire#powerrail
      Contact( "DB341_M_UNIT_01_STA_0".M_CODES_UNIT_01_STA_0.M327 )
      Coil( "DB341_M_UNIT_01_STA_0".M_CODES_UNIT_01_STA_0.Ack_M326 )
   END_RUNG
   // the same network as SCL:
   "DB341_M_UNIT_01_STA_0".M_CODES_UNIT_01_STA_0.Ack_M326 := "DB341_M_UNIT_01_STA_0".M_CODES_UNIT_01_STA_0.M327;
END_REGION

REGION Network 128: M326-FIXTURE 2 CLEANING VALVE SWITCH ON / M52-SWITCH ON FIXTURE 2 FLUSH COOLANT VALVE
   RUNG wire#powerrail
      Contact( "DB331_EXTENDED_M_CODE_UNIT_01_STA_0".M_code[326] )
      wire#w1
      I_Contact( "DB341_M_UNIT_01_STA_0".M_CODES_UNIT_01_STA_0.Ack_M326 )
      I_Contact( "DB2120_MPP_ITC_IPC".RESET_FAULTS )
      I_Contact( "DB341_M_UNIT_01_STA_0".M_CODES_UNIT_01_STA_0.M_RESET_PULSE )
      Coil( "DB341_M_UNIT_01_STA_0".M_CODES_UNIT_01_STA_0.M326 )
   END_RUNG
   RUNG wire#powerrail
      Contact( "DB341_M_UNIT_01_STA_0".M_CODES_UNIT_01_STA_0.M326 )
   END_RUNG wire#w1
   // the same network as SCL:
   "DB341_M_UNIT_01_STA_0".M_CODES_UNIT_01_STA_0.M326 := ("DB331_EXTENDED_M_CODE_UNIT_01_STA_0".M_code[326] OR "DB341_M_UNIT_01_STA_0".M_CODES_UNIT_01_STA_0.M326) AND NOT "DB341_M_UNIT_01_STA_0".M_CODES_UNIT_01_STA_0.Ack_M326 AND NOT "DB2120_MPP_ITC_IPC".RESET_FAULTS AND NOT "DB341_M_UNIT_01_STA_0".M_CODES_UNIT_01_STA_0.M_RESET_PULSE;
END_REGION

REGION Network 129: ACKNOWLEDGE M327-FIXTURE 2 CLEANING VALVE SWITCH OFF / ACKNOWLEDGE M53-SWITCH OFF FIXTURE 2 FLUSH COOLANT VALVE
   RUNG wire#powerrail
      Contact( "M_ZERO" )
      Coil( "DB341_M_UNIT_01_STA_0".M_CODES_UNIT_01_STA_0.Ack_M327 )
   END_RUNG
   // the same network as SCL:
   "DB341_M_UNIT_01_STA_0".M_CODES_UNIT_01_STA_0.Ack_M327 := "M_ZERO";
END_REGION

REGION Network 130: M327-FIXTURE 2 CLEANING VALVE SWITCH OFF / M53-SWITCH OFF FIXTURE 2 FLUSH COOLANT VALVE
   RUNG wire#powerrail
      Contact( "DB331_EXTENDED_M_CODE_UNIT_01_STA_0".M_code[327] )
      I_Contact( "DB341_M_UNIT_01_STA_0".M_CODES_UNIT_01_STA_0.Ack_M327 )
      I_Contact( "DB2120_MPP_ITC_IPC".RESET_FAULTS )
      I_Contact( "DB341_M_UNIT_01_STA_0".M_CODES_UNIT_01_STA_0.M_RESET_PULSE )
      Coil( "DB341_M_UNIT_01_STA_0".M_CODES_UNIT_01_STA_0.M327 )
   END_RUNG
   // the same network as SCL:
   "DB341_M_UNIT_01_STA_0".M_CODES_UNIT_01_STA_0.M327 := "DB331_EXTENDED_M_CODE_UNIT_01_STA_0".M_code[327] AND NOT "DB341_M_UNIT_01_STA_0".M_CODES_UNIT_01_STA_0.Ack_M327 AND NOT "DB2120_MPP_ITC_IPC".RESET_FAULTS AND NOT "DB341_M_UNIT_01_STA_0".M_CODES_UNIT_01_STA_0.M_RESET_PULSE;
END_REGION

REGION Network 131: ACKNOWLEDGE M332-FIXTURE 1 INTERNAL BLOWING SWITCH ON / ACKNOWLEDGE M49-SWITCH OFF FIXTURE 1 INTERNAL BLOWING
   RUNG wire#powerrail
      Contact( "DB341_M_UNIT_01_STA_0".M_CODES_UNIT_01_STA_0.M333 )
      Coil( "DB341_M_UNIT_01_STA_0".M_CODES_UNIT_01_STA_0.Ack_M332 )
   END_RUNG
   // the same network as SCL:
   "DB341_M_UNIT_01_STA_0".M_CODES_UNIT_01_STA_0.Ack_M332 := "DB341_M_UNIT_01_STA_0".M_CODES_UNIT_01_STA_0.M333;
END_REGION

REGION Network 132: M332-FIXTURE 1 INTERNAL BLOWING SWITCH ON / M49-SWITCH OFF FIXTURE 1 INTERNAL BLOWING
   RUNG wire#powerrail
      Contact( "DB331_EXTENDED_M_CODE_UNIT_01_STA_0".M_code[332] )
      wire#w1
      I_Contact( "DB341_M_UNIT_01_STA_0".M_CODES_UNIT_01_STA_0.Ack_M332 )
      I_Contact( "DB2120_MPP_ITC_IPC".RESET_FAULTS )
      I_Contact( "DB341_M_UNIT_01_STA_0".M_CODES_UNIT_01_STA_0.M_RESET_PULSE )
      Coil( "DB341_M_UNIT_01_STA_0".M_CODES_UNIT_01_STA_0.M332 )
   END_RUNG
   RUNG wire#powerrail
      Contact( "DB341_M_UNIT_01_STA_0".M_CODES_UNIT_01_STA_0.M332 )
   END_RUNG wire#w1
   // the same network as SCL:
   "DB341_M_UNIT_01_STA_0".M_CODES_UNIT_01_STA_0.M332 := ("DB331_EXTENDED_M_CODE_UNIT_01_STA_0".M_code[332] OR "DB341_M_UNIT_01_STA_0".M_CODES_UNIT_01_STA_0.M332) AND NOT "DB341_M_UNIT_01_STA_0".M_CODES_UNIT_01_STA_0.Ack_M332 AND NOT "DB2120_MPP_ITC_IPC".RESET_FAULTS AND NOT "DB341_M_UNIT_01_STA_0".M_CODES_UNIT_01_STA_0.M_RESET_PULSE;
END_REGION

REGION Network 133: ACKNOWLEDGE M333-FIXTURE 1 INTERNAL BLOWING SWITCH OFF / ACKNOWLEDGE M56-SWITCH ON FIXTURE 2 INTERNAL BLOWING
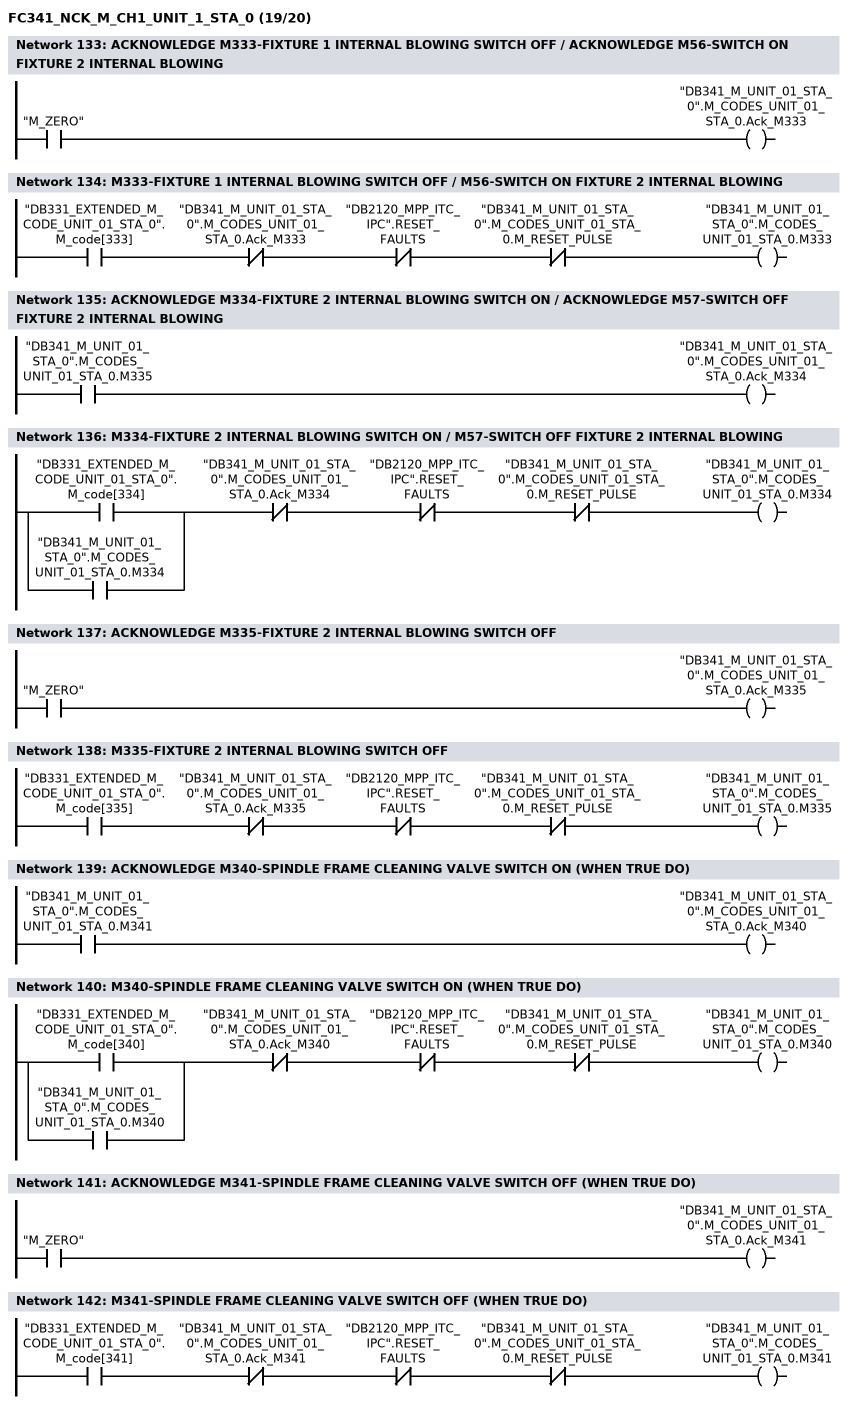
   RUNG wire#powerrail
      Contact( "M_ZERO" )
      Coil( "DB341_M_UNIT_01_STA_0".M_CODES_UNIT_01_STA_0.Ack_M333 )
   END_RUNG
   // the same network as SCL:
   "DB341_M_UNIT_01_STA_0".M_CODES_UNIT_01_STA_0.Ack_M333 := "M_ZERO";
END_REGION

REGION Network 134: M333-FIXTURE 1 INTERNAL BLOWING SWITCH OFF / M56-SWITCH ON FIXTURE 2 INTERNAL BLOWING
   RUNG wire#powerrail
      Contact( "DB331_EXTENDED_M_CODE_UNIT_01_STA_0".M_code[333] )
      I_Contact( "DB341_M_UNIT_01_STA_0".M_CODES_UNIT_01_STA_0.Ack_M333 )
      I_Contact( "DB2120_MPP_ITC_IPC".RESET_FAULTS )
      I_Contact( "DB341_M_UNIT_01_STA_0".M_CODES_UNIT_01_STA_0.M_RESET_PULSE )
      Coil( "DB341_M_UNIT_01_STA_0".M_CODES_UNIT_01_STA_0.M333 )
   END_RUNG
   // the same network as SCL:
   "DB341_M_UNIT_01_STA_0".M_CODES_UNIT_01_STA_0.M333 := "DB331_EXTENDED_M_CODE_UNIT_01_STA_0".M_code[333] AND NOT "DB341_M_UNIT_01_STA_0".M_CODES_UNIT_01_STA_0.Ack_M333 AND NOT "DB2120_MPP_ITC_IPC".RESET_FAULTS AND NOT "DB341_M_UNIT_01_STA_0".M_CODES_UNIT_01_STA_0.M_RESET_PULSE;
END_REGION

REGION Network 135: ACKNOWLEDGE M334-FIXTURE 2 INTERNAL BLOWING SWITCH ON / ACKNOWLEDGE M57-SWITCH OFF FIXTURE 2 INTERNAL BLOWING
   RUNG wire#powerrail
      Contact( "DB341_M_UNIT_01_STA_0".M_CODES_UNIT_01_STA_0.M335 )
      Coil( "DB341_M_UNIT_01_STA_0".M_CODES_UNIT_01_STA_0.Ack_M334 )
   END_RUNG
   // the same network as SCL:
   "DB341_M_UNIT_01_STA_0".M_CODES_UNIT_01_STA_0.Ack_M334 := "DB341_M_UNIT_01_STA_0".M_CODES_UNIT_01_STA_0.M335;
END_REGION

REGION Network 136: M334-FIXTURE 2 INTERNAL BLOWING SWITCH ON / M57-SWITCH OFF FIXTURE 2 INTERNAL BLOWING
   RUNG wire#powerrail
      Contact( "DB331_EXTENDED_M_CODE_UNIT_01_STA_0".M_code[334] )
      wire#w1
      I_Contact( "DB341_M_UNIT_01_STA_0".M_CODES_UNIT_01_STA_0.Ack_M334 )
      I_Contact( "DB2120_MPP_ITC_IPC".RESET_FAULTS )
      I_Contact( "DB341_M_UNIT_01_STA_0".M_CODES_UNIT_01_STA_0.M_RESET_PULSE )
      Coil( "DB341_M_UNIT_01_STA_0".M_CODES_UNIT_01_STA_0.M334 )
   END_RUNG
   RUNG wire#powerrail
      Contact( "DB341_M_UNIT_01_STA_0".M_CODES_UNIT_01_STA_0.M334 )
   END_RUNG wire#w1
   // the same network as SCL:
   "DB341_M_UNIT_01_STA_0".M_CODES_UNIT_01_STA_0.M334 := ("DB331_EXTENDED_M_CODE_UNIT_01_STA_0".M_code[334] OR "DB341_M_UNIT_01_STA_0".M_CODES_UNIT_01_STA_0.M334) AND NOT "DB341_M_UNIT_01_STA_0".M_CODES_UNIT_01_STA_0.Ack_M334 AND NOT "DB2120_MPP_ITC_IPC".RESET_FAULTS AND NOT "DB341_M_UNIT_01_STA_0".M_CODES_UNIT_01_STA_0.M_RESET_PULSE;
END_REGION

